// TIA Portal V17 export
// export: Created 2025-03-07T09:16:41.8974117Z, ExportSetting WithDefaults, DisplayName Totally Integrated Automation Portal, DisplayVersion V17 Update 8, DisplayName TIA Portal Openness, DisplayVersion V17 Update 8, DisplayName TIA Portal Version Control Interface, DisplayVersion V17, DisplayName SINAMICS Startdrive Advanced, DisplayVersion V17 SP2, DisplayName SINAMICS Startdrive G110M, G120, G120C, G120D, G120P, G115D, DisplayVersion V17 SP2, DisplayName SINAMICS Startdrive G130, G150, S120, S150, SINAMICS MV, S210, DisplayVersion V17 SP2, DisplayName STEP 7 Professional, DisplayVersion V17 Update 8, DisplayName SINUMERIK ONE STEP 7 Toolbox, DisplayVersion V17 Update 12, DisplayName SINUMERIK 840D sl STEP 7 Toolbox, DisplayVersion V17 Update 12, DisplayName STEP 7 Safety, DisplayVersion V17 Update 6, DisplayName WinCC Advanced, DisplayVersion V17 Update 8
FUNCTION "FC2440_GLOBAL_DATA_CLADDING" : Void   // FC2440, LAD
{ S7_Optimized_Access := 'FALSE' }
AUTHOR : ETXETAR
VERSION : 1.0
// stored: AutoNumber false, IsIECCheckEnabled false, SetENOAutomatically false, UDAEnableTagReadback false
   VAR_TEMP
      OPTION_ON : Bool;
      OPTION_OFF : Bool;
   END_VAR
   VAR_TEMP   // added for the SCL form of the ladder/FBD networks
      _w1 : Bool;
      _w2 : Bool;
      _w3 : Bool;
      _w4 : Bool;
   END_VAR
BEGIN

REGION Network 1: OPTIONS OFF
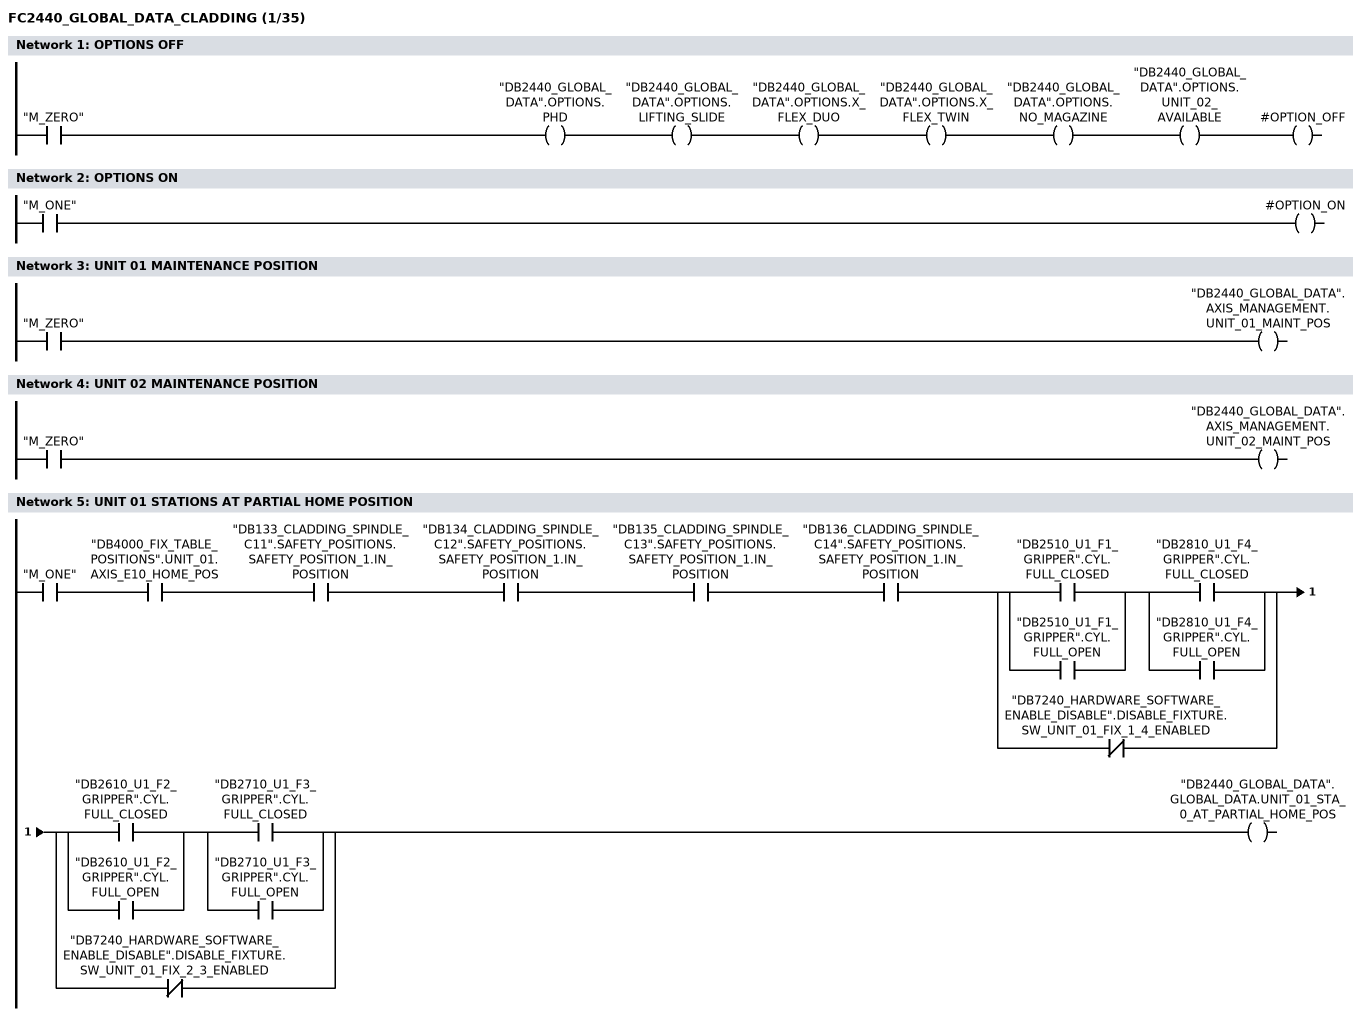
   RUNG wire#powerrail
      Contact( "M_ZERO" )
      Coil( "DB2440_GLOBAL_DATA".OPTIONS.PHD )
      Coil( "DB2440_GLOBAL_DATA".OPTIONS.LIFTING_SLIDE )
      Coil( "DB2440_GLOBAL_DATA".OPTIONS.X_FLEX_DUO )
      Coil( "DB2440_GLOBAL_DATA".OPTIONS.X_FLEX_TWIN )
      Coil( "DB2440_GLOBAL_DATA".OPTIONS.NO_MAGAZINE )
      Coil( "DB2440_GLOBAL_DATA".OPTIONS.UNIT_02_AVAILABLE )
      Coil( #OPTION_OFF )
   END_RUNG
   // the same network as SCL:
   "DB2440_GLOBAL_DATA".OPTIONS.PHD := "M_ZERO";
   "DB2440_GLOBAL_DATA".OPTIONS.LIFTING_SLIDE := "M_ZERO";
   "DB2440_GLOBAL_DATA".OPTIONS.X_FLEX_DUO := "M_ZERO";
   "DB2440_GLOBAL_DATA".OPTIONS.X_FLEX_TWIN := "M_ZERO";
   "DB2440_GLOBAL_DATA".OPTIONS.NO_MAGAZINE := "M_ZERO";
   "DB2440_GLOBAL_DATA".OPTIONS.UNIT_02_AVAILABLE := "M_ZERO";
   #OPTION_OFF := "M_ZERO";
END_REGION

REGION Network 2: OPTIONS ON
   RUNG wire#powerrail
      Contact( "M_ONE" )
      Coil( #OPTION_ON )
   END_RUNG
   // the same network as SCL:
   #OPTION_ON := "M_ONE";
END_REGION

REGION Network 3: UNIT 01 MAINTENANCE POSITION
   RUNG wire#powerrail
      Contact( "M_ZERO" )
      Coil( "DB2440_GLOBAL_DATA".AXIS_MANAGEMENT.UNIT_01_MAINT_POS )
   END_RUNG
   // the same network as SCL:
   "DB2440_GLOBAL_DATA".AXIS_MANAGEMENT.UNIT_01_MAINT_POS := "M_ZERO";
END_REGION

REGION Network 4: UNIT 02 MAINTENANCE POSITION
   RUNG wire#powerrail
      Contact( "M_ZERO" )
      Coil( "DB2440_GLOBAL_DATA".AXIS_MANAGEMENT.UNIT_02_MAINT_POS )
   END_RUNG
   // the same network as SCL:
   "DB2440_GLOBAL_DATA".AXIS_MANAGEMENT.UNIT_02_MAINT_POS := "M_ZERO";
END_REGION

REGION Network 5: UNIT 01 STATIONS AT PARTIAL HOME POSITION
   RUNG wire#powerrail
      Contact( "M_ONE" )
      Contact( "DB4000_FIX_TABLE_POSITIONS".UNIT_01.AXIS_E10_HOME_POS )
      Contact( "DB133_CLADDING_SPINDLE_C11".SAFETY_POSITIONS.SAFETY_POSITION_1.IN_POSITION )
      Contact( "DB134_CLADDING_SPINDLE_C12".SAFETY_POSITIONS.SAFETY_POSITION_1.IN_POSITION )
      Contact( "DB135_CLADDING_SPINDLE_C13".SAFETY_POSITIONS.SAFETY_POSITION_1.IN_POSITION )
      Contact( "DB136_CLADDING_SPINDLE_C14".SAFETY_POSITIONS.SAFETY_POSITION_1.IN_POSITION )
      wire#w1
      Contact( "DB2510_U1_F1_GRIPPER".CYL.FULL_CLOSED )
      wire#w2
      Contact( "DB2810_U1_F4_GRIPPER".CYL.FULL_CLOSED )
      wire#w3
      Contact( "DB2610_U1_F2_GRIPPER".CYL.FULL_CLOSED )
      wire#w4
      Contact( "DB2710_U1_F3_GRIPPER".CYL.FULL_CLOSED )
      wire#w5
      Coil( "DB2440_GLOBAL_DATA".GLOBAL_DATA.UNIT_01_STA_0_AT_PARTIAL_HOME_POS )
   END_RUNG
   RUNG wire#w1
      Contact( "DB2510_U1_F1_GRIPPER".CYL.FULL_OPEN )
   END_RUNG wire#w2
   RUNG wire#w2
      Contact( "DB2810_U1_F4_GRIPPER".CYL.FULL_OPEN )
   END_RUNG wire#w3
   RUNG wire#w1
      I_Contact( "DB7240_HARDWARE_SOFTWARE_ENABLE_DISABLE".DISABLE_FIXTURE.SW_UNIT_01_FIX_1_4_ENABLED )
   END_RUNG wire#w3
   RUNG wire#w3
      Contact( "DB2610_U1_F2_GRIPPER".CYL.FULL_OPEN )
   END_RUNG wire#w4
   RUNG wire#w4
      Contact( "DB2710_U1_F3_GRIPPER".CYL.FULL_OPEN )
   END_RUNG wire#w5
   RUNG wire#w3
      I_Contact( "DB7240_HARDWARE_SOFTWARE_ENABLE_DISABLE".DISABLE_FIXTURE.SW_UNIT_01_FIX_2_3_ENABLED )
   END_RUNG wire#w5
   // the same network as SCL:
   "DB2440_GLOBAL_DATA".GLOBAL_DATA.UNIT_01_STA_0_AT_PARTIAL_HOME_POS := "M_ONE" AND "DB4000_FIX_TABLE_POSITIONS".UNIT_01.AXIS_E10_HOME_POS AND "DB133_CLADDING_SPINDLE_C11".SAFETY_POSITIONS.SAFETY_POSITION_1.IN_POSITION AND "DB134_CLADDING_SPINDLE_C12".SAFETY_POSITIONS.SAFETY_POSITION_1.IN_POSITION AND "DB135_CLADDING_SPINDLE_C13".SAFETY_POSITIONS.SAFETY_POSITION_1.IN_POSITION AND "DB136_CLADDING_SPINDLE_C14".SAFETY_POSITIONS.SAFETY_POSITION_1.IN_POSITION AND ((("DB2510_U1_F1_GRIPPER".CYL.FULL_CLOSED OR "DB2510_U1_F1_GRIPPER".CYL.FULL_OPEN) AND ("DB2810_U1_F4_GRIPPER".CYL.FULL_CLOSED OR "DB2810_U1_F4_GRIPPER".CYL.FULL_OPEN)) OR NOT "DB7240_HARDWARE_SOFTWARE_ENABLE_DISABLE".DISABLE_FIXTURE.SW_UNIT_01_FIX_1_4_ENABLED) AND ((("DB2610_U1_F2_GRIPPER".CYL.FULL_CLOSED OR "DB2610_U1_F2_GRIPPER".CYL.FULL_OPEN) AND ("DB2710_U1_F3_GRIPPER".CYL.FULL_CLOSED OR "DB2710_U1_F3_GRIPPER".CYL.FULL_OPEN)) OR NOT "DB7240_HARDWARE_SOFTWARE_ENABLE_DISABLE".DISABLE_FIXTURE.SW_UNIT_01_FIX_2_3_ENABLED);
END_REGION

REGION Network 6: UNIT 01 STATIONS AT HOME POSITION
   // CILINDERS AND B13
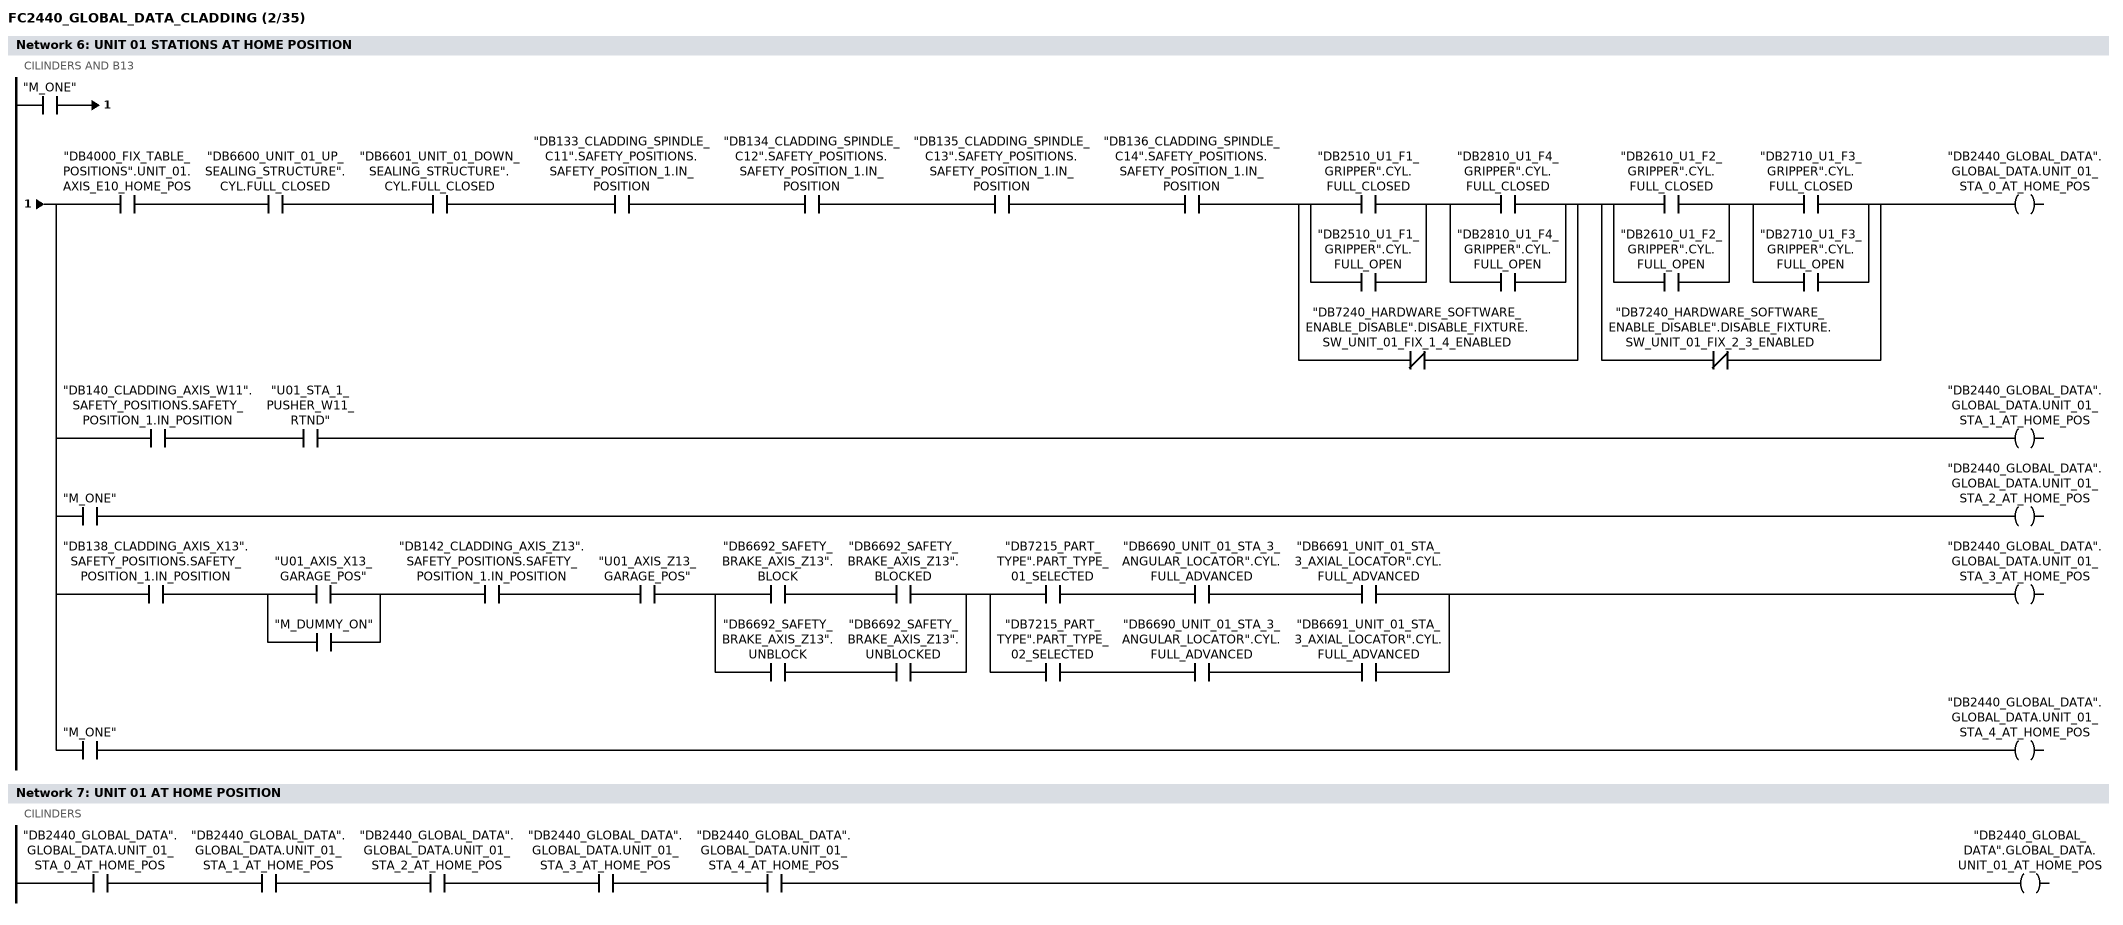
   RUNG wire#powerrail
      Contact( "M_ONE" )
      wire#w1
      Contact( "DB4000_FIX_TABLE_POSITIONS".UNIT_01.AXIS_E10_HOME_POS )
      Contact( "DB6600_UNIT_01_UP_SEALING_STRUCTURE".CYL.FULL_CLOSED )
      Contact( "DB6601_UNIT_01_DOWN_SEALING_STRUCTURE".CYL.FULL_CLOSED )
      Contact( "DB133_CLADDING_SPINDLE_C11".SAFETY_POSITIONS.SAFETY_POSITION_1.IN_POSITION )
      Contact( "DB134_CLADDING_SPINDLE_C12".SAFETY_POSITIONS.SAFETY_POSITION_1.IN_POSITION )
      Contact( "DB135_CLADDING_SPINDLE_C13".SAFETY_POSITIONS.SAFETY_POSITION_1.IN_POSITION )
      Contact( "DB136_CLADDING_SPINDLE_C14".SAFETY_POSITIONS.SAFETY_POSITION_1.IN_POSITION )
      wire#w2
      Contact( "DB2510_U1_F1_GRIPPER".CYL.FULL_CLOSED )
      wire#w3
      Contact( "DB2810_U1_F4_GRIPPER".CYL.FULL_CLOSED )
      wire#w4
      Contact( "DB2610_U1_F2_GRIPPER".CYL.FULL_CLOSED )
      wire#w5
      Contact( "DB2710_U1_F3_GRIPPER".CYL.FULL_CLOSED )
      wire#w6
      Coil( "DB2440_GLOBAL_DATA".GLOBAL_DATA.UNIT_01_STA_0_AT_HOME_POS )
   END_RUNG
   RUNG wire#w2
      Contact( "DB2510_U1_F1_GRIPPER".CYL.FULL_OPEN )
   END_RUNG wire#w3
   RUNG wire#w3
      Contact( "DB2810_U1_F4_GRIPPER".CYL.FULL_OPEN )
   END_RUNG wire#w4
   RUNG wire#w2
      I_Contact( "DB7240_HARDWARE_SOFTWARE_ENABLE_DISABLE".DISABLE_FIXTURE.SW_UNIT_01_FIX_1_4_ENABLED )
   END_RUNG wire#w4
   RUNG wire#w4
      Contact( "DB2610_U1_F2_GRIPPER".CYL.FULL_OPEN )
   END_RUNG wire#w5
   RUNG wire#w5
      Contact( "DB2710_U1_F3_GRIPPER".CYL.FULL_OPEN )
   END_RUNG wire#w6
   RUNG wire#w4
      I_Contact( "DB7240_HARDWARE_SOFTWARE_ENABLE_DISABLE".DISABLE_FIXTURE.SW_UNIT_01_FIX_2_3_ENABLED )
   END_RUNG wire#w6
   RUNG wire#w1
      Contact( "DB140_CLADDING_AXIS_W11".SAFETY_POSITIONS.SAFETY_POSITION_1.IN_POSITION )
      Contact( "U01_STA_1_PUSHER_W11_RTND" )
      Coil( "DB2440_GLOBAL_DATA".GLOBAL_DATA.UNIT_01_STA_1_AT_HOME_POS )
   END_RUNG
   RUNG wire#w1
      Contact( "M_ONE" )
      Coil( "DB2440_GLOBAL_DATA".GLOBAL_DATA.UNIT_01_STA_2_AT_HOME_POS )
   END_RUNG
   RUNG wire#w1
      Contact( "DB138_CLADDING_AXIS_X13".SAFETY_POSITIONS.SAFETY_POSITION_1.IN_POSITION )
      wire#w7
      Contact( "U01_AXIS_X13_GARAGE_POS" )
      wire#w8
      Contact( "DB142_CLADDING_AXIS_Z13".SAFETY_POSITIONS.SAFETY_POSITION_1.IN_POSITION )
      Contact( "U01_AXIS_Z13_GARAGE_POS" )
      wire#w9
      Contact( "DB6692_SAFETY_BRAKE_AXIS_Z13".BLOCK )
      Contact( "DB6692_SAFETY_BRAKE_AXIS_Z13".BLOCKED )
      wire#w10
      Contact( "DB7215_PART_TYPE".PART_TYPE_01_SELECTED )
      Contact( "DB6690_UNIT_01_STA_3_ANGULAR_LOCATOR".CYL.FULL_ADVANCED )
      Contact( "DB6691_UNIT_01_STA_3_AXIAL_LOCATOR".CYL.FULL_ADVANCED )
      wire#w11
      Coil( "DB2440_GLOBAL_DATA".GLOBAL_DATA.UNIT_01_STA_3_AT_HOME_POS )
   END_RUNG
   RUNG wire#w7
      Contact( "M_DUMMY_ON" )
   END_RUNG wire#w8
   RUNG wire#w9
      Contact( "DB6692_SAFETY_BRAKE_AXIS_Z13".UNBLOCK )
      Contact( "DB6692_SAFETY_BRAKE_AXIS_Z13".UNBLOCKED )
   END_RUNG wire#w10
   RUNG wire#w10
      Contact( "DB7215_PART_TYPE".PART_TYPE_02_SELECTED )
      Contact( "DB6690_UNIT_01_STA_3_ANGULAR_LOCATOR".CYL.FULL_ADVANCED )
      Contact( "DB6691_UNIT_01_STA_3_AXIAL_LOCATOR".CYL.FULL_ADVANCED )
   END_RUNG wire#w11
   RUNG wire#w1
      Contact( "M_ONE" )
      Coil( "DB2440_GLOBAL_DATA".GLOBAL_DATA.UNIT_01_STA_4_AT_HOME_POS )
   END_RUNG
   // the same network as SCL:
   "DB2440_GLOBAL_DATA".GLOBAL_DATA.UNIT_01_STA_0_AT_HOME_POS := "M_ONE" AND "DB4000_FIX_TABLE_POSITIONS".UNIT_01.AXIS_E10_HOME_POS AND "DB6600_UNIT_01_UP_SEALING_STRUCTURE".CYL.FULL_CLOSED AND "DB6601_UNIT_01_DOWN_SEALING_STRUCTURE".CYL.FULL_CLOSED AND "DB133_CLADDING_SPINDLE_C11".SAFETY_POSITIONS.SAFETY_POSITION_1.IN_POSITION AND "DB134_CLADDING_SPINDLE_C12".SAFETY_POSITIONS.SAFETY_POSITION_1.IN_POSITION AND "DB135_CLADDING_SPINDLE_C13".SAFETY_POSITIONS.SAFETY_POSITION_1.IN_POSITION AND "DB136_CLADDING_SPINDLE_C14".SAFETY_POSITIONS.SAFETY_POSITION_1.IN_POSITION AND ((("DB2510_U1_F1_GRIPPER".CYL.FULL_CLOSED OR "DB2510_U1_F1_GRIPPER".CYL.FULL_OPEN) AND ("DB2810_U1_F4_GRIPPER".CYL.FULL_CLOSED OR "DB2810_U1_F4_GRIPPER".CYL.FULL_OPEN)) OR NOT "DB7240_HARDWARE_SOFTWARE_ENABLE_DISABLE".DISABLE_FIXTURE.SW_UNIT_01_FIX_1_4_ENABLED) AND ((("DB2610_U1_F2_GRIPPER".CYL.FULL_CLOSED OR "DB2610_U1_F2_GRIPPER".CYL.FULL_OPEN) AND ("DB2710_U1_F3_GRIPPER".CYL.FULL_CLOSED OR "DB2710_U1_F3_GRIPPER".CYL.FULL_OPEN)) OR NOT "DB7240_HARDWARE_SOFTWARE_ENABLE_DISABLE".DISABLE_FIXTURE.SW_UNIT_01_FIX_2_3_ENABLED);
   "DB2440_GLOBAL_DATA".GLOBAL_DATA.UNIT_01_STA_1_AT_HOME_POS := "M_ONE" AND "DB140_CLADDING_AXIS_W11".SAFETY_POSITIONS.SAFETY_POSITION_1.IN_POSITION AND "U01_STA_1_PUSHER_W11_RTND";
   "DB2440_GLOBAL_DATA".GLOBAL_DATA.UNIT_01_STA_2_AT_HOME_POS := "M_ONE" AND "M_ONE";
   "DB2440_GLOBAL_DATA".GLOBAL_DATA.UNIT_01_STA_3_AT_HOME_POS := "M_ONE" AND "DB138_CLADDING_AXIS_X13".SAFETY_POSITIONS.SAFETY_POSITION_1.IN_POSITION AND ("U01_AXIS_X13_GARAGE_POS" OR "M_DUMMY_ON") AND "DB142_CLADDING_AXIS_Z13".SAFETY_POSITIONS.SAFETY_POSITION_1.IN_POSITION AND "U01_AXIS_Z13_GARAGE_POS" AND (("DB6692_SAFETY_BRAKE_AXIS_Z13".BLOCK AND "DB6692_SAFETY_BRAKE_AXIS_Z13".BLOCKED) OR ("DB6692_SAFETY_BRAKE_AXIS_Z13".UNBLOCK AND "DB6692_SAFETY_BRAKE_AXIS_Z13".UNBLOCKED)) AND (("DB7215_PART_TYPE".PART_TYPE_01_SELECTED AND "DB6690_UNIT_01_STA_3_ANGULAR_LOCATOR".CYL.FULL_ADVANCED AND "DB6691_UNIT_01_STA_3_AXIAL_LOCATOR".CYL.FULL_ADVANCED) OR ("DB7215_PART_TYPE".PART_TYPE_02_SELECTED AND "DB6690_UNIT_01_STA_3_ANGULAR_LOCATOR".CYL.FULL_ADVANCED AND "DB6691_UNIT_01_STA_3_AXIAL_LOCATOR".CYL.FULL_ADVANCED));
   "DB2440_GLOBAL_DATA".GLOBAL_DATA.UNIT_01_STA_4_AT_HOME_POS := "M_ONE" AND "M_ONE";
END_REGION

REGION Network 7: UNIT 01 AT HOME POSITION
   // CILINDERS
   RUNG wire#powerrail
      Contact( "DB2440_GLOBAL_DATA".GLOBAL_DATA.UNIT_01_STA_0_AT_HOME_POS )
      Contact( "DB2440_GLOBAL_DATA".GLOBAL_DATA.UNIT_01_STA_1_AT_HOME_POS )
      Contact( "DB2440_GLOBAL_DATA".GLOBAL_DATA.UNIT_01_STA_2_AT_HOME_POS )
      Contact( "DB2440_GLOBAL_DATA".GLOBAL_DATA.UNIT_01_STA_3_AT_HOME_POS )
      Contact( "DB2440_GLOBAL_DATA".GLOBAL_DATA.UNIT_01_STA_4_AT_HOME_POS )
      Coil( "DB2440_GLOBAL_DATA".GLOBAL_DATA.UNIT_01_AT_HOME_POS )
   END_RUNG
   // the same network as SCL:
   "DB2440_GLOBAL_DATA".GLOBAL_DATA.UNIT_01_AT_HOME_POS := "DB2440_GLOBAL_DATA".GLOBAL_DATA.UNIT_01_STA_0_AT_HOME_POS AND "DB2440_GLOBAL_DATA".GLOBAL_DATA.UNIT_01_STA_1_AT_HOME_POS AND "DB2440_GLOBAL_DATA".GLOBAL_DATA.UNIT_01_STA_2_AT_HOME_POS AND "DB2440_GLOBAL_DATA".GLOBAL_DATA.UNIT_01_STA_3_AT_HOME_POS AND "DB2440_GLOBAL_DATA".GLOBAL_DATA.UNIT_01_STA_4_AT_HOME_POS;
END_REGION

REGION Network 8: UNIT 02 STATIONS AT PARTIAL HOME POSITION
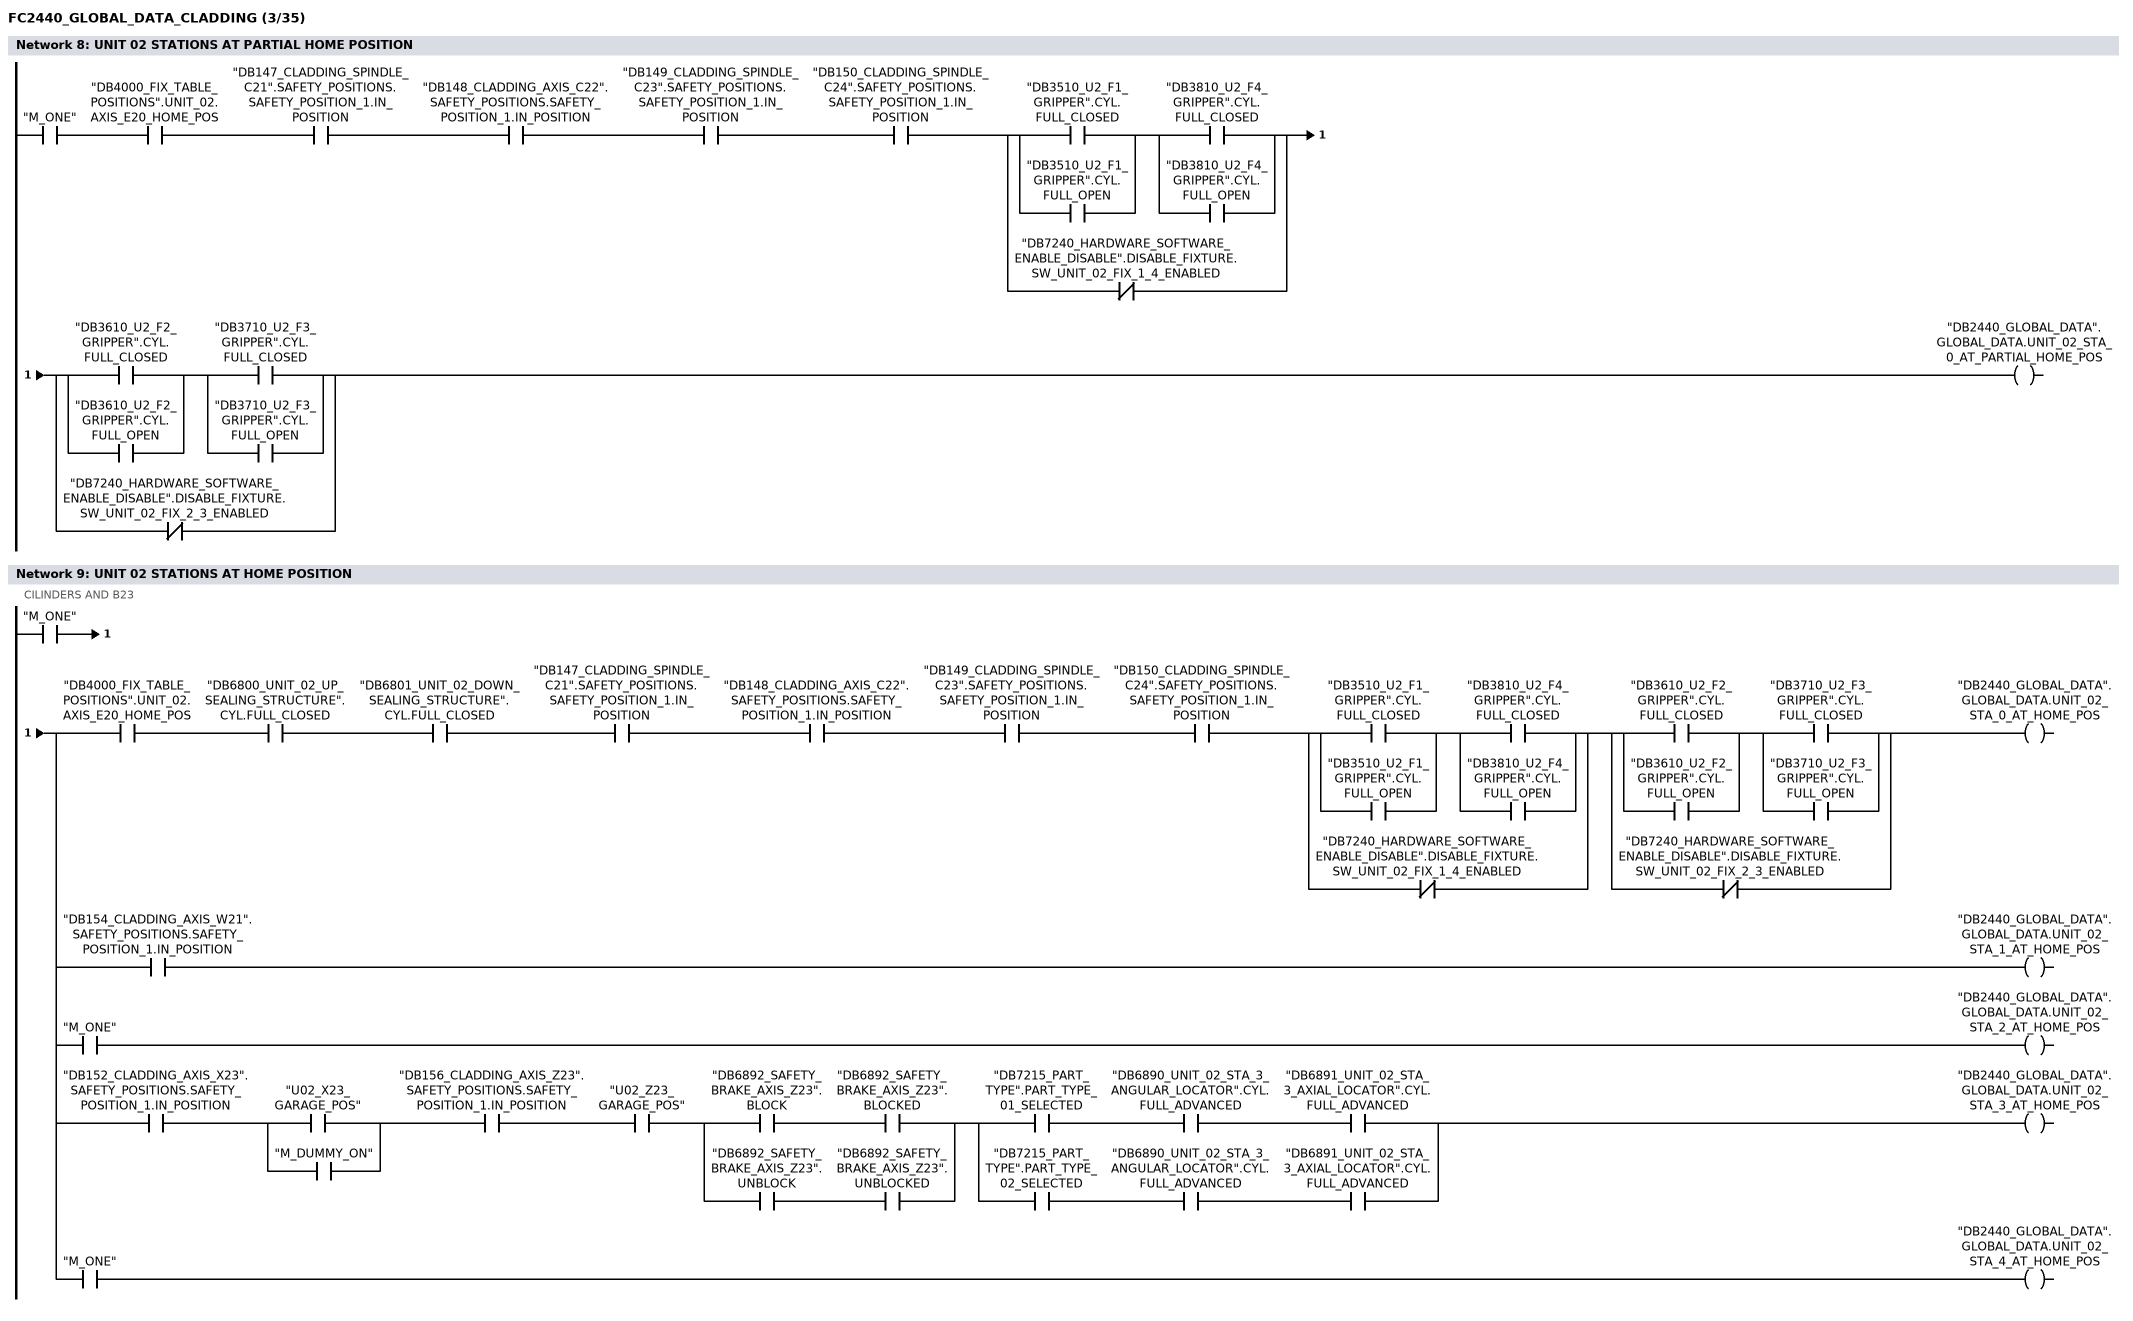
   RUNG wire#powerrail
      Contact( "M_ONE" )
      Contact( "DB4000_FIX_TABLE_POSITIONS".UNIT_02.AXIS_E20_HOME_POS )
      Contact( "DB147_CLADDING_SPINDLE_C21".SAFETY_POSITIONS.SAFETY_POSITION_1.IN_POSITION )
      Contact( "DB148_CLADDING_AXIS_C22".SAFETY_POSITIONS.SAFETY_POSITION_1.IN_POSITION )
      Contact( "DB149_CLADDING_SPINDLE_C23".SAFETY_POSITIONS.SAFETY_POSITION_1.IN_POSITION )
      Contact( "DB150_CLADDING_SPINDLE_C24".SAFETY_POSITIONS.SAFETY_POSITION_1.IN_POSITION )
      wire#w1
      Contact( "DB3510_U2_F1_GRIPPER".CYL.FULL_CLOSED )
      wire#w2
      Contact( "DB3810_U2_F4_GRIPPER".CYL.FULL_CLOSED )
      wire#w3
      Contact( "DB3610_U2_F2_GRIPPER".CYL.FULL_CLOSED )
      wire#w4
      Contact( "DB3710_U2_F3_GRIPPER".CYL.FULL_CLOSED )
      wire#w5
      Coil( "DB2440_GLOBAL_DATA".GLOBAL_DATA.UNIT_02_STA_0_AT_PARTIAL_HOME_POS )
   END_RUNG
   RUNG wire#w1
      Contact( "DB3510_U2_F1_GRIPPER".CYL.FULL_OPEN )
   END_RUNG wire#w2
   RUNG wire#w2
      Contact( "DB3810_U2_F4_GRIPPER".CYL.FULL_OPEN )
   END_RUNG wire#w3
   RUNG wire#w1
      I_Contact( "DB7240_HARDWARE_SOFTWARE_ENABLE_DISABLE".DISABLE_FIXTURE.SW_UNIT_02_FIX_1_4_ENABLED )
   END_RUNG wire#w3
   RUNG wire#w3
      Contact( "DB3610_U2_F2_GRIPPER".CYL.FULL_OPEN )
   END_RUNG wire#w4
   RUNG wire#w4
      Contact( "DB3710_U2_F3_GRIPPER".CYL.FULL_OPEN )
   END_RUNG wire#w5
   RUNG wire#w3
      I_Contact( "DB7240_HARDWARE_SOFTWARE_ENABLE_DISABLE".DISABLE_FIXTURE.SW_UNIT_02_FIX_2_3_ENABLED )
   END_RUNG wire#w5
   // the same network as SCL:
   "DB2440_GLOBAL_DATA".GLOBAL_DATA.UNIT_02_STA_0_AT_PARTIAL_HOME_POS := "M_ONE" AND "DB4000_FIX_TABLE_POSITIONS".UNIT_02.AXIS_E20_HOME_POS AND "DB147_CLADDING_SPINDLE_C21".SAFETY_POSITIONS.SAFETY_POSITION_1.IN_POSITION AND "DB148_CLADDING_AXIS_C22".SAFETY_POSITIONS.SAFETY_POSITION_1.IN_POSITION AND "DB149_CLADDING_SPINDLE_C23".SAFETY_POSITIONS.SAFETY_POSITION_1.IN_POSITION AND "DB150_CLADDING_SPINDLE_C24".SAFETY_POSITIONS.SAFETY_POSITION_1.IN_POSITION AND ((("DB3510_U2_F1_GRIPPER".CYL.FULL_CLOSED OR "DB3510_U2_F1_GRIPPER".CYL.FULL_OPEN) AND ("DB3810_U2_F4_GRIPPER".CYL.FULL_CLOSED OR "DB3810_U2_F4_GRIPPER".CYL.FULL_OPEN)) OR NOT "DB7240_HARDWARE_SOFTWARE_ENABLE_DISABLE".DISABLE_FIXTURE.SW_UNIT_02_FIX_1_4_ENABLED) AND ((("DB3610_U2_F2_GRIPPER".CYL.FULL_CLOSED OR "DB3610_U2_F2_GRIPPER".CYL.FULL_OPEN) AND ("DB3710_U2_F3_GRIPPER".CYL.FULL_CLOSED OR "DB3710_U2_F3_GRIPPER".CYL.FULL_OPEN)) OR NOT "DB7240_HARDWARE_SOFTWARE_ENABLE_DISABLE".DISABLE_FIXTURE.SW_UNIT_02_FIX_2_3_ENABLED);
END_REGION

REGION Network 9: UNIT 02 STATIONS AT HOME POSITION
   // CILINDERS AND B23
   RUNG wire#powerrail
      Contact( "M_ONE" )
      wire#w1
      Contact( "DB4000_FIX_TABLE_POSITIONS".UNIT_02.AXIS_E20_HOME_POS )
      Contact( "DB6800_UNIT_02_UP_SEALING_STRUCTURE".CYL.FULL_CLOSED )
      Contact( "DB6801_UNIT_02_DOWN_SEALING_STRUCTURE".CYL.FULL_CLOSED )
      Contact( "DB147_CLADDING_SPINDLE_C21".SAFETY_POSITIONS.SAFETY_POSITION_1.IN_POSITION )
      Contact( "DB148_CLADDING_AXIS_C22".SAFETY_POSITIONS.SAFETY_POSITION_1.IN_POSITION )
      Contact( "DB149_CLADDING_SPINDLE_C23".SAFETY_POSITIONS.SAFETY_POSITION_1.IN_POSITION )
      Contact( "DB150_CLADDING_SPINDLE_C24".SAFETY_POSITIONS.SAFETY_POSITION_1.IN_POSITION )
      wire#w2
      Contact( "DB3510_U2_F1_GRIPPER".CYL.FULL_CLOSED )
      wire#w3
      Contact( "DB3810_U2_F4_GRIPPER".CYL.FULL_CLOSED )
      wire#w4
      Contact( "DB3610_U2_F2_GRIPPER".CYL.FULL_CLOSED )
      wire#w5
      Contact( "DB3710_U2_F3_GRIPPER".CYL.FULL_CLOSED )
      wire#w6
      Coil( "DB2440_GLOBAL_DATA".GLOBAL_DATA.UNIT_02_STA_0_AT_HOME_POS )
   END_RUNG
   RUNG wire#w2
      Contact( "DB3510_U2_F1_GRIPPER".CYL.FULL_OPEN )
   END_RUNG wire#w3
   RUNG wire#w3
      Contact( "DB3810_U2_F4_GRIPPER".CYL.FULL_OPEN )
   END_RUNG wire#w4
   RUNG wire#w2
      I_Contact( "DB7240_HARDWARE_SOFTWARE_ENABLE_DISABLE".DISABLE_FIXTURE.SW_UNIT_02_FIX_1_4_ENABLED )
   END_RUNG wire#w4
   RUNG wire#w4
      Contact( "DB3610_U2_F2_GRIPPER".CYL.FULL_OPEN )
   END_RUNG wire#w5
   RUNG wire#w5
      Contact( "DB3710_U2_F3_GRIPPER".CYL.FULL_OPEN )
   END_RUNG wire#w6
   RUNG wire#w4
      I_Contact( "DB7240_HARDWARE_SOFTWARE_ENABLE_DISABLE".DISABLE_FIXTURE.SW_UNIT_02_FIX_2_3_ENABLED )
   END_RUNG wire#w6
   RUNG wire#w1
      Contact( "DB154_CLADDING_AXIS_W21".SAFETY_POSITIONS.SAFETY_POSITION_1.IN_POSITION )
      Coil( "DB2440_GLOBAL_DATA".GLOBAL_DATA.UNIT_02_STA_1_AT_HOME_POS )
   END_RUNG
   RUNG wire#w1
      Contact( "M_ONE" )
      Coil( "DB2440_GLOBAL_DATA".GLOBAL_DATA.UNIT_02_STA_2_AT_HOME_POS )
   END_RUNG
   RUNG wire#w1
      Contact( "DB152_CLADDING_AXIS_X23".SAFETY_POSITIONS.SAFETY_POSITION_1.IN_POSITION )
      wire#w7
      Contact( "U02_X23_GARAGE_POS" )
      wire#w8
      Contact( "DB156_CLADDING_AXIS_Z23".SAFETY_POSITIONS.SAFETY_POSITION_1.IN_POSITION )
      Contact( "U02_Z23_GARAGE_POS" )
      wire#w9
      Contact( "DB6892_SAFETY_BRAKE_AXIS_Z23".BLOCK )
      Contact( "DB6892_SAFETY_BRAKE_AXIS_Z23".BLOCKED )
      wire#w10
      Contact( "DB7215_PART_TYPE".PART_TYPE_01_SELECTED )
      Contact( "DB6890_UNIT_02_STA_3_ANGULAR_LOCATOR".CYL.FULL_ADVANCED )
      Contact( "DB6891_UNIT_02_STA_3_AXIAL_LOCATOR".CYL.FULL_ADVANCED )
      wire#w11
      Coil( "DB2440_GLOBAL_DATA".GLOBAL_DATA.UNIT_02_STA_3_AT_HOME_POS )
   END_RUNG
   RUNG wire#w7
      Contact( "M_DUMMY_ON" )
   END_RUNG wire#w8
   RUNG wire#w9
      Contact( "DB6892_SAFETY_BRAKE_AXIS_Z23".UNBLOCK )
      Contact( "DB6892_SAFETY_BRAKE_AXIS_Z23".UNBLOCKED )
   END_RUNG wire#w10
   RUNG wire#w10
      Contact( "DB7215_PART_TYPE".PART_TYPE_02_SELECTED )
      Contact( "DB6890_UNIT_02_STA_3_ANGULAR_LOCATOR".CYL.FULL_ADVANCED )
      Contact( "DB6891_UNIT_02_STA_3_AXIAL_LOCATOR".CYL.FULL_ADVANCED )
   END_RUNG wire#w11
   RUNG wire#w1
      Contact( "M_ONE" )
      Coil( "DB2440_GLOBAL_DATA".GLOBAL_DATA.UNIT_02_STA_4_AT_HOME_POS )
   END_RUNG
   // the same network as SCL:
   "DB2440_GLOBAL_DATA".GLOBAL_DATA.UNIT_02_STA_0_AT_HOME_POS := "M_ONE" AND "DB4000_FIX_TABLE_POSITIONS".UNIT_02.AXIS_E20_HOME_POS AND "DB6800_UNIT_02_UP_SEALING_STRUCTURE".CYL.FULL_CLOSED AND "DB6801_UNIT_02_DOWN_SEALING_STRUCTURE".CYL.FULL_CLOSED AND "DB147_CLADDING_SPINDLE_C21".SAFETY_POSITIONS.SAFETY_POSITION_1.IN_POSITION AND "DB148_CLADDING_AXIS_C22".SAFETY_POSITIONS.SAFETY_POSITION_1.IN_POSITION AND "DB149_CLADDING_SPINDLE_C23".SAFETY_POSITIONS.SAFETY_POSITION_1.IN_POSITION AND "DB150_CLADDING_SPINDLE_C24".SAFETY_POSITIONS.SAFETY_POSITION_1.IN_POSITION AND ((("DB3510_U2_F1_GRIPPER".CYL.FULL_CLOSED OR "DB3510_U2_F1_GRIPPER".CYL.FULL_OPEN) AND ("DB3810_U2_F4_GRIPPER".CYL.FULL_CLOSED OR "DB3810_U2_F4_GRIPPER".CYL.FULL_OPEN)) OR NOT "DB7240_HARDWARE_SOFTWARE_ENABLE_DISABLE".DISABLE_FIXTURE.SW_UNIT_02_FIX_1_4_ENABLED) AND ((("DB3610_U2_F2_GRIPPER".CYL.FULL_CLOSED OR "DB3610_U2_F2_GRIPPER".CYL.FULL_OPEN) AND ("DB3710_U2_F3_GRIPPER".CYL.FULL_CLOSED OR "DB3710_U2_F3_GRIPPER".CYL.FULL_OPEN)) OR NOT "DB7240_HARDWARE_SOFTWARE_ENABLE_DISABLE".DISABLE_FIXTURE.SW_UNIT_02_FIX_2_3_ENABLED);
   "DB2440_GLOBAL_DATA".GLOBAL_DATA.UNIT_02_STA_1_AT_HOME_POS := "M_ONE" AND "DB154_CLADDING_AXIS_W21".SAFETY_POSITIONS.SAFETY_POSITION_1.IN_POSITION;
   "DB2440_GLOBAL_DATA".GLOBAL_DATA.UNIT_02_STA_2_AT_HOME_POS := "M_ONE" AND "M_ONE";
   "DB2440_GLOBAL_DATA".GLOBAL_DATA.UNIT_02_STA_3_AT_HOME_POS := "M_ONE" AND "DB152_CLADDING_AXIS_X23".SAFETY_POSITIONS.SAFETY_POSITION_1.IN_POSITION AND ("U02_X23_GARAGE_POS" OR "M_DUMMY_ON") AND "DB156_CLADDING_AXIS_Z23".SAFETY_POSITIONS.SAFETY_POSITION_1.IN_POSITION AND "U02_Z23_GARAGE_POS" AND (("DB6892_SAFETY_BRAKE_AXIS_Z23".BLOCK AND "DB6892_SAFETY_BRAKE_AXIS_Z23".BLOCKED) OR ("DB6892_SAFETY_BRAKE_AXIS_Z23".UNBLOCK AND "DB6892_SAFETY_BRAKE_AXIS_Z23".UNBLOCKED)) AND (("DB7215_PART_TYPE".PART_TYPE_01_SELECTED AND "DB6890_UNIT_02_STA_3_ANGULAR_LOCATOR".CYL.FULL_ADVANCED AND "DB6891_UNIT_02_STA_3_AXIAL_LOCATOR".CYL.FULL_ADVANCED) OR ("DB7215_PART_TYPE".PART_TYPE_02_SELECTED AND "DB6890_UNIT_02_STA_3_ANGULAR_LOCATOR".CYL.FULL_ADVANCED AND "DB6891_UNIT_02_STA_3_AXIAL_LOCATOR".CYL.FULL_ADVANCED));
   "DB2440_GLOBAL_DATA".GLOBAL_DATA.UNIT_02_STA_4_AT_HOME_POS := "M_ONE" AND "M_ONE";
END_REGION

REGION Network 10: UNIT 02 AT HOME POSITION
   // CILINDERS
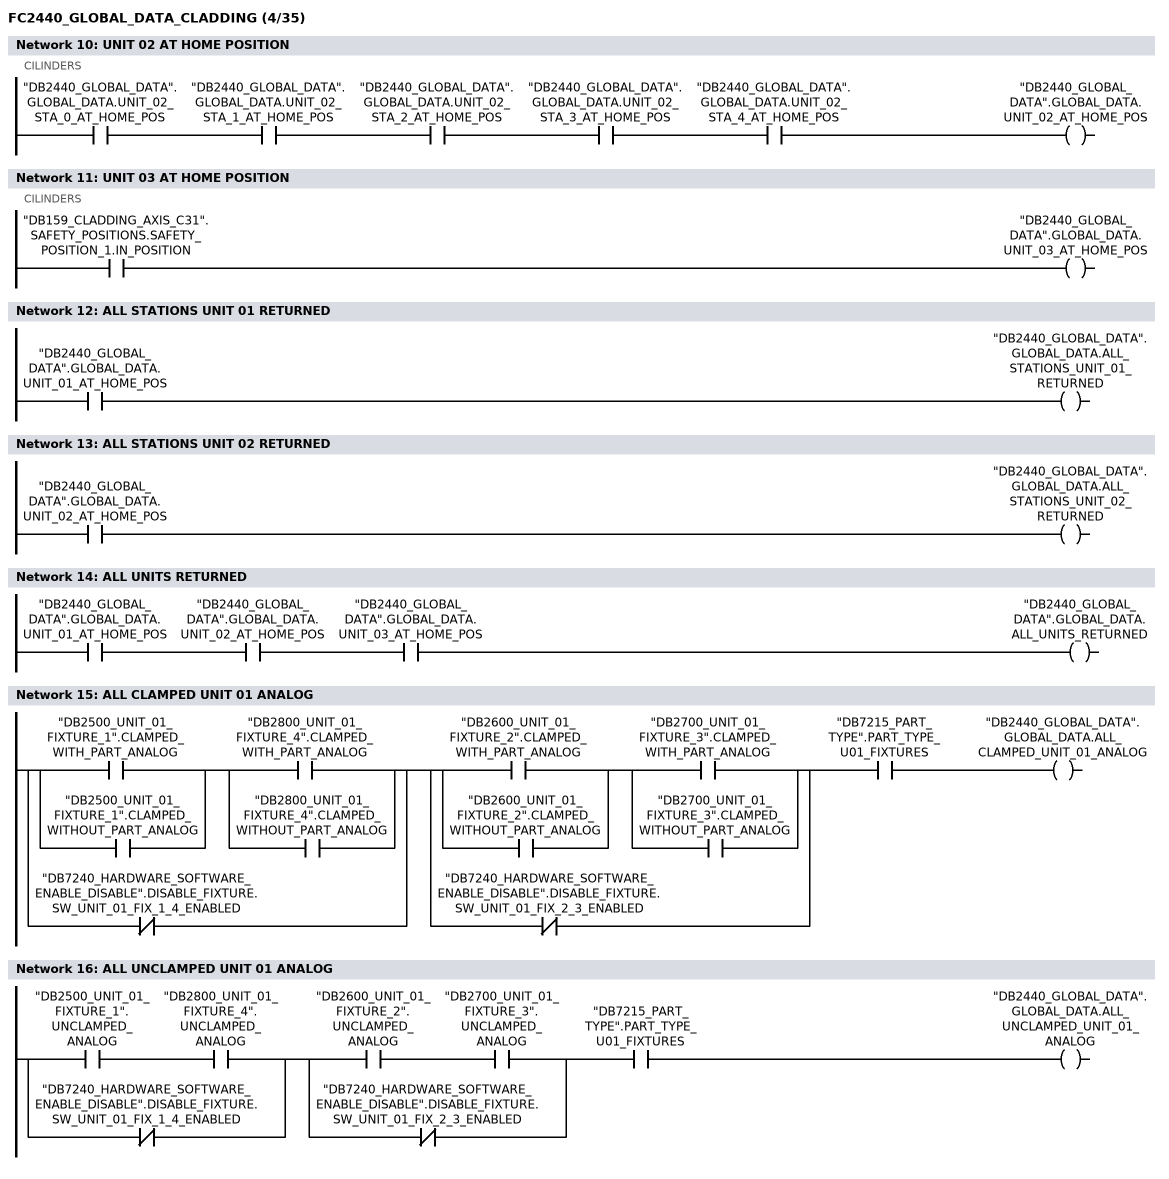
   RUNG wire#powerrail
      Contact( "DB2440_GLOBAL_DATA".GLOBAL_DATA.UNIT_02_STA_0_AT_HOME_POS )
      Contact( "DB2440_GLOBAL_DATA".GLOBAL_DATA.UNIT_02_STA_1_AT_HOME_POS )
      Contact( "DB2440_GLOBAL_DATA".GLOBAL_DATA.UNIT_02_STA_2_AT_HOME_POS )
      Contact( "DB2440_GLOBAL_DATA".GLOBAL_DATA.UNIT_02_STA_3_AT_HOME_POS )
      Contact( "DB2440_GLOBAL_DATA".GLOBAL_DATA.UNIT_02_STA_4_AT_HOME_POS )
      Coil( "DB2440_GLOBAL_DATA".GLOBAL_DATA.UNIT_02_AT_HOME_POS )
   END_RUNG
   // the same network as SCL:
   "DB2440_GLOBAL_DATA".GLOBAL_DATA.UNIT_02_AT_HOME_POS := "DB2440_GLOBAL_DATA".GLOBAL_DATA.UNIT_02_STA_0_AT_HOME_POS AND "DB2440_GLOBAL_DATA".GLOBAL_DATA.UNIT_02_STA_1_AT_HOME_POS AND "DB2440_GLOBAL_DATA".GLOBAL_DATA.UNIT_02_STA_2_AT_HOME_POS AND "DB2440_GLOBAL_DATA".GLOBAL_DATA.UNIT_02_STA_3_AT_HOME_POS AND "DB2440_GLOBAL_DATA".GLOBAL_DATA.UNIT_02_STA_4_AT_HOME_POS;
END_REGION

REGION Network 11: UNIT 03 AT HOME POSITION
   // CILINDERS
   RUNG wire#powerrail
      Contact( "DB159_CLADDING_AXIS_C31".SAFETY_POSITIONS.SAFETY_POSITION_1.IN_POSITION )
      Coil( "DB2440_GLOBAL_DATA".GLOBAL_DATA.UNIT_03_AT_HOME_POS )
   END_RUNG
   // the same network as SCL:
   "DB2440_GLOBAL_DATA".GLOBAL_DATA.UNIT_03_AT_HOME_POS := "DB159_CLADDING_AXIS_C31".SAFETY_POSITIONS.SAFETY_POSITION_1.IN_POSITION;
END_REGION

REGION Network 12: ALL STATIONS UNIT 01 RETURNED
   RUNG wire#powerrail
      Contact( "DB2440_GLOBAL_DATA".GLOBAL_DATA.UNIT_01_AT_HOME_POS )
      Coil( "DB2440_GLOBAL_DATA".GLOBAL_DATA.ALL_STATIONS_UNIT_01_RETURNED )
   END_RUNG
   // the same network as SCL:
   "DB2440_GLOBAL_DATA".GLOBAL_DATA.ALL_STATIONS_UNIT_01_RETURNED := "DB2440_GLOBAL_DATA".GLOBAL_DATA.UNIT_01_AT_HOME_POS;
END_REGION

REGION Network 13: ALL STATIONS UNIT 02 RETURNED
   RUNG wire#powerrail
      Contact( "DB2440_GLOBAL_DATA".GLOBAL_DATA.UNIT_02_AT_HOME_POS )
      Coil( "DB2440_GLOBAL_DATA".GLOBAL_DATA.ALL_STATIONS_UNIT_02_RETURNED )
   END_RUNG
   // the same network as SCL:
   "DB2440_GLOBAL_DATA".GLOBAL_DATA.ALL_STATIONS_UNIT_02_RETURNED := "DB2440_GLOBAL_DATA".GLOBAL_DATA.UNIT_02_AT_HOME_POS;
END_REGION

REGION Network 14: ALL UNITS RETURNED
   RUNG wire#powerrail
      Contact( "DB2440_GLOBAL_DATA".GLOBAL_DATA.UNIT_01_AT_HOME_POS )
      Contact( "DB2440_GLOBAL_DATA".GLOBAL_DATA.UNIT_02_AT_HOME_POS )
      Contact( "DB2440_GLOBAL_DATA".GLOBAL_DATA.UNIT_03_AT_HOME_POS )
      Coil( "DB2440_GLOBAL_DATA".GLOBAL_DATA.ALL_UNITS_RETURNED )
   END_RUNG
   // the same network as SCL:
   "DB2440_GLOBAL_DATA".GLOBAL_DATA.ALL_UNITS_RETURNED := "DB2440_GLOBAL_DATA".GLOBAL_DATA.UNIT_01_AT_HOME_POS AND "DB2440_GLOBAL_DATA".GLOBAL_DATA.UNIT_02_AT_HOME_POS AND "DB2440_GLOBAL_DATA".GLOBAL_DATA.UNIT_03_AT_HOME_POS;
END_REGION

REGION Network 15: ALL CLAMPED UNIT 01 ANALOG
   RUNG wire#powerrail
      Contact( "DB2500_UNIT_01_FIXTURE_1".CLAMPED_WITH_PART_ANALOG )
      wire#w1
      Contact( "DB2800_UNIT_01_FIXTURE_4".CLAMPED_WITH_PART_ANALOG )
      wire#w2
      Contact( "DB2600_UNIT_01_FIXTURE_2".CLAMPED_WITH_PART_ANALOG )
      wire#w3
      Contact( "DB2700_UNIT_01_FIXTURE_3".CLAMPED_WITH_PART_ANALOG )
      wire#w4
      Contact( "DB7215_PART_TYPE".PART_TYPE_U01_FIXTURES )
      Coil( "DB2440_GLOBAL_DATA".GLOBAL_DATA.ALL_CLAMPED_UNIT_01_ANALOG )
   END_RUNG
   RUNG wire#powerrail
      Contact( "DB2500_UNIT_01_FIXTURE_1".CLAMPED_WITHOUT_PART_ANALOG )
   END_RUNG wire#w1
   RUNG wire#w1
      Contact( "DB2800_UNIT_01_FIXTURE_4".CLAMPED_WITHOUT_PART_ANALOG )
   END_RUNG wire#w2
   RUNG wire#powerrail
      I_Contact( "DB7240_HARDWARE_SOFTWARE_ENABLE_DISABLE".DISABLE_FIXTURE.SW_UNIT_01_FIX_1_4_ENABLED )
   END_RUNG wire#w2
   RUNG wire#w2
      Contact( "DB2600_UNIT_01_FIXTURE_2".CLAMPED_WITHOUT_PART_ANALOG )
   END_RUNG wire#w3
   RUNG wire#w3
      Contact( "DB2700_UNIT_01_FIXTURE_3".CLAMPED_WITHOUT_PART_ANALOG )
   END_RUNG wire#w4
   RUNG wire#w2
      I_Contact( "DB7240_HARDWARE_SOFTWARE_ENABLE_DISABLE".DISABLE_FIXTURE.SW_UNIT_01_FIX_2_3_ENABLED )
   END_RUNG wire#w4
   // the same network as SCL:
   "DB2440_GLOBAL_DATA".GLOBAL_DATA.ALL_CLAMPED_UNIT_01_ANALOG := ((("DB2500_UNIT_01_FIXTURE_1".CLAMPED_WITH_PART_ANALOG OR "DB2500_UNIT_01_FIXTURE_1".CLAMPED_WITHOUT_PART_ANALOG) AND ("DB2800_UNIT_01_FIXTURE_4".CLAMPED_WITH_PART_ANALOG OR "DB2800_UNIT_01_FIXTURE_4".CLAMPED_WITHOUT_PART_ANALOG)) OR NOT "DB7240_HARDWARE_SOFTWARE_ENABLE_DISABLE".DISABLE_FIXTURE.SW_UNIT_01_FIX_1_4_ENABLED) AND ((("DB2600_UNIT_01_FIXTURE_2".CLAMPED_WITH_PART_ANALOG OR "DB2600_UNIT_01_FIXTURE_2".CLAMPED_WITHOUT_PART_ANALOG) AND ("DB2700_UNIT_01_FIXTURE_3".CLAMPED_WITH_PART_ANALOG OR "DB2700_UNIT_01_FIXTURE_3".CLAMPED_WITHOUT_PART_ANALOG)) OR NOT "DB7240_HARDWARE_SOFTWARE_ENABLE_DISABLE".DISABLE_FIXTURE.SW_UNIT_01_FIX_2_3_ENABLED) AND "DB7215_PART_TYPE".PART_TYPE_U01_FIXTURES;
END_REGION

REGION Network 16: ALL UNCLAMPED UNIT 01 ANALOG
   RUNG wire#powerrail
      Contact( "DB2500_UNIT_01_FIXTURE_1".UNCLAMPED_ANALOG )
      Contact( "DB2800_UNIT_01_FIXTURE_4".UNCLAMPED_ANALOG )
      wire#w1
      Contact( "DB2600_UNIT_01_FIXTURE_2".UNCLAMPED_ANALOG )
      Contact( "DB2700_UNIT_01_FIXTURE_3".UNCLAMPED_ANALOG )
      wire#w2
      Contact( "DB7215_PART_TYPE".PART_TYPE_U01_FIXTURES )
      Coil( "DB2440_GLOBAL_DATA".GLOBAL_DATA.ALL_UNCLAMPED_UNIT_01_ANALOG )
   END_RUNG
   RUNG wire#powerrail
      I_Contact( "DB7240_HARDWARE_SOFTWARE_ENABLE_DISABLE".DISABLE_FIXTURE.SW_UNIT_01_FIX_1_4_ENABLED )
   END_RUNG wire#w1
   RUNG wire#w1
      I_Contact( "DB7240_HARDWARE_SOFTWARE_ENABLE_DISABLE".DISABLE_FIXTURE.SW_UNIT_01_FIX_2_3_ENABLED )
   END_RUNG wire#w2
   // the same network as SCL:
   "DB2440_GLOBAL_DATA".GLOBAL_DATA.ALL_UNCLAMPED_UNIT_01_ANALOG := (("DB2500_UNIT_01_FIXTURE_1".UNCLAMPED_ANALOG AND "DB2800_UNIT_01_FIXTURE_4".UNCLAMPED_ANALOG) OR NOT "DB7240_HARDWARE_SOFTWARE_ENABLE_DISABLE".DISABLE_FIXTURE.SW_UNIT_01_FIX_1_4_ENABLED) AND (("DB2600_UNIT_01_FIXTURE_2".UNCLAMPED_ANALOG AND "DB2700_UNIT_01_FIXTURE_3".UNCLAMPED_ANALOG) OR NOT "DB7240_HARDWARE_SOFTWARE_ENABLE_DISABLE".DISABLE_FIXTURE.SW_UNIT_01_FIX_2_3_ENABLED) AND "DB7215_PART_TYPE".PART_TYPE_U01_FIXTURES;
END_REGION

REGION Network 17: CLAMPED OR UNCLAMPED UNIT 01 ANALOG
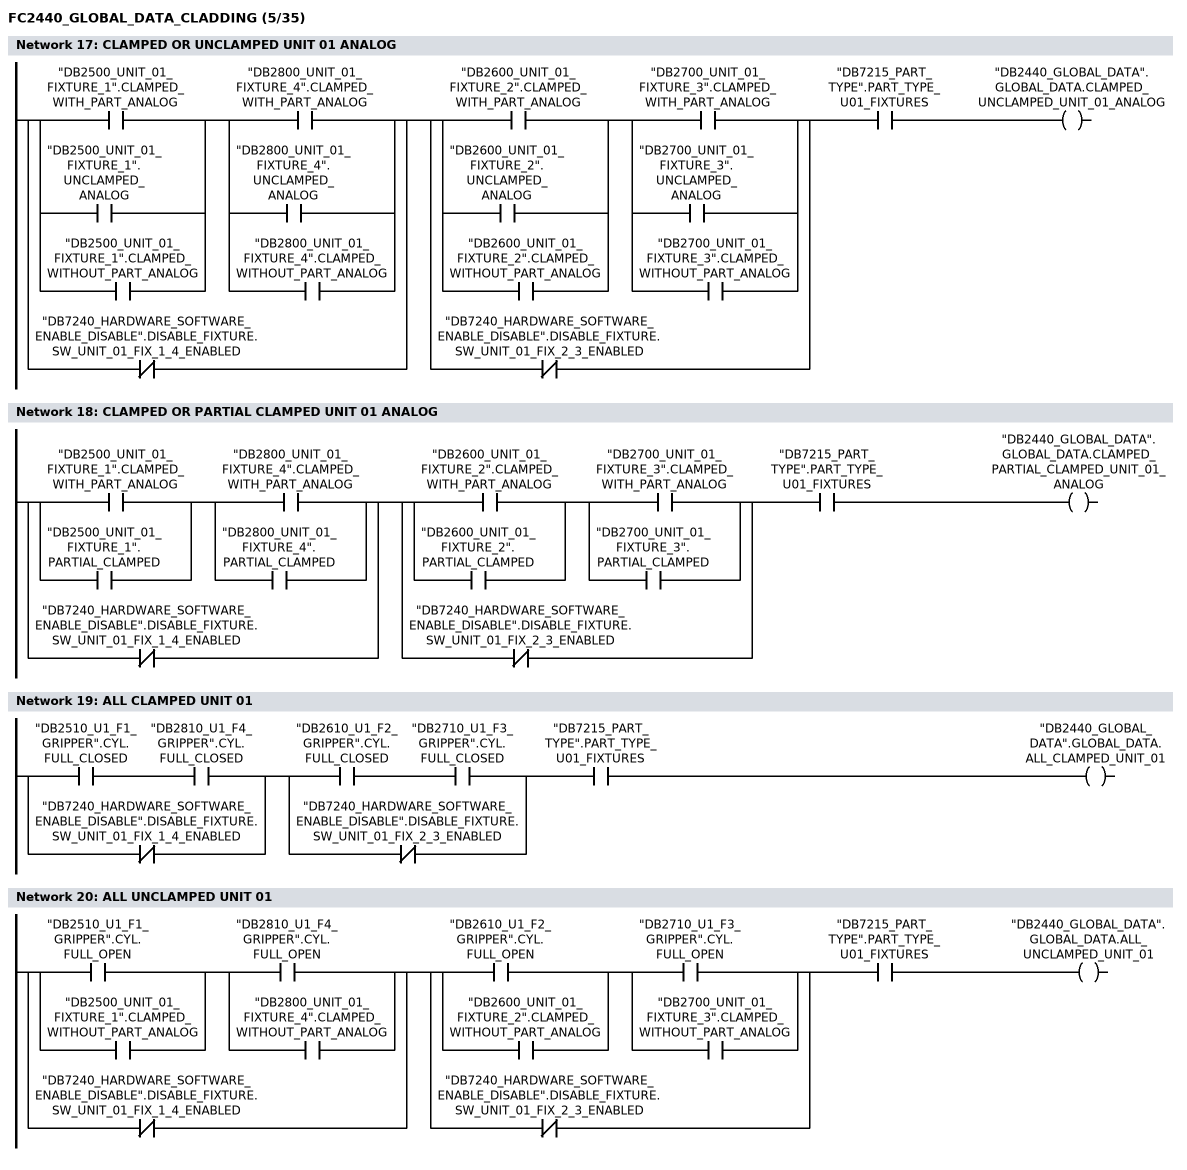
   RUNG wire#powerrail
      Contact( "DB2500_UNIT_01_FIXTURE_1".CLAMPED_WITH_PART_ANALOG )
      wire#w1
      Contact( "DB2800_UNIT_01_FIXTURE_4".CLAMPED_WITH_PART_ANALOG )
      wire#w2
      Contact( "DB2600_UNIT_01_FIXTURE_2".CLAMPED_WITH_PART_ANALOG )
      wire#w3
      Contact( "DB2700_UNIT_01_FIXTURE_3".CLAMPED_WITH_PART_ANALOG )
      wire#w4
      Contact( "DB7215_PART_TYPE".PART_TYPE_U01_FIXTURES )
      Coil( "DB2440_GLOBAL_DATA".GLOBAL_DATA.CLAMPED_UNCLAMPED_UNIT_01_ANALOG )
   END_RUNG
   RUNG wire#powerrail
      Contact( "DB2500_UNIT_01_FIXTURE_1".UNCLAMPED_ANALOG )
   END_RUNG wire#w1
   RUNG wire#powerrail
      Contact( "DB2500_UNIT_01_FIXTURE_1".CLAMPED_WITHOUT_PART_ANALOG )
   END_RUNG wire#w1
   RUNG wire#w1
      Contact( "DB2800_UNIT_01_FIXTURE_4".UNCLAMPED_ANALOG )
   END_RUNG wire#w2
   RUNG wire#w1
      Contact( "DB2800_UNIT_01_FIXTURE_4".CLAMPED_WITHOUT_PART_ANALOG )
   END_RUNG wire#w2
   RUNG wire#powerrail
      I_Contact( "DB7240_HARDWARE_SOFTWARE_ENABLE_DISABLE".DISABLE_FIXTURE.SW_UNIT_01_FIX_1_4_ENABLED )
   END_RUNG wire#w2
   RUNG wire#w2
      Contact( "DB2600_UNIT_01_FIXTURE_2".UNCLAMPED_ANALOG )
   END_RUNG wire#w3
   RUNG wire#w2
      Contact( "DB2600_UNIT_01_FIXTURE_2".CLAMPED_WITHOUT_PART_ANALOG )
   END_RUNG wire#w3
   RUNG wire#w3
      Contact( "DB2700_UNIT_01_FIXTURE_3".UNCLAMPED_ANALOG )
   END_RUNG wire#w4
   RUNG wire#w3
      Contact( "DB2700_UNIT_01_FIXTURE_3".CLAMPED_WITHOUT_PART_ANALOG )
   END_RUNG wire#w4
   RUNG wire#w2
      I_Contact( "DB7240_HARDWARE_SOFTWARE_ENABLE_DISABLE".DISABLE_FIXTURE.SW_UNIT_01_FIX_2_3_ENABLED )
   END_RUNG wire#w4
   // the same network as SCL:
   "DB2440_GLOBAL_DATA".GLOBAL_DATA.CLAMPED_UNCLAMPED_UNIT_01_ANALOG := ((("DB2500_UNIT_01_FIXTURE_1".CLAMPED_WITH_PART_ANALOG OR "DB2500_UNIT_01_FIXTURE_1".UNCLAMPED_ANALOG OR "DB2500_UNIT_01_FIXTURE_1".CLAMPED_WITHOUT_PART_ANALOG) AND ("DB2800_UNIT_01_FIXTURE_4".CLAMPED_WITH_PART_ANALOG OR "DB2800_UNIT_01_FIXTURE_4".UNCLAMPED_ANALOG OR "DB2800_UNIT_01_FIXTURE_4".CLAMPED_WITHOUT_PART_ANALOG)) OR NOT "DB7240_HARDWARE_SOFTWARE_ENABLE_DISABLE".DISABLE_FIXTURE.SW_UNIT_01_FIX_1_4_ENABLED) AND ((("DB2600_UNIT_01_FIXTURE_2".CLAMPED_WITH_PART_ANALOG OR "DB2600_UNIT_01_FIXTURE_2".UNCLAMPED_ANALOG OR "DB2600_UNIT_01_FIXTURE_2".CLAMPED_WITHOUT_PART_ANALOG) AND ("DB2700_UNIT_01_FIXTURE_3".CLAMPED_WITH_PART_ANALOG OR "DB2700_UNIT_01_FIXTURE_3".UNCLAMPED_ANALOG OR "DB2700_UNIT_01_FIXTURE_3".CLAMPED_WITHOUT_PART_ANALOG)) OR NOT "DB7240_HARDWARE_SOFTWARE_ENABLE_DISABLE".DISABLE_FIXTURE.SW_UNIT_01_FIX_2_3_ENABLED) AND "DB7215_PART_TYPE".PART_TYPE_U01_FIXTURES;
END_REGION

REGION Network 18: CLAMPED OR PARTIAL CLAMPED UNIT 01 ANALOG
   RUNG wire#powerrail
      Contact( "DB2500_UNIT_01_FIXTURE_1".CLAMPED_WITH_PART_ANALOG )
      wire#w1
      Contact( "DB2800_UNIT_01_FIXTURE_4".CLAMPED_WITH_PART_ANALOG )
      wire#w2
      Contact( "DB2600_UNIT_01_FIXTURE_2".CLAMPED_WITH_PART_ANALOG )
      wire#w3
      Contact( "DB2700_UNIT_01_FIXTURE_3".CLAMPED_WITH_PART_ANALOG )
      wire#w4
      Contact( "DB7215_PART_TYPE".PART_TYPE_U01_FIXTURES )
      Coil( "DB2440_GLOBAL_DATA".GLOBAL_DATA.CLAMPED_PARTIAL_CLAMPED_UNIT_01_ANALOG )
   END_RUNG
   RUNG wire#powerrail
      Contact( "DB2500_UNIT_01_FIXTURE_1".PARTIAL_CLAMPED )
   END_RUNG wire#w1
   RUNG wire#w1
      Contact( "DB2800_UNIT_01_FIXTURE_4".PARTIAL_CLAMPED )
   END_RUNG wire#w2
   RUNG wire#powerrail
      I_Contact( "DB7240_HARDWARE_SOFTWARE_ENABLE_DISABLE".DISABLE_FIXTURE.SW_UNIT_01_FIX_1_4_ENABLED )
   END_RUNG wire#w2
   RUNG wire#w2
      Contact( "DB2600_UNIT_01_FIXTURE_2".PARTIAL_CLAMPED )
   END_RUNG wire#w3
   RUNG wire#w3
      Contact( "DB2700_UNIT_01_FIXTURE_3".PARTIAL_CLAMPED )
   END_RUNG wire#w4
   RUNG wire#w2
      I_Contact( "DB7240_HARDWARE_SOFTWARE_ENABLE_DISABLE".DISABLE_FIXTURE.SW_UNIT_01_FIX_2_3_ENABLED )
   END_RUNG wire#w4
   // the same network as SCL:
   "DB2440_GLOBAL_DATA".GLOBAL_DATA.CLAMPED_PARTIAL_CLAMPED_UNIT_01_ANALOG := ((("DB2500_UNIT_01_FIXTURE_1".CLAMPED_WITH_PART_ANALOG OR "DB2500_UNIT_01_FIXTURE_1".PARTIAL_CLAMPED) AND ("DB2800_UNIT_01_FIXTURE_4".CLAMPED_WITH_PART_ANALOG OR "DB2800_UNIT_01_FIXTURE_4".PARTIAL_CLAMPED)) OR NOT "DB7240_HARDWARE_SOFTWARE_ENABLE_DISABLE".DISABLE_FIXTURE.SW_UNIT_01_FIX_1_4_ENABLED) AND ((("DB2600_UNIT_01_FIXTURE_2".CLAMPED_WITH_PART_ANALOG OR "DB2600_UNIT_01_FIXTURE_2".PARTIAL_CLAMPED) AND ("DB2700_UNIT_01_FIXTURE_3".CLAMPED_WITH_PART_ANALOG OR "DB2700_UNIT_01_FIXTURE_3".PARTIAL_CLAMPED)) OR NOT "DB7240_HARDWARE_SOFTWARE_ENABLE_DISABLE".DISABLE_FIXTURE.SW_UNIT_01_FIX_2_3_ENABLED) AND "DB7215_PART_TYPE".PART_TYPE_U01_FIXTURES;
END_REGION

REGION Network 19: ALL CLAMPED UNIT 01
   RUNG wire#powerrail
      Contact( "DB2510_U1_F1_GRIPPER".CYL.FULL_CLOSED )
      Contact( "DB2810_U1_F4_GRIPPER".CYL.FULL_CLOSED )
      wire#w1
      Contact( "DB2610_U1_F2_GRIPPER".CYL.FULL_CLOSED )
      Contact( "DB2710_U1_F3_GRIPPER".CYL.FULL_CLOSED )
      wire#w2
      Contact( "DB7215_PART_TYPE".PART_TYPE_U01_FIXTURES )
      Coil( "DB2440_GLOBAL_DATA".GLOBAL_DATA.ALL_CLAMPED_UNIT_01 )
   END_RUNG
   RUNG wire#powerrail
      I_Contact( "DB7240_HARDWARE_SOFTWARE_ENABLE_DISABLE".DISABLE_FIXTURE.SW_UNIT_01_FIX_1_4_ENABLED )
   END_RUNG wire#w1
   RUNG wire#w1
      I_Contact( "DB7240_HARDWARE_SOFTWARE_ENABLE_DISABLE".DISABLE_FIXTURE.SW_UNIT_01_FIX_2_3_ENABLED )
   END_RUNG wire#w2
   // the same network as SCL:
   "DB2440_GLOBAL_DATA".GLOBAL_DATA.ALL_CLAMPED_UNIT_01 := (("DB2510_U1_F1_GRIPPER".CYL.FULL_CLOSED AND "DB2810_U1_F4_GRIPPER".CYL.FULL_CLOSED) OR NOT "DB7240_HARDWARE_SOFTWARE_ENABLE_DISABLE".DISABLE_FIXTURE.SW_UNIT_01_FIX_1_4_ENABLED) AND (("DB2610_U1_F2_GRIPPER".CYL.FULL_CLOSED AND "DB2710_U1_F3_GRIPPER".CYL.FULL_CLOSED) OR NOT "DB7240_HARDWARE_SOFTWARE_ENABLE_DISABLE".DISABLE_FIXTURE.SW_UNIT_01_FIX_2_3_ENABLED) AND "DB7215_PART_TYPE".PART_TYPE_U01_FIXTURES;
END_REGION

REGION Network 20: ALL UNCLAMPED UNIT 01
   RUNG wire#powerrail
      Contact( "DB2510_U1_F1_GRIPPER".CYL.FULL_OPEN )
      wire#w1
      Contact( "DB2810_U1_F4_GRIPPER".CYL.FULL_OPEN )
      wire#w2
      Contact( "DB2610_U1_F2_GRIPPER".CYL.FULL_OPEN )
      wire#w3
      Contact( "DB2710_U1_F3_GRIPPER".CYL.FULL_OPEN )
      wire#w4
      Contact( "DB7215_PART_TYPE".PART_TYPE_U01_FIXTURES )
      Coil( "DB2440_GLOBAL_DATA".GLOBAL_DATA.ALL_UNCLAMPED_UNIT_01 )
   END_RUNG
   RUNG wire#powerrail
      Contact( "DB2500_UNIT_01_FIXTURE_1".CLAMPED_WITHOUT_PART_ANALOG )
   END_RUNG wire#w1
   RUNG wire#w1
      Contact( "DB2800_UNIT_01_FIXTURE_4".CLAMPED_WITHOUT_PART_ANALOG )
   END_RUNG wire#w2
   RUNG wire#powerrail
      I_Contact( "DB7240_HARDWARE_SOFTWARE_ENABLE_DISABLE".DISABLE_FIXTURE.SW_UNIT_01_FIX_1_4_ENABLED )
   END_RUNG wire#w2
   RUNG wire#w2
      Contact( "DB2600_UNIT_01_FIXTURE_2".CLAMPED_WITHOUT_PART_ANALOG )
   END_RUNG wire#w3
   RUNG wire#w3
      Contact( "DB2700_UNIT_01_FIXTURE_3".CLAMPED_WITHOUT_PART_ANALOG )
   END_RUNG wire#w4
   RUNG wire#w2
      I_Contact( "DB7240_HARDWARE_SOFTWARE_ENABLE_DISABLE".DISABLE_FIXTURE.SW_UNIT_01_FIX_2_3_ENABLED )
   END_RUNG wire#w4
   // the same network as SCL:
   "DB2440_GLOBAL_DATA".GLOBAL_DATA.ALL_UNCLAMPED_UNIT_01 := ((("DB2510_U1_F1_GRIPPER".CYL.FULL_OPEN OR "DB2500_UNIT_01_FIXTURE_1".CLAMPED_WITHOUT_PART_ANALOG) AND ("DB2810_U1_F4_GRIPPER".CYL.FULL_OPEN OR "DB2800_UNIT_01_FIXTURE_4".CLAMPED_WITHOUT_PART_ANALOG)) OR NOT "DB7240_HARDWARE_SOFTWARE_ENABLE_DISABLE".DISABLE_FIXTURE.SW_UNIT_01_FIX_1_4_ENABLED) AND ((("DB2610_U1_F2_GRIPPER".CYL.FULL_OPEN OR "DB2600_UNIT_01_FIXTURE_2".CLAMPED_WITHOUT_PART_ANALOG) AND ("DB2710_U1_F3_GRIPPER".CYL.FULL_OPEN OR "DB2700_UNIT_01_FIXTURE_3".CLAMPED_WITHOUT_PART_ANALOG)) OR NOT "DB7240_HARDWARE_SOFTWARE_ENABLE_DISABLE".DISABLE_FIXTURE.SW_UNIT_01_FIX_2_3_ENABLED) AND "DB7215_PART_TYPE".PART_TYPE_U01_FIXTURES;
END_REGION

REGION Network 21: CLAMPED OR UNCLAMPED UNIT 01
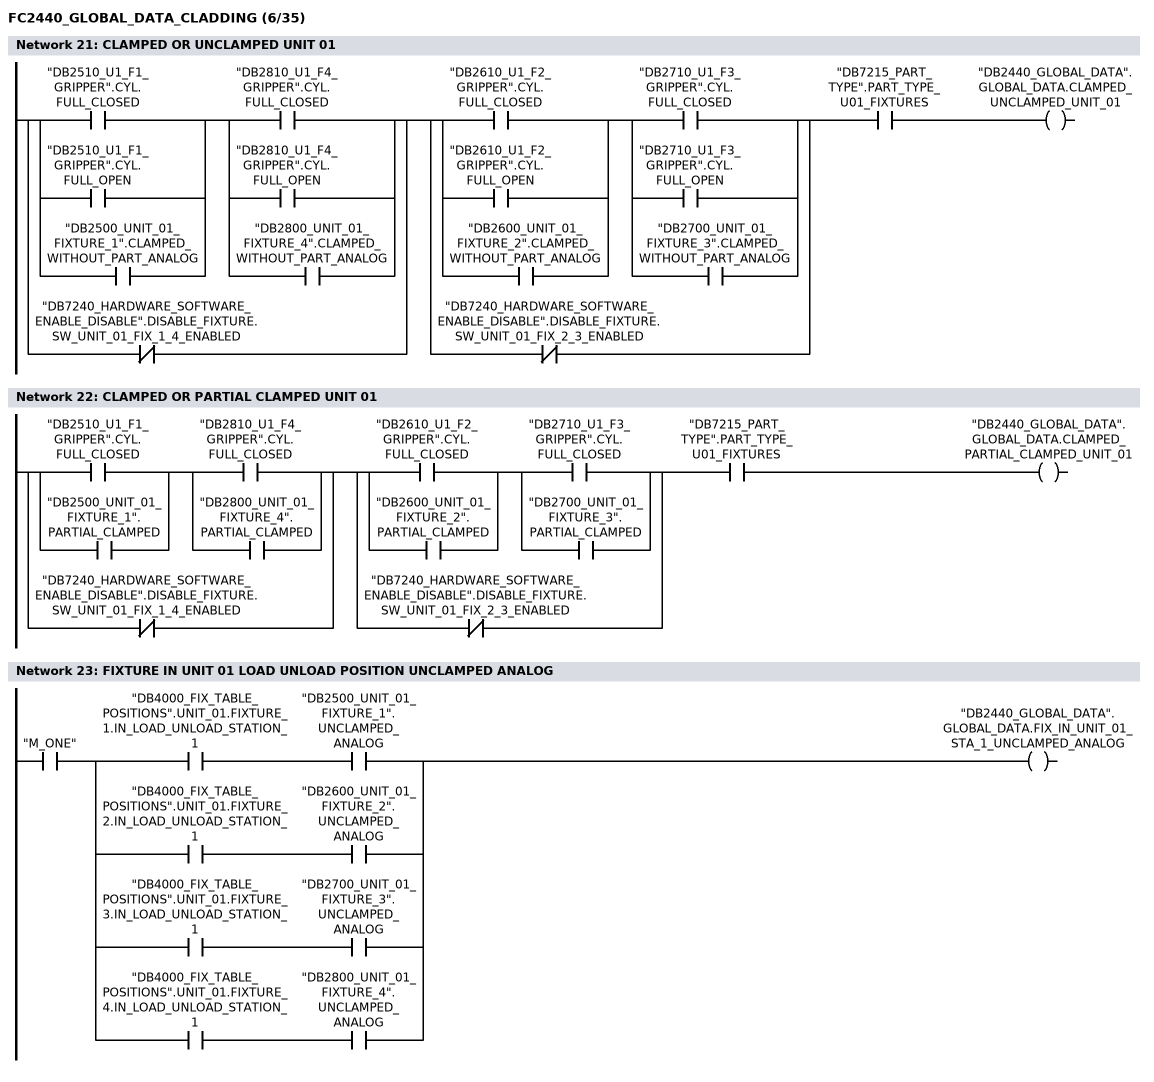
   RUNG wire#powerrail
      Contact( "DB2510_U1_F1_GRIPPER".CYL.FULL_CLOSED )
      wire#w1
      Contact( "DB2810_U1_F4_GRIPPER".CYL.FULL_CLOSED )
      wire#w2
      Contact( "DB2610_U1_F2_GRIPPER".CYL.FULL_CLOSED )
      wire#w3
      Contact( "DB2710_U1_F3_GRIPPER".CYL.FULL_CLOSED )
      wire#w4
      Contact( "DB7215_PART_TYPE".PART_TYPE_U01_FIXTURES )
      Coil( "DB2440_GLOBAL_DATA".GLOBAL_DATA.CLAMPED_UNCLAMPED_UNIT_01 )
   END_RUNG
   RUNG wire#powerrail
      Contact( "DB2510_U1_F1_GRIPPER".CYL.FULL_OPEN )
   END_RUNG wire#w1
   RUNG wire#powerrail
      Contact( "DB2500_UNIT_01_FIXTURE_1".CLAMPED_WITHOUT_PART_ANALOG )
   END_RUNG wire#w1
   RUNG wire#w1
      Contact( "DB2810_U1_F4_GRIPPER".CYL.FULL_OPEN )
   END_RUNG wire#w2
   RUNG wire#w1
      Contact( "DB2800_UNIT_01_FIXTURE_4".CLAMPED_WITHOUT_PART_ANALOG )
   END_RUNG wire#w2
   RUNG wire#powerrail
      I_Contact( "DB7240_HARDWARE_SOFTWARE_ENABLE_DISABLE".DISABLE_FIXTURE.SW_UNIT_01_FIX_1_4_ENABLED )
   END_RUNG wire#w2
   RUNG wire#w2
      Contact( "DB2610_U1_F2_GRIPPER".CYL.FULL_OPEN )
   END_RUNG wire#w3
   RUNG wire#w2
      Contact( "DB2600_UNIT_01_FIXTURE_2".CLAMPED_WITHOUT_PART_ANALOG )
   END_RUNG wire#w3
   RUNG wire#w3
      Contact( "DB2710_U1_F3_GRIPPER".CYL.FULL_OPEN )
   END_RUNG wire#w4
   RUNG wire#w3
      Contact( "DB2700_UNIT_01_FIXTURE_3".CLAMPED_WITHOUT_PART_ANALOG )
   END_RUNG wire#w4
   RUNG wire#w2
      I_Contact( "DB7240_HARDWARE_SOFTWARE_ENABLE_DISABLE".DISABLE_FIXTURE.SW_UNIT_01_FIX_2_3_ENABLED )
   END_RUNG wire#w4
   // the same network as SCL:
   "DB2440_GLOBAL_DATA".GLOBAL_DATA.CLAMPED_UNCLAMPED_UNIT_01 := ((("DB2510_U1_F1_GRIPPER".CYL.FULL_CLOSED OR "DB2510_U1_F1_GRIPPER".CYL.FULL_OPEN OR "DB2500_UNIT_01_FIXTURE_1".CLAMPED_WITHOUT_PART_ANALOG) AND ("DB2810_U1_F4_GRIPPER".CYL.FULL_CLOSED OR "DB2810_U1_F4_GRIPPER".CYL.FULL_OPEN OR "DB2800_UNIT_01_FIXTURE_4".CLAMPED_WITHOUT_PART_ANALOG)) OR NOT "DB7240_HARDWARE_SOFTWARE_ENABLE_DISABLE".DISABLE_FIXTURE.SW_UNIT_01_FIX_1_4_ENABLED) AND ((("DB2610_U1_F2_GRIPPER".CYL.FULL_CLOSED OR "DB2610_U1_F2_GRIPPER".CYL.FULL_OPEN OR "DB2600_UNIT_01_FIXTURE_2".CLAMPED_WITHOUT_PART_ANALOG) AND ("DB2710_U1_F3_GRIPPER".CYL.FULL_CLOSED OR "DB2710_U1_F3_GRIPPER".CYL.FULL_OPEN OR "DB2700_UNIT_01_FIXTURE_3".CLAMPED_WITHOUT_PART_ANALOG)) OR NOT "DB7240_HARDWARE_SOFTWARE_ENABLE_DISABLE".DISABLE_FIXTURE.SW_UNIT_01_FIX_2_3_ENABLED) AND "DB7215_PART_TYPE".PART_TYPE_U01_FIXTURES;
END_REGION

REGION Network 22: CLAMPED OR PARTIAL CLAMPED UNIT 01
   RUNG wire#powerrail
      Contact( "DB2510_U1_F1_GRIPPER".CYL.FULL_CLOSED )
      wire#w1
      Contact( "DB2810_U1_F4_GRIPPER".CYL.FULL_CLOSED )
      wire#w2
      Contact( "DB2610_U1_F2_GRIPPER".CYL.FULL_CLOSED )
      wire#w3
      Contact( "DB2710_U1_F3_GRIPPER".CYL.FULL_CLOSED )
      wire#w4
      Contact( "DB7215_PART_TYPE".PART_TYPE_U01_FIXTURES )
      Coil( "DB2440_GLOBAL_DATA".GLOBAL_DATA.CLAMPED_PARTIAL_CLAMPED_UNIT_01 )
   END_RUNG
   RUNG wire#powerrail
      Contact( "DB2500_UNIT_01_FIXTURE_1".PARTIAL_CLAMPED )
   END_RUNG wire#w1
   RUNG wire#w1
      Contact( "DB2800_UNIT_01_FIXTURE_4".PARTIAL_CLAMPED )
   END_RUNG wire#w2
   RUNG wire#powerrail
      I_Contact( "DB7240_HARDWARE_SOFTWARE_ENABLE_DISABLE".DISABLE_FIXTURE.SW_UNIT_01_FIX_1_4_ENABLED )
   END_RUNG wire#w2
   RUNG wire#w2
      Contact( "DB2600_UNIT_01_FIXTURE_2".PARTIAL_CLAMPED )
   END_RUNG wire#w3
   RUNG wire#w3
      Contact( "DB2700_UNIT_01_FIXTURE_3".PARTIAL_CLAMPED )
   END_RUNG wire#w4
   RUNG wire#w2
      I_Contact( "DB7240_HARDWARE_SOFTWARE_ENABLE_DISABLE".DISABLE_FIXTURE.SW_UNIT_01_FIX_2_3_ENABLED )
   END_RUNG wire#w4
   // the same network as SCL:
   "DB2440_GLOBAL_DATA".GLOBAL_DATA.CLAMPED_PARTIAL_CLAMPED_UNIT_01 := ((("DB2510_U1_F1_GRIPPER".CYL.FULL_CLOSED OR "DB2500_UNIT_01_FIXTURE_1".PARTIAL_CLAMPED) AND ("DB2810_U1_F4_GRIPPER".CYL.FULL_CLOSED OR "DB2800_UNIT_01_FIXTURE_4".PARTIAL_CLAMPED)) OR NOT "DB7240_HARDWARE_SOFTWARE_ENABLE_DISABLE".DISABLE_FIXTURE.SW_UNIT_01_FIX_1_4_ENABLED) AND ((("DB2610_U1_F2_GRIPPER".CYL.FULL_CLOSED OR "DB2600_UNIT_01_FIXTURE_2".PARTIAL_CLAMPED) AND ("DB2710_U1_F3_GRIPPER".CYL.FULL_CLOSED OR "DB2700_UNIT_01_FIXTURE_3".PARTIAL_CLAMPED)) OR NOT "DB7240_HARDWARE_SOFTWARE_ENABLE_DISABLE".DISABLE_FIXTURE.SW_UNIT_01_FIX_2_3_ENABLED) AND "DB7215_PART_TYPE".PART_TYPE_U01_FIXTURES;
END_REGION

REGION Network 23: FIXTURE IN UNIT 01 LOAD UNLOAD POSITION UNCLAMPED ANALOG
   RUNG wire#powerrail
      Contact( "M_ONE" )
      wire#w1
      Contact( "DB4000_FIX_TABLE_POSITIONS".UNIT_01.FIXTURE_1.IN_LOAD_UNLOAD_STATION_1 )
      Contact( "DB2500_UNIT_01_FIXTURE_1".UNCLAMPED_ANALOG )
      wire#w2
      Coil( "DB2440_GLOBAL_DATA".GLOBAL_DATA.FIX_IN_UNIT_01_STA_1_UNCLAMPED_ANALOG )
   END_RUNG
   RUNG wire#w1
      Contact( "DB4000_FIX_TABLE_POSITIONS".UNIT_01.FIXTURE_2.IN_LOAD_UNLOAD_STATION_1 )
      Contact( "DB2600_UNIT_01_FIXTURE_2".UNCLAMPED_ANALOG )
   END_RUNG wire#w2
   RUNG wire#w1
      Contact( "DB4000_FIX_TABLE_POSITIONS".UNIT_01.FIXTURE_3.IN_LOAD_UNLOAD_STATION_1 )
      Contact( "DB2700_UNIT_01_FIXTURE_3".UNCLAMPED_ANALOG )
   END_RUNG wire#w2
   RUNG wire#w1
      Contact( "DB4000_FIX_TABLE_POSITIONS".UNIT_01.FIXTURE_4.IN_LOAD_UNLOAD_STATION_1 )
      Contact( "DB2800_UNIT_01_FIXTURE_4".UNCLAMPED_ANALOG )
   END_RUNG wire#w2
   // the same network as SCL:
   "DB2440_GLOBAL_DATA".GLOBAL_DATA.FIX_IN_UNIT_01_STA_1_UNCLAMPED_ANALOG := "M_ONE" AND (("DB4000_FIX_TABLE_POSITIONS".UNIT_01.FIXTURE_1.IN_LOAD_UNLOAD_STATION_1 AND "DB2500_UNIT_01_FIXTURE_1".UNCLAMPED_ANALOG) OR ("DB4000_FIX_TABLE_POSITIONS".UNIT_01.FIXTURE_2.IN_LOAD_UNLOAD_STATION_1 AND "DB2600_UNIT_01_FIXTURE_2".UNCLAMPED_ANALOG) OR ("DB4000_FIX_TABLE_POSITIONS".UNIT_01.FIXTURE_3.IN_LOAD_UNLOAD_STATION_1 AND "DB2700_UNIT_01_FIXTURE_3".UNCLAMPED_ANALOG) OR ("DB4000_FIX_TABLE_POSITIONS".UNIT_01.FIXTURE_4.IN_LOAD_UNLOAD_STATION_1 AND "DB2800_UNIT_01_FIXTURE_4".UNCLAMPED_ANALOG));
END_REGION

REGION Network 24: FIXTURE IN UNIT 01 LOAD UNLOAD POSITION CLAMPED ANALOG
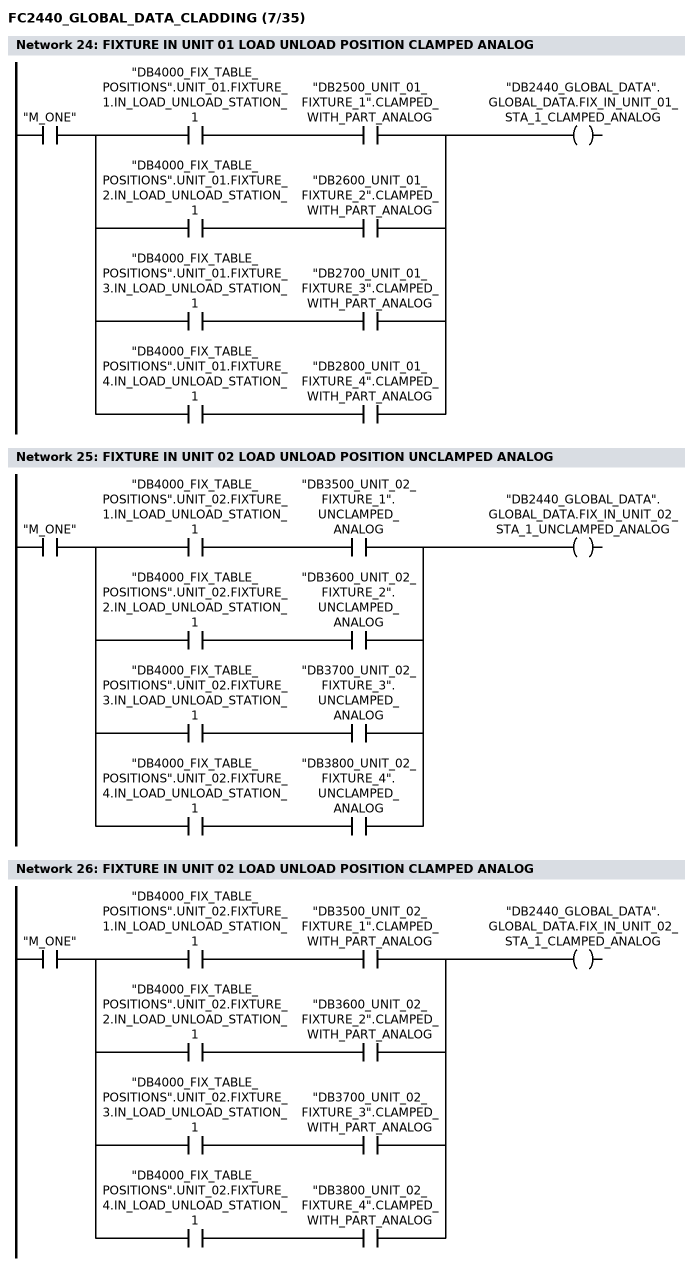
   RUNG wire#powerrail
      Contact( "M_ONE" )
      wire#w1
      Contact( "DB4000_FIX_TABLE_POSITIONS".UNIT_01.FIXTURE_1.IN_LOAD_UNLOAD_STATION_1 )
      Contact( "DB2500_UNIT_01_FIXTURE_1".CLAMPED_WITH_PART_ANALOG )
      wire#w2
      Coil( "DB2440_GLOBAL_DATA".GLOBAL_DATA.FIX_IN_UNIT_01_STA_1_CLAMPED_ANALOG )
   END_RUNG
   RUNG wire#w1
      Contact( "DB4000_FIX_TABLE_POSITIONS".UNIT_01.FIXTURE_2.IN_LOAD_UNLOAD_STATION_1 )
      Contact( "DB2600_UNIT_01_FIXTURE_2".CLAMPED_WITH_PART_ANALOG )
   END_RUNG wire#w2
   RUNG wire#w1
      Contact( "DB4000_FIX_TABLE_POSITIONS".UNIT_01.FIXTURE_3.IN_LOAD_UNLOAD_STATION_1 )
      Contact( "DB2700_UNIT_01_FIXTURE_3".CLAMPED_WITH_PART_ANALOG )
   END_RUNG wire#w2
   RUNG wire#w1
      Contact( "DB4000_FIX_TABLE_POSITIONS".UNIT_01.FIXTURE_4.IN_LOAD_UNLOAD_STATION_1 )
      Contact( "DB2800_UNIT_01_FIXTURE_4".CLAMPED_WITH_PART_ANALOG )
   END_RUNG wire#w2
   // the same network as SCL:
   "DB2440_GLOBAL_DATA".GLOBAL_DATA.FIX_IN_UNIT_01_STA_1_CLAMPED_ANALOG := "M_ONE" AND (("DB4000_FIX_TABLE_POSITIONS".UNIT_01.FIXTURE_1.IN_LOAD_UNLOAD_STATION_1 AND "DB2500_UNIT_01_FIXTURE_1".CLAMPED_WITH_PART_ANALOG) OR ("DB4000_FIX_TABLE_POSITIONS".UNIT_01.FIXTURE_2.IN_LOAD_UNLOAD_STATION_1 AND "DB2600_UNIT_01_FIXTURE_2".CLAMPED_WITH_PART_ANALOG) OR ("DB4000_FIX_TABLE_POSITIONS".UNIT_01.FIXTURE_3.IN_LOAD_UNLOAD_STATION_1 AND "DB2700_UNIT_01_FIXTURE_3".CLAMPED_WITH_PART_ANALOG) OR ("DB4000_FIX_TABLE_POSITIONS".UNIT_01.FIXTURE_4.IN_LOAD_UNLOAD_STATION_1 AND "DB2800_UNIT_01_FIXTURE_4".CLAMPED_WITH_PART_ANALOG));
END_REGION

REGION Network 25: FIXTURE IN UNIT 02 LOAD UNLOAD POSITION UNCLAMPED ANALOG
   RUNG wire#powerrail
      Contact( "M_ONE" )
      wire#w1
      Contact( "DB4000_FIX_TABLE_POSITIONS".UNIT_02.FIXTURE_1.IN_LOAD_UNLOAD_STATION_1 )
      Contact( "DB3500_UNIT_02_FIXTURE_1".UNCLAMPED_ANALOG )
      wire#w2
      Coil( "DB2440_GLOBAL_DATA".GLOBAL_DATA.FIX_IN_UNIT_02_STA_1_UNCLAMPED_ANALOG )
   END_RUNG
   RUNG wire#w1
      Contact( "DB4000_FIX_TABLE_POSITIONS".UNIT_02.FIXTURE_2.IN_LOAD_UNLOAD_STATION_1 )
      Contact( "DB3600_UNIT_02_FIXTURE_2".UNCLAMPED_ANALOG )
   END_RUNG wire#w2
   RUNG wire#w1
      Contact( "DB4000_FIX_TABLE_POSITIONS".UNIT_02.FIXTURE_3.IN_LOAD_UNLOAD_STATION_1 )
      Contact( "DB3700_UNIT_02_FIXTURE_3".UNCLAMPED_ANALOG )
   END_RUNG wire#w2
   RUNG wire#w1
      Contact( "DB4000_FIX_TABLE_POSITIONS".UNIT_02.FIXTURE_4.IN_LOAD_UNLOAD_STATION_1 )
      Contact( "DB3800_UNIT_02_FIXTURE_4".UNCLAMPED_ANALOG )
   END_RUNG wire#w2
   // the same network as SCL:
   "DB2440_GLOBAL_DATA".GLOBAL_DATA.FIX_IN_UNIT_02_STA_1_UNCLAMPED_ANALOG := "M_ONE" AND (("DB4000_FIX_TABLE_POSITIONS".UNIT_02.FIXTURE_1.IN_LOAD_UNLOAD_STATION_1 AND "DB3500_UNIT_02_FIXTURE_1".UNCLAMPED_ANALOG) OR ("DB4000_FIX_TABLE_POSITIONS".UNIT_02.FIXTURE_2.IN_LOAD_UNLOAD_STATION_1 AND "DB3600_UNIT_02_FIXTURE_2".UNCLAMPED_ANALOG) OR ("DB4000_FIX_TABLE_POSITIONS".UNIT_02.FIXTURE_3.IN_LOAD_UNLOAD_STATION_1 AND "DB3700_UNIT_02_FIXTURE_3".UNCLAMPED_ANALOG) OR ("DB4000_FIX_TABLE_POSITIONS".UNIT_02.FIXTURE_4.IN_LOAD_UNLOAD_STATION_1 AND "DB3800_UNIT_02_FIXTURE_4".UNCLAMPED_ANALOG));
END_REGION

REGION Network 26: FIXTURE IN UNIT 02 LOAD UNLOAD POSITION CLAMPED ANALOG
   RUNG wire#powerrail
      Contact( "M_ONE" )
      wire#w1
      Contact( "DB4000_FIX_TABLE_POSITIONS".UNIT_02.FIXTURE_1.IN_LOAD_UNLOAD_STATION_1 )
      Contact( "DB3500_UNIT_02_FIXTURE_1".CLAMPED_WITH_PART_ANALOG )
      wire#w2
      Coil( "DB2440_GLOBAL_DATA".GLOBAL_DATA.FIX_IN_UNIT_02_STA_1_CLAMPED_ANALOG )
   END_RUNG
   RUNG wire#w1
      Contact( "DB4000_FIX_TABLE_POSITIONS".UNIT_02.FIXTURE_2.IN_LOAD_UNLOAD_STATION_1 )
      Contact( "DB3600_UNIT_02_FIXTURE_2".CLAMPED_WITH_PART_ANALOG )
   END_RUNG wire#w2
   RUNG wire#w1
      Contact( "DB4000_FIX_TABLE_POSITIONS".UNIT_02.FIXTURE_3.IN_LOAD_UNLOAD_STATION_1 )
      Contact( "DB3700_UNIT_02_FIXTURE_3".CLAMPED_WITH_PART_ANALOG )
   END_RUNG wire#w2
   RUNG wire#w1
      Contact( "DB4000_FIX_TABLE_POSITIONS".UNIT_02.FIXTURE_4.IN_LOAD_UNLOAD_STATION_1 )
      Contact( "DB3800_UNIT_02_FIXTURE_4".CLAMPED_WITH_PART_ANALOG )
   END_RUNG wire#w2
   // the same network as SCL:
   "DB2440_GLOBAL_DATA".GLOBAL_DATA.FIX_IN_UNIT_02_STA_1_CLAMPED_ANALOG := "M_ONE" AND (("DB4000_FIX_TABLE_POSITIONS".UNIT_02.FIXTURE_1.IN_LOAD_UNLOAD_STATION_1 AND "DB3500_UNIT_02_FIXTURE_1".CLAMPED_WITH_PART_ANALOG) OR ("DB4000_FIX_TABLE_POSITIONS".UNIT_02.FIXTURE_2.IN_LOAD_UNLOAD_STATION_1 AND "DB3600_UNIT_02_FIXTURE_2".CLAMPED_WITH_PART_ANALOG) OR ("DB4000_FIX_TABLE_POSITIONS".UNIT_02.FIXTURE_3.IN_LOAD_UNLOAD_STATION_1 AND "DB3700_UNIT_02_FIXTURE_3".CLAMPED_WITH_PART_ANALOG) OR ("DB4000_FIX_TABLE_POSITIONS".UNIT_02.FIXTURE_4.IN_LOAD_UNLOAD_STATION_1 AND "DB3800_UNIT_02_FIXTURE_4".CLAMPED_WITH_PART_ANALOG));
END_REGION

REGION Network 27: FIXTURE IN UNIT 01 SPARE POSITION UNCLAMPED ANALOG
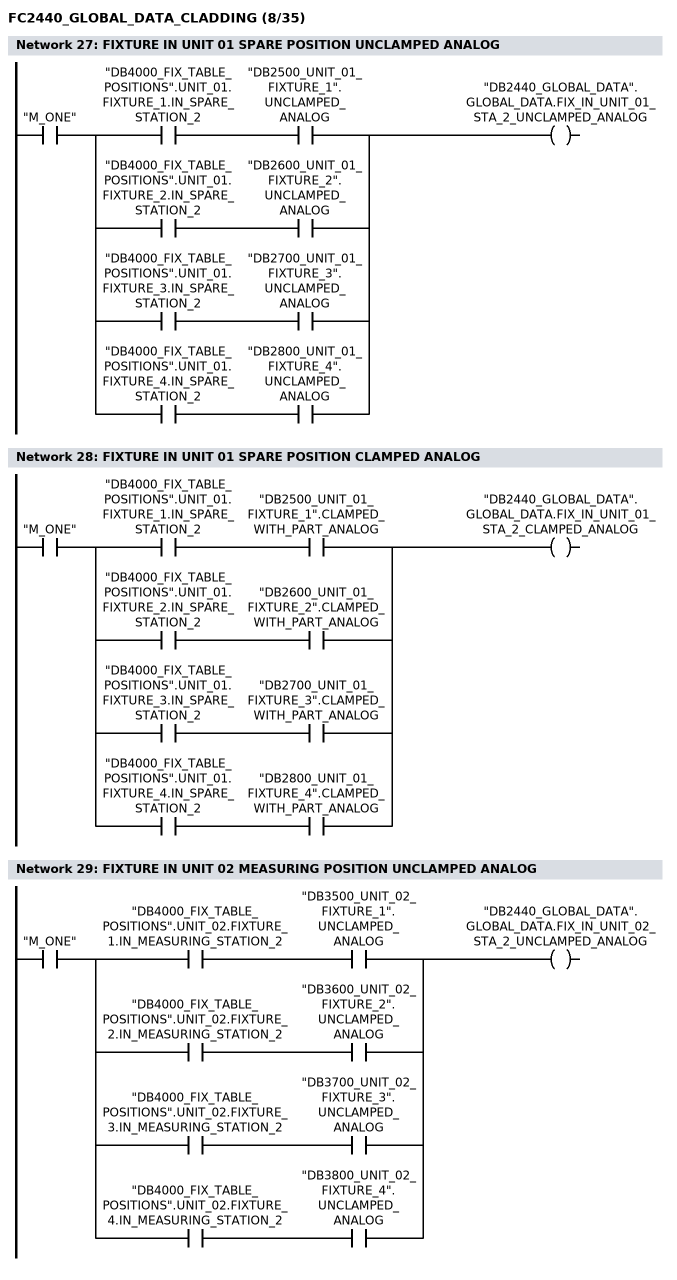
   RUNG wire#powerrail
      Contact( "M_ONE" )
      wire#w1
      Contact( "DB4000_FIX_TABLE_POSITIONS".UNIT_01.FIXTURE_1.IN_SPARE_STATION_2 )
      Contact( "DB2500_UNIT_01_FIXTURE_1".UNCLAMPED_ANALOG )
      wire#w2
      Coil( "DB2440_GLOBAL_DATA".GLOBAL_DATA.FIX_IN_UNIT_01_STA_2_UNCLAMPED_ANALOG )
   END_RUNG
   RUNG wire#w1
      Contact( "DB4000_FIX_TABLE_POSITIONS".UNIT_01.FIXTURE_2.IN_SPARE_STATION_2 )
      Contact( "DB2600_UNIT_01_FIXTURE_2".UNCLAMPED_ANALOG )
   END_RUNG wire#w2
   RUNG wire#w1
      Contact( "DB4000_FIX_TABLE_POSITIONS".UNIT_01.FIXTURE_3.IN_SPARE_STATION_2 )
      Contact( "DB2700_UNIT_01_FIXTURE_3".UNCLAMPED_ANALOG )
   END_RUNG wire#w2
   RUNG wire#w1
      Contact( "DB4000_FIX_TABLE_POSITIONS".UNIT_01.FIXTURE_4.IN_SPARE_STATION_2 )
      Contact( "DB2800_UNIT_01_FIXTURE_4".UNCLAMPED_ANALOG )
   END_RUNG wire#w2
   // the same network as SCL:
   "DB2440_GLOBAL_DATA".GLOBAL_DATA.FIX_IN_UNIT_01_STA_2_UNCLAMPED_ANALOG := "M_ONE" AND (("DB4000_FIX_TABLE_POSITIONS".UNIT_01.FIXTURE_1.IN_SPARE_STATION_2 AND "DB2500_UNIT_01_FIXTURE_1".UNCLAMPED_ANALOG) OR ("DB4000_FIX_TABLE_POSITIONS".UNIT_01.FIXTURE_2.IN_SPARE_STATION_2 AND "DB2600_UNIT_01_FIXTURE_2".UNCLAMPED_ANALOG) OR ("DB4000_FIX_TABLE_POSITIONS".UNIT_01.FIXTURE_3.IN_SPARE_STATION_2 AND "DB2700_UNIT_01_FIXTURE_3".UNCLAMPED_ANALOG) OR ("DB4000_FIX_TABLE_POSITIONS".UNIT_01.FIXTURE_4.IN_SPARE_STATION_2 AND "DB2800_UNIT_01_FIXTURE_4".UNCLAMPED_ANALOG));
END_REGION

REGION Network 28: FIXTURE IN UNIT 01 SPARE POSITION CLAMPED ANALOG
   RUNG wire#powerrail
      Contact( "M_ONE" )
      wire#w1
      Contact( "DB4000_FIX_TABLE_POSITIONS".UNIT_01.FIXTURE_1.IN_SPARE_STATION_2 )
      Contact( "DB2500_UNIT_01_FIXTURE_1".CLAMPED_WITH_PART_ANALOG )
      wire#w2
      Coil( "DB2440_GLOBAL_DATA".GLOBAL_DATA.FIX_IN_UNIT_01_STA_2_CLAMPED_ANALOG )
   END_RUNG
   RUNG wire#w1
      Contact( "DB4000_FIX_TABLE_POSITIONS".UNIT_01.FIXTURE_2.IN_SPARE_STATION_2 )
      Contact( "DB2600_UNIT_01_FIXTURE_2".CLAMPED_WITH_PART_ANALOG )
   END_RUNG wire#w2
   RUNG wire#w1
      Contact( "DB4000_FIX_TABLE_POSITIONS".UNIT_01.FIXTURE_3.IN_SPARE_STATION_2 )
      Contact( "DB2700_UNIT_01_FIXTURE_3".CLAMPED_WITH_PART_ANALOG )
   END_RUNG wire#w2
   RUNG wire#w1
      Contact( "DB4000_FIX_TABLE_POSITIONS".UNIT_01.FIXTURE_4.IN_SPARE_STATION_2 )
      Contact( "DB2800_UNIT_01_FIXTURE_4".CLAMPED_WITH_PART_ANALOG )
   END_RUNG wire#w2
   // the same network as SCL:
   "DB2440_GLOBAL_DATA".GLOBAL_DATA.FIX_IN_UNIT_01_STA_2_CLAMPED_ANALOG := "M_ONE" AND (("DB4000_FIX_TABLE_POSITIONS".UNIT_01.FIXTURE_1.IN_SPARE_STATION_2 AND "DB2500_UNIT_01_FIXTURE_1".CLAMPED_WITH_PART_ANALOG) OR ("DB4000_FIX_TABLE_POSITIONS".UNIT_01.FIXTURE_2.IN_SPARE_STATION_2 AND "DB2600_UNIT_01_FIXTURE_2".CLAMPED_WITH_PART_ANALOG) OR ("DB4000_FIX_TABLE_POSITIONS".UNIT_01.FIXTURE_3.IN_SPARE_STATION_2 AND "DB2700_UNIT_01_FIXTURE_3".CLAMPED_WITH_PART_ANALOG) OR ("DB4000_FIX_TABLE_POSITIONS".UNIT_01.FIXTURE_4.IN_SPARE_STATION_2 AND "DB2800_UNIT_01_FIXTURE_4".CLAMPED_WITH_PART_ANALOG));
END_REGION

REGION Network 29: FIXTURE IN UNIT 02 MEASURING POSITION UNCLAMPED ANALOG
   RUNG wire#powerrail
      Contact( "M_ONE" )
      wire#w1
      Contact( "DB4000_FIX_TABLE_POSITIONS".UNIT_02.FIXTURE_1.IN_MEASURING_STATION_2 )
      Contact( "DB3500_UNIT_02_FIXTURE_1".UNCLAMPED_ANALOG )
      wire#w2
      Coil( "DB2440_GLOBAL_DATA".GLOBAL_DATA.FIX_IN_UNIT_02_STA_2_UNCLAMPED_ANALOG )
   END_RUNG
   RUNG wire#w1
      Contact( "DB4000_FIX_TABLE_POSITIONS".UNIT_02.FIXTURE_2.IN_MEASURING_STATION_2 )
      Contact( "DB3600_UNIT_02_FIXTURE_2".UNCLAMPED_ANALOG )
   END_RUNG wire#w2
   RUNG wire#w1
      Contact( "DB4000_FIX_TABLE_POSITIONS".UNIT_02.FIXTURE_3.IN_MEASURING_STATION_2 )
      Contact( "DB3700_UNIT_02_FIXTURE_3".UNCLAMPED_ANALOG )
   END_RUNG wire#w2
   RUNG wire#w1
      Contact( "DB4000_FIX_TABLE_POSITIONS".UNIT_02.FIXTURE_4.IN_MEASURING_STATION_2 )
      Contact( "DB3800_UNIT_02_FIXTURE_4".UNCLAMPED_ANALOG )
   END_RUNG wire#w2
   // the same network as SCL:
   "DB2440_GLOBAL_DATA".GLOBAL_DATA.FIX_IN_UNIT_02_STA_2_UNCLAMPED_ANALOG := "M_ONE" AND (("DB4000_FIX_TABLE_POSITIONS".UNIT_02.FIXTURE_1.IN_MEASURING_STATION_2 AND "DB3500_UNIT_02_FIXTURE_1".UNCLAMPED_ANALOG) OR ("DB4000_FIX_TABLE_POSITIONS".UNIT_02.FIXTURE_2.IN_MEASURING_STATION_2 AND "DB3600_UNIT_02_FIXTURE_2".UNCLAMPED_ANALOG) OR ("DB4000_FIX_TABLE_POSITIONS".UNIT_02.FIXTURE_3.IN_MEASURING_STATION_2 AND "DB3700_UNIT_02_FIXTURE_3".UNCLAMPED_ANALOG) OR ("DB4000_FIX_TABLE_POSITIONS".UNIT_02.FIXTURE_4.IN_MEASURING_STATION_2 AND "DB3800_UNIT_02_FIXTURE_4".UNCLAMPED_ANALOG));
END_REGION

REGION Network 30: FIXTURE IN UNIT 02 MEASURING POSITION CLAMPED ANALOG
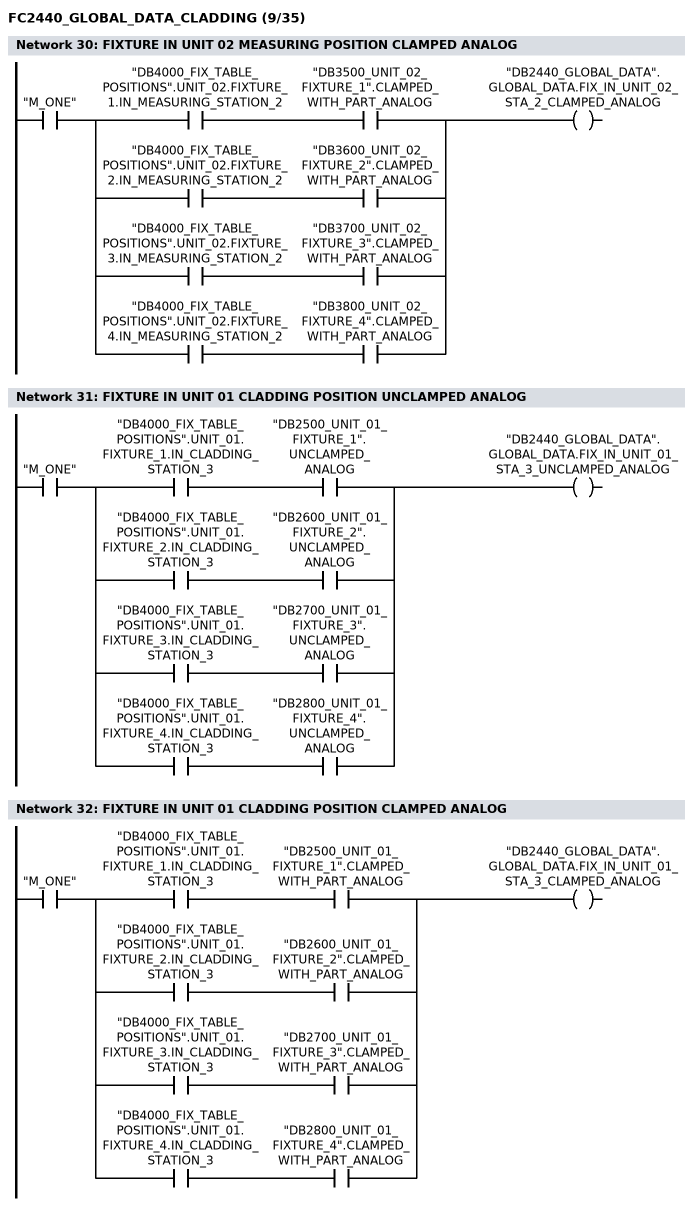
   RUNG wire#powerrail
      Contact( "M_ONE" )
      wire#w1
      Contact( "DB4000_FIX_TABLE_POSITIONS".UNIT_02.FIXTURE_1.IN_MEASURING_STATION_2 )
      Contact( "DB3500_UNIT_02_FIXTURE_1".CLAMPED_WITH_PART_ANALOG )
      wire#w2
      Coil( "DB2440_GLOBAL_DATA".GLOBAL_DATA.FIX_IN_UNIT_02_STA_2_CLAMPED_ANALOG )
   END_RUNG
   RUNG wire#w1
      Contact( "DB4000_FIX_TABLE_POSITIONS".UNIT_02.FIXTURE_2.IN_MEASURING_STATION_2 )
      Contact( "DB3600_UNIT_02_FIXTURE_2".CLAMPED_WITH_PART_ANALOG )
   END_RUNG wire#w2
   RUNG wire#w1
      Contact( "DB4000_FIX_TABLE_POSITIONS".UNIT_02.FIXTURE_3.IN_MEASURING_STATION_2 )
      Contact( "DB3700_UNIT_02_FIXTURE_3".CLAMPED_WITH_PART_ANALOG )
   END_RUNG wire#w2
   RUNG wire#w1
      Contact( "DB4000_FIX_TABLE_POSITIONS".UNIT_02.FIXTURE_4.IN_MEASURING_STATION_2 )
      Contact( "DB3800_UNIT_02_FIXTURE_4".CLAMPED_WITH_PART_ANALOG )
   END_RUNG wire#w2
   // the same network as SCL:
   "DB2440_GLOBAL_DATA".GLOBAL_DATA.FIX_IN_UNIT_02_STA_2_CLAMPED_ANALOG := "M_ONE" AND (("DB4000_FIX_TABLE_POSITIONS".UNIT_02.FIXTURE_1.IN_MEASURING_STATION_2 AND "DB3500_UNIT_02_FIXTURE_1".CLAMPED_WITH_PART_ANALOG) OR ("DB4000_FIX_TABLE_POSITIONS".UNIT_02.FIXTURE_2.IN_MEASURING_STATION_2 AND "DB3600_UNIT_02_FIXTURE_2".CLAMPED_WITH_PART_ANALOG) OR ("DB4000_FIX_TABLE_POSITIONS".UNIT_02.FIXTURE_3.IN_MEASURING_STATION_2 AND "DB3700_UNIT_02_FIXTURE_3".CLAMPED_WITH_PART_ANALOG) OR ("DB4000_FIX_TABLE_POSITIONS".UNIT_02.FIXTURE_4.IN_MEASURING_STATION_2 AND "DB3800_UNIT_02_FIXTURE_4".CLAMPED_WITH_PART_ANALOG));
END_REGION

REGION Network 31: FIXTURE IN UNIT 01 CLADDING POSITION UNCLAMPED ANALOG
   RUNG wire#powerrail
      Contact( "M_ONE" )
      wire#w1
      Contact( "DB4000_FIX_TABLE_POSITIONS".UNIT_01.FIXTURE_1.IN_CLADDING_STATION_3 )
      Contact( "DB2500_UNIT_01_FIXTURE_1".UNCLAMPED_ANALOG )
      wire#w2
      Coil( "DB2440_GLOBAL_DATA".GLOBAL_DATA.FIX_IN_UNIT_01_STA_3_UNCLAMPED_ANALOG )
   END_RUNG
   RUNG wire#w1
      Contact( "DB4000_FIX_TABLE_POSITIONS".UNIT_01.FIXTURE_2.IN_CLADDING_STATION_3 )
      Contact( "DB2600_UNIT_01_FIXTURE_2".UNCLAMPED_ANALOG )
   END_RUNG wire#w2
   RUNG wire#w1
      Contact( "DB4000_FIX_TABLE_POSITIONS".UNIT_01.FIXTURE_3.IN_CLADDING_STATION_3 )
      Contact( "DB2700_UNIT_01_FIXTURE_3".UNCLAMPED_ANALOG )
   END_RUNG wire#w2
   RUNG wire#w1
      Contact( "DB4000_FIX_TABLE_POSITIONS".UNIT_01.FIXTURE_4.IN_CLADDING_STATION_3 )
      Contact( "DB2800_UNIT_01_FIXTURE_4".UNCLAMPED_ANALOG )
   END_RUNG wire#w2
   // the same network as SCL:
   "DB2440_GLOBAL_DATA".GLOBAL_DATA.FIX_IN_UNIT_01_STA_3_UNCLAMPED_ANALOG := "M_ONE" AND (("DB4000_FIX_TABLE_POSITIONS".UNIT_01.FIXTURE_1.IN_CLADDING_STATION_3 AND "DB2500_UNIT_01_FIXTURE_1".UNCLAMPED_ANALOG) OR ("DB4000_FIX_TABLE_POSITIONS".UNIT_01.FIXTURE_2.IN_CLADDING_STATION_3 AND "DB2600_UNIT_01_FIXTURE_2".UNCLAMPED_ANALOG) OR ("DB4000_FIX_TABLE_POSITIONS".UNIT_01.FIXTURE_3.IN_CLADDING_STATION_3 AND "DB2700_UNIT_01_FIXTURE_3".UNCLAMPED_ANALOG) OR ("DB4000_FIX_TABLE_POSITIONS".UNIT_01.FIXTURE_4.IN_CLADDING_STATION_3 AND "DB2800_UNIT_01_FIXTURE_4".UNCLAMPED_ANALOG));
END_REGION

REGION Network 32: FIXTURE IN UNIT 01 CLADDING POSITION CLAMPED ANALOG
   RUNG wire#powerrail
      Contact( "M_ONE" )
      wire#w1
      Contact( "DB4000_FIX_TABLE_POSITIONS".UNIT_01.FIXTURE_1.IN_CLADDING_STATION_3 )
      Contact( "DB2500_UNIT_01_FIXTURE_1".CLAMPED_WITH_PART_ANALOG )
      wire#w2
      Coil( "DB2440_GLOBAL_DATA".GLOBAL_DATA.FIX_IN_UNIT_01_STA_3_CLAMPED_ANALOG )
   END_RUNG
   RUNG wire#w1
      Contact( "DB4000_FIX_TABLE_POSITIONS".UNIT_01.FIXTURE_2.IN_CLADDING_STATION_3 )
      Contact( "DB2600_UNIT_01_FIXTURE_2".CLAMPED_WITH_PART_ANALOG )
   END_RUNG wire#w2
   RUNG wire#w1
      Contact( "DB4000_FIX_TABLE_POSITIONS".UNIT_01.FIXTURE_3.IN_CLADDING_STATION_3 )
      Contact( "DB2700_UNIT_01_FIXTURE_3".CLAMPED_WITH_PART_ANALOG )
   END_RUNG wire#w2
   RUNG wire#w1
      Contact( "DB4000_FIX_TABLE_POSITIONS".UNIT_01.FIXTURE_4.IN_CLADDING_STATION_3 )
      Contact( "DB2800_UNIT_01_FIXTURE_4".CLAMPED_WITH_PART_ANALOG )
   END_RUNG wire#w2
   // the same network as SCL:
   "DB2440_GLOBAL_DATA".GLOBAL_DATA.FIX_IN_UNIT_01_STA_3_CLAMPED_ANALOG := "M_ONE" AND (("DB4000_FIX_TABLE_POSITIONS".UNIT_01.FIXTURE_1.IN_CLADDING_STATION_3 AND "DB2500_UNIT_01_FIXTURE_1".CLAMPED_WITH_PART_ANALOG) OR ("DB4000_FIX_TABLE_POSITIONS".UNIT_01.FIXTURE_2.IN_CLADDING_STATION_3 AND "DB2600_UNIT_01_FIXTURE_2".CLAMPED_WITH_PART_ANALOG) OR ("DB4000_FIX_TABLE_POSITIONS".UNIT_01.FIXTURE_3.IN_CLADDING_STATION_3 AND "DB2700_UNIT_01_FIXTURE_3".CLAMPED_WITH_PART_ANALOG) OR ("DB4000_FIX_TABLE_POSITIONS".UNIT_01.FIXTURE_4.IN_CLADDING_STATION_3 AND "DB2800_UNIT_01_FIXTURE_4".CLAMPED_WITH_PART_ANALOG));
END_REGION

REGION Network 33: FIXTURE IN UNIT 02 CLADDING POSITION UNCLAMPED ANALOG
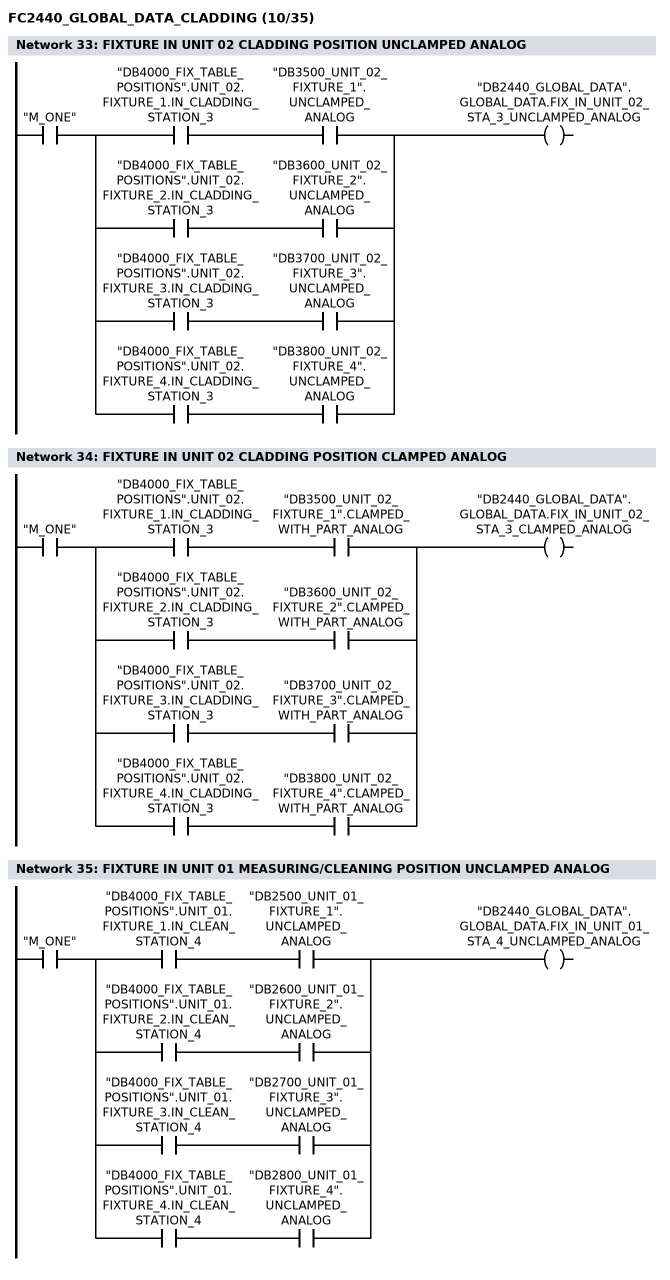
   RUNG wire#powerrail
      Contact( "M_ONE" )
      wire#w1
      Contact( "DB4000_FIX_TABLE_POSITIONS".UNIT_02.FIXTURE_1.IN_CLADDING_STATION_3 )
      Contact( "DB3500_UNIT_02_FIXTURE_1".UNCLAMPED_ANALOG )
      wire#w2
      Coil( "DB2440_GLOBAL_DATA".GLOBAL_DATA.FIX_IN_UNIT_02_STA_3_UNCLAMPED_ANALOG )
   END_RUNG
   RUNG wire#w1
      Contact( "DB4000_FIX_TABLE_POSITIONS".UNIT_02.FIXTURE_2.IN_CLADDING_STATION_3 )
      Contact( "DB3600_UNIT_02_FIXTURE_2".UNCLAMPED_ANALOG )
   END_RUNG wire#w2
   RUNG wire#w1
      Contact( "DB4000_FIX_TABLE_POSITIONS".UNIT_02.FIXTURE_3.IN_CLADDING_STATION_3 )
      Contact( "DB3700_UNIT_02_FIXTURE_3".UNCLAMPED_ANALOG )
   END_RUNG wire#w2
   RUNG wire#w1
      Contact( "DB4000_FIX_TABLE_POSITIONS".UNIT_02.FIXTURE_4.IN_CLADDING_STATION_3 )
      Contact( "DB3800_UNIT_02_FIXTURE_4".UNCLAMPED_ANALOG )
   END_RUNG wire#w2
   // the same network as SCL:
   "DB2440_GLOBAL_DATA".GLOBAL_DATA.FIX_IN_UNIT_02_STA_3_UNCLAMPED_ANALOG := "M_ONE" AND (("DB4000_FIX_TABLE_POSITIONS".UNIT_02.FIXTURE_1.IN_CLADDING_STATION_3 AND "DB3500_UNIT_02_FIXTURE_1".UNCLAMPED_ANALOG) OR ("DB4000_FIX_TABLE_POSITIONS".UNIT_02.FIXTURE_2.IN_CLADDING_STATION_3 AND "DB3600_UNIT_02_FIXTURE_2".UNCLAMPED_ANALOG) OR ("DB4000_FIX_TABLE_POSITIONS".UNIT_02.FIXTURE_3.IN_CLADDING_STATION_3 AND "DB3700_UNIT_02_FIXTURE_3".UNCLAMPED_ANALOG) OR ("DB4000_FIX_TABLE_POSITIONS".UNIT_02.FIXTURE_4.IN_CLADDING_STATION_3 AND "DB3800_UNIT_02_FIXTURE_4".UNCLAMPED_ANALOG));
END_REGION

REGION Network 34: FIXTURE IN UNIT 02 CLADDING POSITION CLAMPED ANALOG
   RUNG wire#powerrail
      Contact( "M_ONE" )
      wire#w1
      Contact( "DB4000_FIX_TABLE_POSITIONS".UNIT_02.FIXTURE_1.IN_CLADDING_STATION_3 )
      Contact( "DB3500_UNIT_02_FIXTURE_1".CLAMPED_WITH_PART_ANALOG )
      wire#w2
      Coil( "DB2440_GLOBAL_DATA".GLOBAL_DATA.FIX_IN_UNIT_02_STA_3_CLAMPED_ANALOG )
   END_RUNG
   RUNG wire#w1
      Contact( "DB4000_FIX_TABLE_POSITIONS".UNIT_02.FIXTURE_2.IN_CLADDING_STATION_3 )
      Contact( "DB3600_UNIT_02_FIXTURE_2".CLAMPED_WITH_PART_ANALOG )
   END_RUNG wire#w2
   RUNG wire#w1
      Contact( "DB4000_FIX_TABLE_POSITIONS".UNIT_02.FIXTURE_3.IN_CLADDING_STATION_3 )
      Contact( "DB3700_UNIT_02_FIXTURE_3".CLAMPED_WITH_PART_ANALOG )
   END_RUNG wire#w2
   RUNG wire#w1
      Contact( "DB4000_FIX_TABLE_POSITIONS".UNIT_02.FIXTURE_4.IN_CLADDING_STATION_3 )
      Contact( "DB3800_UNIT_02_FIXTURE_4".CLAMPED_WITH_PART_ANALOG )
   END_RUNG wire#w2
   // the same network as SCL:
   "DB2440_GLOBAL_DATA".GLOBAL_DATA.FIX_IN_UNIT_02_STA_3_CLAMPED_ANALOG := "M_ONE" AND (("DB4000_FIX_TABLE_POSITIONS".UNIT_02.FIXTURE_1.IN_CLADDING_STATION_3 AND "DB3500_UNIT_02_FIXTURE_1".CLAMPED_WITH_PART_ANALOG) OR ("DB4000_FIX_TABLE_POSITIONS".UNIT_02.FIXTURE_2.IN_CLADDING_STATION_3 AND "DB3600_UNIT_02_FIXTURE_2".CLAMPED_WITH_PART_ANALOG) OR ("DB4000_FIX_TABLE_POSITIONS".UNIT_02.FIXTURE_3.IN_CLADDING_STATION_3 AND "DB3700_UNIT_02_FIXTURE_3".CLAMPED_WITH_PART_ANALOG) OR ("DB4000_FIX_TABLE_POSITIONS".UNIT_02.FIXTURE_4.IN_CLADDING_STATION_3 AND "DB3800_UNIT_02_FIXTURE_4".CLAMPED_WITH_PART_ANALOG));
END_REGION

REGION Network 35: FIXTURE IN UNIT 01 MEASURING/CLEANING POSITION UNCLAMPED ANALOG
   RUNG wire#powerrail
      Contact( "M_ONE" )
      wire#w1
      Contact( "DB4000_FIX_TABLE_POSITIONS".UNIT_01.FIXTURE_1.IN_CLEAN_STATION_4 )
      Contact( "DB2500_UNIT_01_FIXTURE_1".UNCLAMPED_ANALOG )
      wire#w2
      Coil( "DB2440_GLOBAL_DATA".GLOBAL_DATA.FIX_IN_UNIT_01_STA_4_UNCLAMPED_ANALOG )
   END_RUNG
   RUNG wire#w1
      Contact( "DB4000_FIX_TABLE_POSITIONS".UNIT_01.FIXTURE_2.IN_CLEAN_STATION_4 )
      Contact( "DB2600_UNIT_01_FIXTURE_2".UNCLAMPED_ANALOG )
   END_RUNG wire#w2
   RUNG wire#w1
      Contact( "DB4000_FIX_TABLE_POSITIONS".UNIT_01.FIXTURE_3.IN_CLEAN_STATION_4 )
      Contact( "DB2700_UNIT_01_FIXTURE_3".UNCLAMPED_ANALOG )
   END_RUNG wire#w2
   RUNG wire#w1
      Contact( "DB4000_FIX_TABLE_POSITIONS".UNIT_01.FIXTURE_4.IN_CLEAN_STATION_4 )
      Contact( "DB2800_UNIT_01_FIXTURE_4".UNCLAMPED_ANALOG )
   END_RUNG wire#w2
   // the same network as SCL:
   "DB2440_GLOBAL_DATA".GLOBAL_DATA.FIX_IN_UNIT_01_STA_4_UNCLAMPED_ANALOG := "M_ONE" AND (("DB4000_FIX_TABLE_POSITIONS".UNIT_01.FIXTURE_1.IN_CLEAN_STATION_4 AND "DB2500_UNIT_01_FIXTURE_1".UNCLAMPED_ANALOG) OR ("DB4000_FIX_TABLE_POSITIONS".UNIT_01.FIXTURE_2.IN_CLEAN_STATION_4 AND "DB2600_UNIT_01_FIXTURE_2".UNCLAMPED_ANALOG) OR ("DB4000_FIX_TABLE_POSITIONS".UNIT_01.FIXTURE_3.IN_CLEAN_STATION_4 AND "DB2700_UNIT_01_FIXTURE_3".UNCLAMPED_ANALOG) OR ("DB4000_FIX_TABLE_POSITIONS".UNIT_01.FIXTURE_4.IN_CLEAN_STATION_4 AND "DB2800_UNIT_01_FIXTURE_4".UNCLAMPED_ANALOG));
END_REGION

REGION Network 36: FIXTURE IN UNIT 01 MEASURING/CLEANING POSITION CLAMPED ANALOG
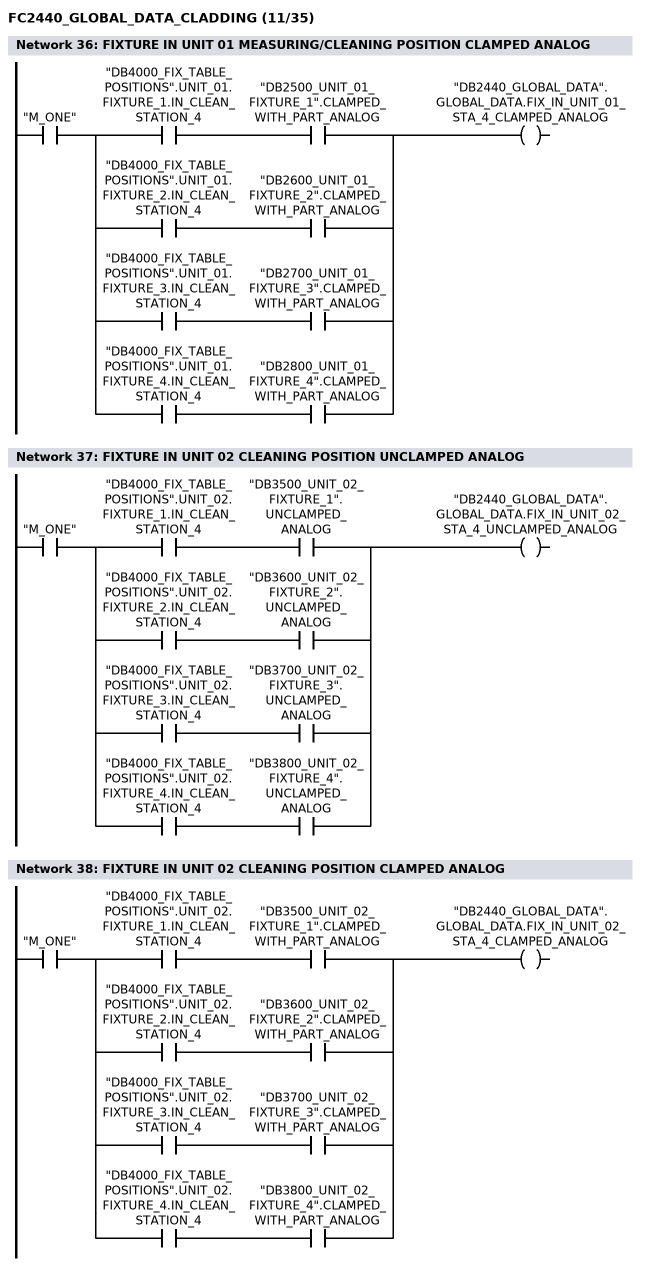
   RUNG wire#powerrail
      Contact( "M_ONE" )
      wire#w1
      Contact( "DB4000_FIX_TABLE_POSITIONS".UNIT_01.FIXTURE_1.IN_CLEAN_STATION_4 )
      Contact( "DB2500_UNIT_01_FIXTURE_1".CLAMPED_WITH_PART_ANALOG )
      wire#w2
      Coil( "DB2440_GLOBAL_DATA".GLOBAL_DATA.FIX_IN_UNIT_01_STA_4_CLAMPED_ANALOG )
   END_RUNG
   RUNG wire#w1
      Contact( "DB4000_FIX_TABLE_POSITIONS".UNIT_01.FIXTURE_2.IN_CLEAN_STATION_4 )
      Contact( "DB2600_UNIT_01_FIXTURE_2".CLAMPED_WITH_PART_ANALOG )
   END_RUNG wire#w2
   RUNG wire#w1
      Contact( "DB4000_FIX_TABLE_POSITIONS".UNIT_01.FIXTURE_3.IN_CLEAN_STATION_4 )
      Contact( "DB2700_UNIT_01_FIXTURE_3".CLAMPED_WITH_PART_ANALOG )
   END_RUNG wire#w2
   RUNG wire#w1
      Contact( "DB4000_FIX_TABLE_POSITIONS".UNIT_01.FIXTURE_4.IN_CLEAN_STATION_4 )
      Contact( "DB2800_UNIT_01_FIXTURE_4".CLAMPED_WITH_PART_ANALOG )
   END_RUNG wire#w2
   // the same network as SCL:
   "DB2440_GLOBAL_DATA".GLOBAL_DATA.FIX_IN_UNIT_01_STA_4_CLAMPED_ANALOG := "M_ONE" AND (("DB4000_FIX_TABLE_POSITIONS".UNIT_01.FIXTURE_1.IN_CLEAN_STATION_4 AND "DB2500_UNIT_01_FIXTURE_1".CLAMPED_WITH_PART_ANALOG) OR ("DB4000_FIX_TABLE_POSITIONS".UNIT_01.FIXTURE_2.IN_CLEAN_STATION_4 AND "DB2600_UNIT_01_FIXTURE_2".CLAMPED_WITH_PART_ANALOG) OR ("DB4000_FIX_TABLE_POSITIONS".UNIT_01.FIXTURE_3.IN_CLEAN_STATION_4 AND "DB2700_UNIT_01_FIXTURE_3".CLAMPED_WITH_PART_ANALOG) OR ("DB4000_FIX_TABLE_POSITIONS".UNIT_01.FIXTURE_4.IN_CLEAN_STATION_4 AND "DB2800_UNIT_01_FIXTURE_4".CLAMPED_WITH_PART_ANALOG));
END_REGION

REGION Network 37: FIXTURE IN UNIT 02 CLEANING POSITION UNCLAMPED ANALOG
   RUNG wire#powerrail
      Contact( "M_ONE" )
      wire#w1
      Contact( "DB4000_FIX_TABLE_POSITIONS".UNIT_02.FIXTURE_1.IN_CLEAN_STATION_4 )
      Contact( "DB3500_UNIT_02_FIXTURE_1".UNCLAMPED_ANALOG )
      wire#w2
      Coil( "DB2440_GLOBAL_DATA".GLOBAL_DATA.FIX_IN_UNIT_02_STA_4_UNCLAMPED_ANALOG )
   END_RUNG
   RUNG wire#w1
      Contact( "DB4000_FIX_TABLE_POSITIONS".UNIT_02.FIXTURE_2.IN_CLEAN_STATION_4 )
      Contact( "DB3600_UNIT_02_FIXTURE_2".UNCLAMPED_ANALOG )
   END_RUNG wire#w2
   RUNG wire#w1
      Contact( "DB4000_FIX_TABLE_POSITIONS".UNIT_02.FIXTURE_3.IN_CLEAN_STATION_4 )
      Contact( "DB3700_UNIT_02_FIXTURE_3".UNCLAMPED_ANALOG )
   END_RUNG wire#w2
   RUNG wire#w1
      Contact( "DB4000_FIX_TABLE_POSITIONS".UNIT_02.FIXTURE_4.IN_CLEAN_STATION_4 )
      Contact( "DB3800_UNIT_02_FIXTURE_4".UNCLAMPED_ANALOG )
   END_RUNG wire#w2
   // the same network as SCL:
   "DB2440_GLOBAL_DATA".GLOBAL_DATA.FIX_IN_UNIT_02_STA_4_UNCLAMPED_ANALOG := "M_ONE" AND (("DB4000_FIX_TABLE_POSITIONS".UNIT_02.FIXTURE_1.IN_CLEAN_STATION_4 AND "DB3500_UNIT_02_FIXTURE_1".UNCLAMPED_ANALOG) OR ("DB4000_FIX_TABLE_POSITIONS".UNIT_02.FIXTURE_2.IN_CLEAN_STATION_4 AND "DB3600_UNIT_02_FIXTURE_2".UNCLAMPED_ANALOG) OR ("DB4000_FIX_TABLE_POSITIONS".UNIT_02.FIXTURE_3.IN_CLEAN_STATION_4 AND "DB3700_UNIT_02_FIXTURE_3".UNCLAMPED_ANALOG) OR ("DB4000_FIX_TABLE_POSITIONS".UNIT_02.FIXTURE_4.IN_CLEAN_STATION_4 AND "DB3800_UNIT_02_FIXTURE_4".UNCLAMPED_ANALOG));
END_REGION

REGION Network 38: FIXTURE IN UNIT 02 CLEANING POSITION CLAMPED ANALOG
   RUNG wire#powerrail
      Contact( "M_ONE" )
      wire#w1
      Contact( "DB4000_FIX_TABLE_POSITIONS".UNIT_02.FIXTURE_1.IN_CLEAN_STATION_4 )
      Contact( "DB3500_UNIT_02_FIXTURE_1".CLAMPED_WITH_PART_ANALOG )
      wire#w2
      Coil( "DB2440_GLOBAL_DATA".GLOBAL_DATA.FIX_IN_UNIT_02_STA_4_CLAMPED_ANALOG )
   END_RUNG
   RUNG wire#w1
      Contact( "DB4000_FIX_TABLE_POSITIONS".UNIT_02.FIXTURE_2.IN_CLEAN_STATION_4 )
      Contact( "DB3600_UNIT_02_FIXTURE_2".CLAMPED_WITH_PART_ANALOG )
   END_RUNG wire#w2
   RUNG wire#w1
      Contact( "DB4000_FIX_TABLE_POSITIONS".UNIT_02.FIXTURE_3.IN_CLEAN_STATION_4 )
      Contact( "DB3700_UNIT_02_FIXTURE_3".CLAMPED_WITH_PART_ANALOG )
   END_RUNG wire#w2
   RUNG wire#w1
      Contact( "DB4000_FIX_TABLE_POSITIONS".UNIT_02.FIXTURE_4.IN_CLEAN_STATION_4 )
      Contact( "DB3800_UNIT_02_FIXTURE_4".CLAMPED_WITH_PART_ANALOG )
   END_RUNG wire#w2
   // the same network as SCL:
   "DB2440_GLOBAL_DATA".GLOBAL_DATA.FIX_IN_UNIT_02_STA_4_CLAMPED_ANALOG := "M_ONE" AND (("DB4000_FIX_TABLE_POSITIONS".UNIT_02.FIXTURE_1.IN_CLEAN_STATION_4 AND "DB3500_UNIT_02_FIXTURE_1".CLAMPED_WITH_PART_ANALOG) OR ("DB4000_FIX_TABLE_POSITIONS".UNIT_02.FIXTURE_2.IN_CLEAN_STATION_4 AND "DB3600_UNIT_02_FIXTURE_2".CLAMPED_WITH_PART_ANALOG) OR ("DB4000_FIX_TABLE_POSITIONS".UNIT_02.FIXTURE_3.IN_CLEAN_STATION_4 AND "DB3700_UNIT_02_FIXTURE_3".CLAMPED_WITH_PART_ANALOG) OR ("DB4000_FIX_TABLE_POSITIONS".UNIT_02.FIXTURE_4.IN_CLEAN_STATION_4 AND "DB3800_UNIT_02_FIXTURE_4".CLAMPED_WITH_PART_ANALOG));
END_REGION

REGION Network 39: FIXTURE IN UNIT 01 LOAD UNLOAD POSITION UNCLAMPED
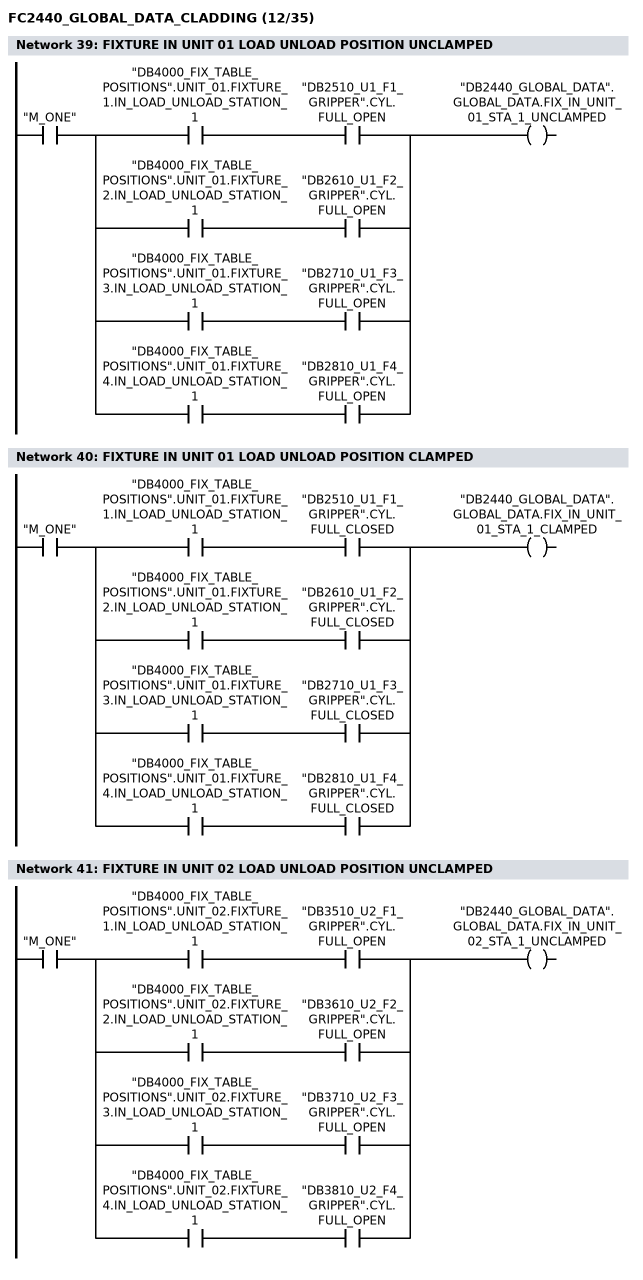
   RUNG wire#powerrail
      Contact( "M_ONE" )
      wire#w1
      Contact( "DB4000_FIX_TABLE_POSITIONS".UNIT_01.FIXTURE_1.IN_LOAD_UNLOAD_STATION_1 )
      Contact( "DB2510_U1_F1_GRIPPER".CYL.FULL_OPEN )
      wire#w2
      Coil( "DB2440_GLOBAL_DATA".GLOBAL_DATA.FIX_IN_UNIT_01_STA_1_UNCLAMPED )
   END_RUNG
   RUNG wire#w1
      Contact( "DB4000_FIX_TABLE_POSITIONS".UNIT_01.FIXTURE_2.IN_LOAD_UNLOAD_STATION_1 )
      Contact( "DB2610_U1_F2_GRIPPER".CYL.FULL_OPEN )
   END_RUNG wire#w2
   RUNG wire#w1
      Contact( "DB4000_FIX_TABLE_POSITIONS".UNIT_01.FIXTURE_3.IN_LOAD_UNLOAD_STATION_1 )
      Contact( "DB2710_U1_F3_GRIPPER".CYL.FULL_OPEN )
   END_RUNG wire#w2
   RUNG wire#w1
      Contact( "DB4000_FIX_TABLE_POSITIONS".UNIT_01.FIXTURE_4.IN_LOAD_UNLOAD_STATION_1 )
      Contact( "DB2810_U1_F4_GRIPPER".CYL.FULL_OPEN )
   END_RUNG wire#w2
   // the same network as SCL:
   "DB2440_GLOBAL_DATA".GLOBAL_DATA.FIX_IN_UNIT_01_STA_1_UNCLAMPED := "M_ONE" AND (("DB4000_FIX_TABLE_POSITIONS".UNIT_01.FIXTURE_1.IN_LOAD_UNLOAD_STATION_1 AND "DB2510_U1_F1_GRIPPER".CYL.FULL_OPEN) OR ("DB4000_FIX_TABLE_POSITIONS".UNIT_01.FIXTURE_2.IN_LOAD_UNLOAD_STATION_1 AND "DB2610_U1_F2_GRIPPER".CYL.FULL_OPEN) OR ("DB4000_FIX_TABLE_POSITIONS".UNIT_01.FIXTURE_3.IN_LOAD_UNLOAD_STATION_1 AND "DB2710_U1_F3_GRIPPER".CYL.FULL_OPEN) OR ("DB4000_FIX_TABLE_POSITIONS".UNIT_01.FIXTURE_4.IN_LOAD_UNLOAD_STATION_1 AND "DB2810_U1_F4_GRIPPER".CYL.FULL_OPEN));
END_REGION

REGION Network 40: FIXTURE IN UNIT 01 LOAD UNLOAD POSITION CLAMPED
   RUNG wire#powerrail
      Contact( "M_ONE" )
      wire#w1
      Contact( "DB4000_FIX_TABLE_POSITIONS".UNIT_01.FIXTURE_1.IN_LOAD_UNLOAD_STATION_1 )
      Contact( "DB2510_U1_F1_GRIPPER".CYL.FULL_CLOSED )
      wire#w2
      Coil( "DB2440_GLOBAL_DATA".GLOBAL_DATA.FIX_IN_UNIT_01_STA_1_CLAMPED )
   END_RUNG
   RUNG wire#w1
      Contact( "DB4000_FIX_TABLE_POSITIONS".UNIT_01.FIXTURE_2.IN_LOAD_UNLOAD_STATION_1 )
      Contact( "DB2610_U1_F2_GRIPPER".CYL.FULL_CLOSED )
   END_RUNG wire#w2
   RUNG wire#w1
      Contact( "DB4000_FIX_TABLE_POSITIONS".UNIT_01.FIXTURE_3.IN_LOAD_UNLOAD_STATION_1 )
      Contact( "DB2710_U1_F3_GRIPPER".CYL.FULL_CLOSED )
   END_RUNG wire#w2
   RUNG wire#w1
      Contact( "DB4000_FIX_TABLE_POSITIONS".UNIT_01.FIXTURE_4.IN_LOAD_UNLOAD_STATION_1 )
      Contact( "DB2810_U1_F4_GRIPPER".CYL.FULL_CLOSED )
   END_RUNG wire#w2
   // the same network as SCL:
   "DB2440_GLOBAL_DATA".GLOBAL_DATA.FIX_IN_UNIT_01_STA_1_CLAMPED := "M_ONE" AND (("DB4000_FIX_TABLE_POSITIONS".UNIT_01.FIXTURE_1.IN_LOAD_UNLOAD_STATION_1 AND "DB2510_U1_F1_GRIPPER".CYL.FULL_CLOSED) OR ("DB4000_FIX_TABLE_POSITIONS".UNIT_01.FIXTURE_2.IN_LOAD_UNLOAD_STATION_1 AND "DB2610_U1_F2_GRIPPER".CYL.FULL_CLOSED) OR ("DB4000_FIX_TABLE_POSITIONS".UNIT_01.FIXTURE_3.IN_LOAD_UNLOAD_STATION_1 AND "DB2710_U1_F3_GRIPPER".CYL.FULL_CLOSED) OR ("DB4000_FIX_TABLE_POSITIONS".UNIT_01.FIXTURE_4.IN_LOAD_UNLOAD_STATION_1 AND "DB2810_U1_F4_GRIPPER".CYL.FULL_CLOSED));
END_REGION

REGION Network 41: FIXTURE IN UNIT 02 LOAD UNLOAD POSITION UNCLAMPED
   RUNG wire#powerrail
      Contact( "M_ONE" )
      wire#w1
      Contact( "DB4000_FIX_TABLE_POSITIONS".UNIT_02.FIXTURE_1.IN_LOAD_UNLOAD_STATION_1 )
      Contact( "DB3510_U2_F1_GRIPPER".CYL.FULL_OPEN )
      wire#w2
      Coil( "DB2440_GLOBAL_DATA".GLOBAL_DATA.FIX_IN_UNIT_02_STA_1_UNCLAMPED )
   END_RUNG
   RUNG wire#w1
      Contact( "DB4000_FIX_TABLE_POSITIONS".UNIT_02.FIXTURE_2.IN_LOAD_UNLOAD_STATION_1 )
      Contact( "DB3610_U2_F2_GRIPPER".CYL.FULL_OPEN )
   END_RUNG wire#w2
   RUNG wire#w1
      Contact( "DB4000_FIX_TABLE_POSITIONS".UNIT_02.FIXTURE_3.IN_LOAD_UNLOAD_STATION_1 )
      Contact( "DB3710_U2_F3_GRIPPER".CYL.FULL_OPEN )
   END_RUNG wire#w2
   RUNG wire#w1
      Contact( "DB4000_FIX_TABLE_POSITIONS".UNIT_02.FIXTURE_4.IN_LOAD_UNLOAD_STATION_1 )
      Contact( "DB3810_U2_F4_GRIPPER".CYL.FULL_OPEN )
   END_RUNG wire#w2
   // the same network as SCL:
   "DB2440_GLOBAL_DATA".GLOBAL_DATA.FIX_IN_UNIT_02_STA_1_UNCLAMPED := "M_ONE" AND (("DB4000_FIX_TABLE_POSITIONS".UNIT_02.FIXTURE_1.IN_LOAD_UNLOAD_STATION_1 AND "DB3510_U2_F1_GRIPPER".CYL.FULL_OPEN) OR ("DB4000_FIX_TABLE_POSITIONS".UNIT_02.FIXTURE_2.IN_LOAD_UNLOAD_STATION_1 AND "DB3610_U2_F2_GRIPPER".CYL.FULL_OPEN) OR ("DB4000_FIX_TABLE_POSITIONS".UNIT_02.FIXTURE_3.IN_LOAD_UNLOAD_STATION_1 AND "DB3710_U2_F3_GRIPPER".CYL.FULL_OPEN) OR ("DB4000_FIX_TABLE_POSITIONS".UNIT_02.FIXTURE_4.IN_LOAD_UNLOAD_STATION_1 AND "DB3810_U2_F4_GRIPPER".CYL.FULL_OPEN));
END_REGION

REGION Network 42: FIXTURE IN UNIT 02 LOAD UNLOAD POSITION CLAMPED
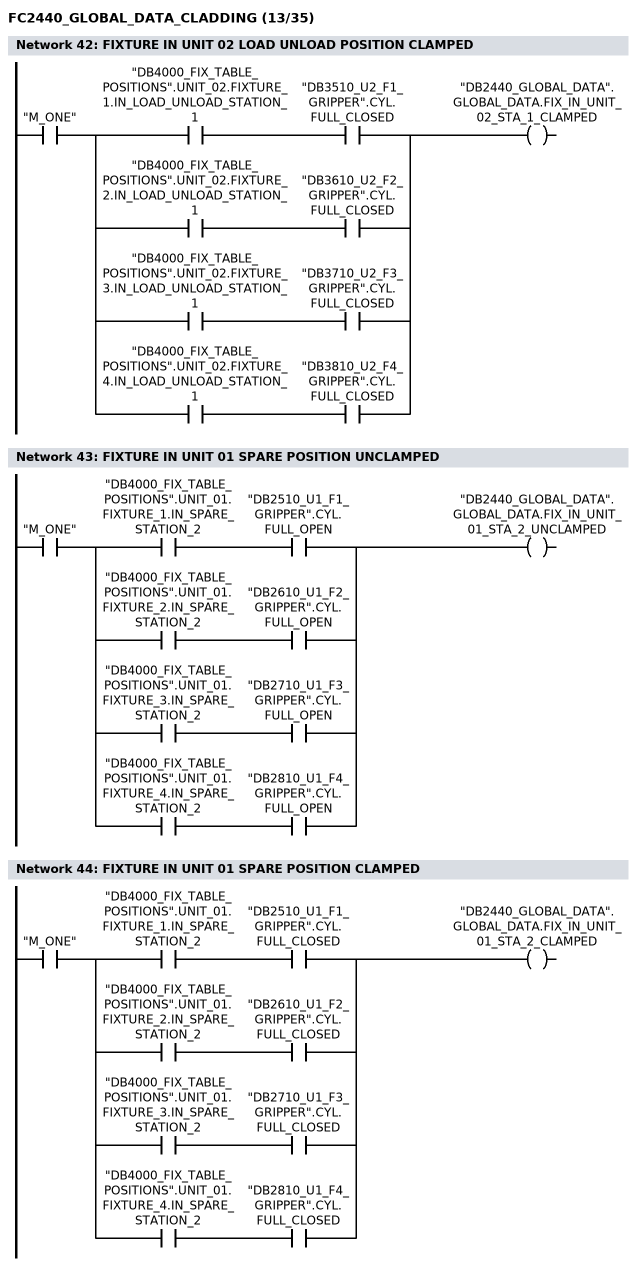
   RUNG wire#powerrail
      Contact( "M_ONE" )
      wire#w1
      Contact( "DB4000_FIX_TABLE_POSITIONS".UNIT_02.FIXTURE_1.IN_LOAD_UNLOAD_STATION_1 )
      Contact( "DB3510_U2_F1_GRIPPER".CYL.FULL_CLOSED )
      wire#w2
      Coil( "DB2440_GLOBAL_DATA".GLOBAL_DATA.FIX_IN_UNIT_02_STA_1_CLAMPED )
   END_RUNG
   RUNG wire#w1
      Contact( "DB4000_FIX_TABLE_POSITIONS".UNIT_02.FIXTURE_2.IN_LOAD_UNLOAD_STATION_1 )
      Contact( "DB3610_U2_F2_GRIPPER".CYL.FULL_CLOSED )
   END_RUNG wire#w2
   RUNG wire#w1
      Contact( "DB4000_FIX_TABLE_POSITIONS".UNIT_02.FIXTURE_3.IN_LOAD_UNLOAD_STATION_1 )
      Contact( "DB3710_U2_F3_GRIPPER".CYL.FULL_CLOSED )
   END_RUNG wire#w2
   RUNG wire#w1
      Contact( "DB4000_FIX_TABLE_POSITIONS".UNIT_02.FIXTURE_4.IN_LOAD_UNLOAD_STATION_1 )
      Contact( "DB3810_U2_F4_GRIPPER".CYL.FULL_CLOSED )
   END_RUNG wire#w2
   // the same network as SCL:
   "DB2440_GLOBAL_DATA".GLOBAL_DATA.FIX_IN_UNIT_02_STA_1_CLAMPED := "M_ONE" AND (("DB4000_FIX_TABLE_POSITIONS".UNIT_02.FIXTURE_1.IN_LOAD_UNLOAD_STATION_1 AND "DB3510_U2_F1_GRIPPER".CYL.FULL_CLOSED) OR ("DB4000_FIX_TABLE_POSITIONS".UNIT_02.FIXTURE_2.IN_LOAD_UNLOAD_STATION_1 AND "DB3610_U2_F2_GRIPPER".CYL.FULL_CLOSED) OR ("DB4000_FIX_TABLE_POSITIONS".UNIT_02.FIXTURE_3.IN_LOAD_UNLOAD_STATION_1 AND "DB3710_U2_F3_GRIPPER".CYL.FULL_CLOSED) OR ("DB4000_FIX_TABLE_POSITIONS".UNIT_02.FIXTURE_4.IN_LOAD_UNLOAD_STATION_1 AND "DB3810_U2_F4_GRIPPER".CYL.FULL_CLOSED));
END_REGION

REGION Network 43: FIXTURE IN UNIT 01 SPARE POSITION UNCLAMPED
   RUNG wire#powerrail
      Contact( "M_ONE" )
      wire#w1
      Contact( "DB4000_FIX_TABLE_POSITIONS".UNIT_01.FIXTURE_1.IN_SPARE_STATION_2 )
      Contact( "DB2510_U1_F1_GRIPPER".CYL.FULL_OPEN )
      wire#w2
      Coil( "DB2440_GLOBAL_DATA".GLOBAL_DATA.FIX_IN_UNIT_01_STA_2_UNCLAMPED )
   END_RUNG
   RUNG wire#w1
      Contact( "DB4000_FIX_TABLE_POSITIONS".UNIT_01.FIXTURE_2.IN_SPARE_STATION_2 )
      Contact( "DB2610_U1_F2_GRIPPER".CYL.FULL_OPEN )
   END_RUNG wire#w2
   RUNG wire#w1
      Contact( "DB4000_FIX_TABLE_POSITIONS".UNIT_01.FIXTURE_3.IN_SPARE_STATION_2 )
      Contact( "DB2710_U1_F3_GRIPPER".CYL.FULL_OPEN )
   END_RUNG wire#w2
   RUNG wire#w1
      Contact( "DB4000_FIX_TABLE_POSITIONS".UNIT_01.FIXTURE_4.IN_SPARE_STATION_2 )
      Contact( "DB2810_U1_F4_GRIPPER".CYL.FULL_OPEN )
   END_RUNG wire#w2
   // the same network as SCL:
   "DB2440_GLOBAL_DATA".GLOBAL_DATA.FIX_IN_UNIT_01_STA_2_UNCLAMPED := "M_ONE" AND (("DB4000_FIX_TABLE_POSITIONS".UNIT_01.FIXTURE_1.IN_SPARE_STATION_2 AND "DB2510_U1_F1_GRIPPER".CYL.FULL_OPEN) OR ("DB4000_FIX_TABLE_POSITIONS".UNIT_01.FIXTURE_2.IN_SPARE_STATION_2 AND "DB2610_U1_F2_GRIPPER".CYL.FULL_OPEN) OR ("DB4000_FIX_TABLE_POSITIONS".UNIT_01.FIXTURE_3.IN_SPARE_STATION_2 AND "DB2710_U1_F3_GRIPPER".CYL.FULL_OPEN) OR ("DB4000_FIX_TABLE_POSITIONS".UNIT_01.FIXTURE_4.IN_SPARE_STATION_2 AND "DB2810_U1_F4_GRIPPER".CYL.FULL_OPEN));
END_REGION

REGION Network 44: FIXTURE IN UNIT 01 SPARE POSITION CLAMPED
   RUNG wire#powerrail
      Contact( "M_ONE" )
      wire#w1
      Contact( "DB4000_FIX_TABLE_POSITIONS".UNIT_01.FIXTURE_1.IN_SPARE_STATION_2 )
      Contact( "DB2510_U1_F1_GRIPPER".CYL.FULL_CLOSED )
      wire#w2
      Coil( "DB2440_GLOBAL_DATA".GLOBAL_DATA.FIX_IN_UNIT_01_STA_2_CLAMPED )
   END_RUNG
   RUNG wire#w1
      Contact( "DB4000_FIX_TABLE_POSITIONS".UNIT_01.FIXTURE_2.IN_SPARE_STATION_2 )
      Contact( "DB2610_U1_F2_GRIPPER".CYL.FULL_CLOSED )
   END_RUNG wire#w2
   RUNG wire#w1
      Contact( "DB4000_FIX_TABLE_POSITIONS".UNIT_01.FIXTURE_3.IN_SPARE_STATION_2 )
      Contact( "DB2710_U1_F3_GRIPPER".CYL.FULL_CLOSED )
   END_RUNG wire#w2
   RUNG wire#w1
      Contact( "DB4000_FIX_TABLE_POSITIONS".UNIT_01.FIXTURE_4.IN_SPARE_STATION_2 )
      Contact( "DB2810_U1_F4_GRIPPER".CYL.FULL_CLOSED )
   END_RUNG wire#w2
   // the same network as SCL:
   "DB2440_GLOBAL_DATA".GLOBAL_DATA.FIX_IN_UNIT_01_STA_2_CLAMPED := "M_ONE" AND (("DB4000_FIX_TABLE_POSITIONS".UNIT_01.FIXTURE_1.IN_SPARE_STATION_2 AND "DB2510_U1_F1_GRIPPER".CYL.FULL_CLOSED) OR ("DB4000_FIX_TABLE_POSITIONS".UNIT_01.FIXTURE_2.IN_SPARE_STATION_2 AND "DB2610_U1_F2_GRIPPER".CYL.FULL_CLOSED) OR ("DB4000_FIX_TABLE_POSITIONS".UNIT_01.FIXTURE_3.IN_SPARE_STATION_2 AND "DB2710_U1_F3_GRIPPER".CYL.FULL_CLOSED) OR ("DB4000_FIX_TABLE_POSITIONS".UNIT_01.FIXTURE_4.IN_SPARE_STATION_2 AND "DB2810_U1_F4_GRIPPER".CYL.FULL_CLOSED));
END_REGION

REGION Network 45: FIXTURE IN UNIT 02 MEASURING POSITION UNCLAMPED
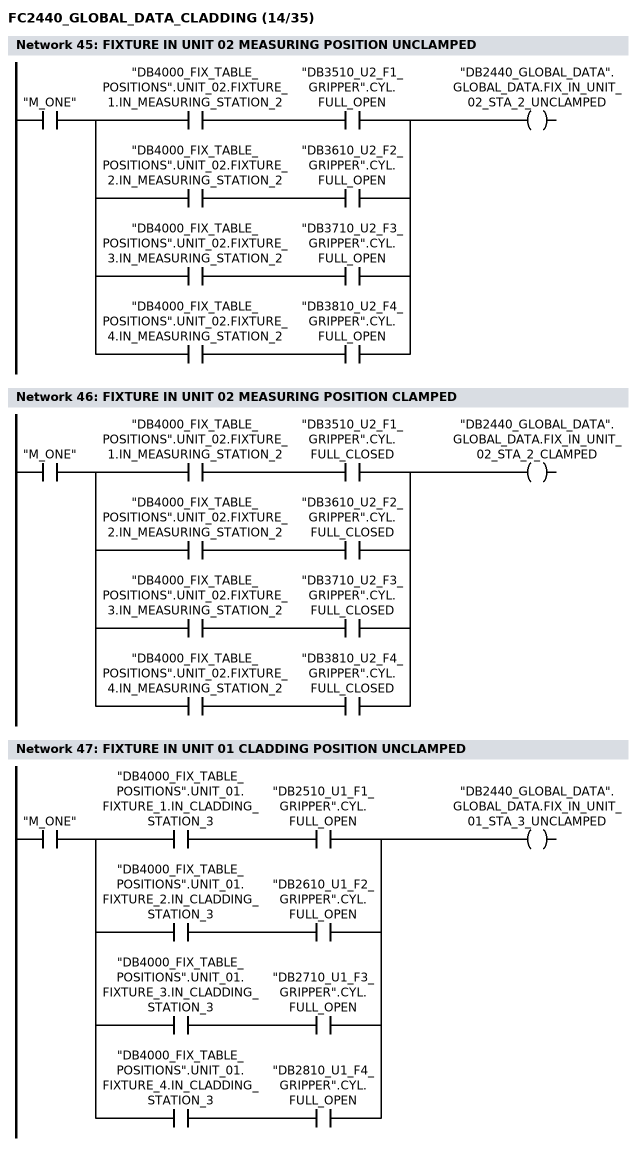
   RUNG wire#powerrail
      Contact( "M_ONE" )
      wire#w1
      Contact( "DB4000_FIX_TABLE_POSITIONS".UNIT_02.FIXTURE_1.IN_MEASURING_STATION_2 )
      Contact( "DB3510_U2_F1_GRIPPER".CYL.FULL_OPEN )
      wire#w2
      Coil( "DB2440_GLOBAL_DATA".GLOBAL_DATA.FIX_IN_UNIT_02_STA_2_UNCLAMPED )
   END_RUNG
   RUNG wire#w1
      Contact( "DB4000_FIX_TABLE_POSITIONS".UNIT_02.FIXTURE_2.IN_MEASURING_STATION_2 )
      Contact( "DB3610_U2_F2_GRIPPER".CYL.FULL_OPEN )
   END_RUNG wire#w2
   RUNG wire#w1
      Contact( "DB4000_FIX_TABLE_POSITIONS".UNIT_02.FIXTURE_3.IN_MEASURING_STATION_2 )
      Contact( "DB3710_U2_F3_GRIPPER".CYL.FULL_OPEN )
   END_RUNG wire#w2
   RUNG wire#w1
      Contact( "DB4000_FIX_TABLE_POSITIONS".UNIT_02.FIXTURE_4.IN_MEASURING_STATION_2 )
      Contact( "DB3810_U2_F4_GRIPPER".CYL.FULL_OPEN )
   END_RUNG wire#w2
   // the same network as SCL:
   "DB2440_GLOBAL_DATA".GLOBAL_DATA.FIX_IN_UNIT_02_STA_2_UNCLAMPED := "M_ONE" AND (("DB4000_FIX_TABLE_POSITIONS".UNIT_02.FIXTURE_1.IN_MEASURING_STATION_2 AND "DB3510_U2_F1_GRIPPER".CYL.FULL_OPEN) OR ("DB4000_FIX_TABLE_POSITIONS".UNIT_02.FIXTURE_2.IN_MEASURING_STATION_2 AND "DB3610_U2_F2_GRIPPER".CYL.FULL_OPEN) OR ("DB4000_FIX_TABLE_POSITIONS".UNIT_02.FIXTURE_3.IN_MEASURING_STATION_2 AND "DB3710_U2_F3_GRIPPER".CYL.FULL_OPEN) OR ("DB4000_FIX_TABLE_POSITIONS".UNIT_02.FIXTURE_4.IN_MEASURING_STATION_2 AND "DB3810_U2_F4_GRIPPER".CYL.FULL_OPEN));
END_REGION

REGION Network 46: FIXTURE IN UNIT 02 MEASURING POSITION CLAMPED
   RUNG wire#powerrail
      Contact( "M_ONE" )
      wire#w1
      Contact( "DB4000_FIX_TABLE_POSITIONS".UNIT_02.FIXTURE_1.IN_MEASURING_STATION_2 )
      Contact( "DB3510_U2_F1_GRIPPER".CYL.FULL_CLOSED )
      wire#w2
      Coil( "DB2440_GLOBAL_DATA".GLOBAL_DATA.FIX_IN_UNIT_02_STA_2_CLAMPED )
   END_RUNG
   RUNG wire#w1
      Contact( "DB4000_FIX_TABLE_POSITIONS".UNIT_02.FIXTURE_2.IN_MEASURING_STATION_2 )
      Contact( "DB3610_U2_F2_GRIPPER".CYL.FULL_CLOSED )
   END_RUNG wire#w2
   RUNG wire#w1
      Contact( "DB4000_FIX_TABLE_POSITIONS".UNIT_02.FIXTURE_3.IN_MEASURING_STATION_2 )
      Contact( "DB3710_U2_F3_GRIPPER".CYL.FULL_CLOSED )
   END_RUNG wire#w2
   RUNG wire#w1
      Contact( "DB4000_FIX_TABLE_POSITIONS".UNIT_02.FIXTURE_4.IN_MEASURING_STATION_2 )
      Contact( "DB3810_U2_F4_GRIPPER".CYL.FULL_CLOSED )
   END_RUNG wire#w2
   // the same network as SCL:
   "DB2440_GLOBAL_DATA".GLOBAL_DATA.FIX_IN_UNIT_02_STA_2_CLAMPED := "M_ONE" AND (("DB4000_FIX_TABLE_POSITIONS".UNIT_02.FIXTURE_1.IN_MEASURING_STATION_2 AND "DB3510_U2_F1_GRIPPER".CYL.FULL_CLOSED) OR ("DB4000_FIX_TABLE_POSITIONS".UNIT_02.FIXTURE_2.IN_MEASURING_STATION_2 AND "DB3610_U2_F2_GRIPPER".CYL.FULL_CLOSED) OR ("DB4000_FIX_TABLE_POSITIONS".UNIT_02.FIXTURE_3.IN_MEASURING_STATION_2 AND "DB3710_U2_F3_GRIPPER".CYL.FULL_CLOSED) OR ("DB4000_FIX_TABLE_POSITIONS".UNIT_02.FIXTURE_4.IN_MEASURING_STATION_2 AND "DB3810_U2_F4_GRIPPER".CYL.FULL_CLOSED));
END_REGION

REGION Network 47: FIXTURE IN UNIT 01 CLADDING POSITION UNCLAMPED
   RUNG wire#powerrail
      Contact( "M_ONE" )
      wire#w1
      Contact( "DB4000_FIX_TABLE_POSITIONS".UNIT_01.FIXTURE_1.IN_CLADDING_STATION_3 )
      Contact( "DB2510_U1_F1_GRIPPER".CYL.FULL_OPEN )
      wire#w2
      Coil( "DB2440_GLOBAL_DATA".GLOBAL_DATA.FIX_IN_UNIT_01_STA_3_UNCLAMPED )
   END_RUNG
   RUNG wire#w1
      Contact( "DB4000_FIX_TABLE_POSITIONS".UNIT_01.FIXTURE_2.IN_CLADDING_STATION_3 )
      Contact( "DB2610_U1_F2_GRIPPER".CYL.FULL_OPEN )
   END_RUNG wire#w2
   RUNG wire#w1
      Contact( "DB4000_FIX_TABLE_POSITIONS".UNIT_01.FIXTURE_3.IN_CLADDING_STATION_3 )
      Contact( "DB2710_U1_F3_GRIPPER".CYL.FULL_OPEN )
   END_RUNG wire#w2
   RUNG wire#w1
      Contact( "DB4000_FIX_TABLE_POSITIONS".UNIT_01.FIXTURE_4.IN_CLADDING_STATION_3 )
      Contact( "DB2810_U1_F4_GRIPPER".CYL.FULL_OPEN )
   END_RUNG wire#w2
   // the same network as SCL:
   "DB2440_GLOBAL_DATA".GLOBAL_DATA.FIX_IN_UNIT_01_STA_3_UNCLAMPED := "M_ONE" AND (("DB4000_FIX_TABLE_POSITIONS".UNIT_01.FIXTURE_1.IN_CLADDING_STATION_3 AND "DB2510_U1_F1_GRIPPER".CYL.FULL_OPEN) OR ("DB4000_FIX_TABLE_POSITIONS".UNIT_01.FIXTURE_2.IN_CLADDING_STATION_3 AND "DB2610_U1_F2_GRIPPER".CYL.FULL_OPEN) OR ("DB4000_FIX_TABLE_POSITIONS".UNIT_01.FIXTURE_3.IN_CLADDING_STATION_3 AND "DB2710_U1_F3_GRIPPER".CYL.FULL_OPEN) OR ("DB4000_FIX_TABLE_POSITIONS".UNIT_01.FIXTURE_4.IN_CLADDING_STATION_3 AND "DB2810_U1_F4_GRIPPER".CYL.FULL_OPEN));
END_REGION

REGION Network 48: FIXTURE IN UNIT 01 CLADDING POSITION CLAMPED
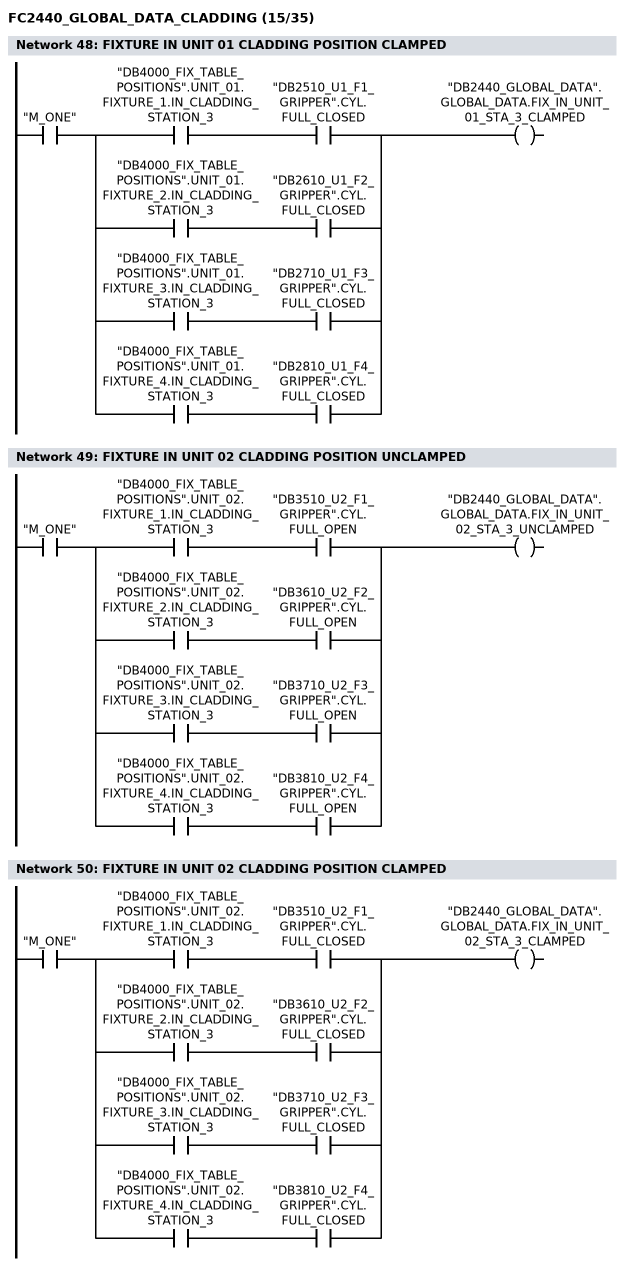
   RUNG wire#powerrail
      Contact( "M_ONE" )
      wire#w1
      Contact( "DB4000_FIX_TABLE_POSITIONS".UNIT_01.FIXTURE_1.IN_CLADDING_STATION_3 )
      Contact( "DB2510_U1_F1_GRIPPER".CYL.FULL_CLOSED )
      wire#w2
      Coil( "DB2440_GLOBAL_DATA".GLOBAL_DATA.FIX_IN_UNIT_01_STA_3_CLAMPED )
   END_RUNG
   RUNG wire#w1
      Contact( "DB4000_FIX_TABLE_POSITIONS".UNIT_01.FIXTURE_2.IN_CLADDING_STATION_3 )
      Contact( "DB2610_U1_F2_GRIPPER".CYL.FULL_CLOSED )
   END_RUNG wire#w2
   RUNG wire#w1
      Contact( "DB4000_FIX_TABLE_POSITIONS".UNIT_01.FIXTURE_3.IN_CLADDING_STATION_3 )
      Contact( "DB2710_U1_F3_GRIPPER".CYL.FULL_CLOSED )
   END_RUNG wire#w2
   RUNG wire#w1
      Contact( "DB4000_FIX_TABLE_POSITIONS".UNIT_01.FIXTURE_4.IN_CLADDING_STATION_3 )
      Contact( "DB2810_U1_F4_GRIPPER".CYL.FULL_CLOSED )
   END_RUNG wire#w2
   // the same network as SCL:
   "DB2440_GLOBAL_DATA".GLOBAL_DATA.FIX_IN_UNIT_01_STA_3_CLAMPED := "M_ONE" AND (("DB4000_FIX_TABLE_POSITIONS".UNIT_01.FIXTURE_1.IN_CLADDING_STATION_3 AND "DB2510_U1_F1_GRIPPER".CYL.FULL_CLOSED) OR ("DB4000_FIX_TABLE_POSITIONS".UNIT_01.FIXTURE_2.IN_CLADDING_STATION_3 AND "DB2610_U1_F2_GRIPPER".CYL.FULL_CLOSED) OR ("DB4000_FIX_TABLE_POSITIONS".UNIT_01.FIXTURE_3.IN_CLADDING_STATION_3 AND "DB2710_U1_F3_GRIPPER".CYL.FULL_CLOSED) OR ("DB4000_FIX_TABLE_POSITIONS".UNIT_01.FIXTURE_4.IN_CLADDING_STATION_3 AND "DB2810_U1_F4_GRIPPER".CYL.FULL_CLOSED));
END_REGION

REGION Network 49: FIXTURE IN UNIT 02 CLADDING POSITION UNCLAMPED
   RUNG wire#powerrail
      Contact( "M_ONE" )
      wire#w1
      Contact( "DB4000_FIX_TABLE_POSITIONS".UNIT_02.FIXTURE_1.IN_CLADDING_STATION_3 )
      Contact( "DB3510_U2_F1_GRIPPER".CYL.FULL_OPEN )
      wire#w2
      Coil( "DB2440_GLOBAL_DATA".GLOBAL_DATA.FIX_IN_UNIT_02_STA_3_UNCLAMPED )
   END_RUNG
   RUNG wire#w1
      Contact( "DB4000_FIX_TABLE_POSITIONS".UNIT_02.FIXTURE_2.IN_CLADDING_STATION_3 )
      Contact( "DB3610_U2_F2_GRIPPER".CYL.FULL_OPEN )
   END_RUNG wire#w2
   RUNG wire#w1
      Contact( "DB4000_FIX_TABLE_POSITIONS".UNIT_02.FIXTURE_3.IN_CLADDING_STATION_3 )
      Contact( "DB3710_U2_F3_GRIPPER".CYL.FULL_OPEN )
   END_RUNG wire#w2
   RUNG wire#w1
      Contact( "DB4000_FIX_TABLE_POSITIONS".UNIT_02.FIXTURE_4.IN_CLADDING_STATION_3 )
      Contact( "DB3810_U2_F4_GRIPPER".CYL.FULL_OPEN )
   END_RUNG wire#w2
   // the same network as SCL:
   "DB2440_GLOBAL_DATA".GLOBAL_DATA.FIX_IN_UNIT_02_STA_3_UNCLAMPED := "M_ONE" AND (("DB4000_FIX_TABLE_POSITIONS".UNIT_02.FIXTURE_1.IN_CLADDING_STATION_3 AND "DB3510_U2_F1_GRIPPER".CYL.FULL_OPEN) OR ("DB4000_FIX_TABLE_POSITIONS".UNIT_02.FIXTURE_2.IN_CLADDING_STATION_3 AND "DB3610_U2_F2_GRIPPER".CYL.FULL_OPEN) OR ("DB4000_FIX_TABLE_POSITIONS".UNIT_02.FIXTURE_3.IN_CLADDING_STATION_3 AND "DB3710_U2_F3_GRIPPER".CYL.FULL_OPEN) OR ("DB4000_FIX_TABLE_POSITIONS".UNIT_02.FIXTURE_4.IN_CLADDING_STATION_3 AND "DB3810_U2_F4_GRIPPER".CYL.FULL_OPEN));
END_REGION

REGION Network 50: FIXTURE IN UNIT 02 CLADDING POSITION CLAMPED
   RUNG wire#powerrail
      Contact( "M_ONE" )
      wire#w1
      Contact( "DB4000_FIX_TABLE_POSITIONS".UNIT_02.FIXTURE_1.IN_CLADDING_STATION_3 )
      Contact( "DB3510_U2_F1_GRIPPER".CYL.FULL_CLOSED )
      wire#w2
      Coil( "DB2440_GLOBAL_DATA".GLOBAL_DATA.FIX_IN_UNIT_02_STA_3_CLAMPED )
   END_RUNG
   RUNG wire#w1
      Contact( "DB4000_FIX_TABLE_POSITIONS".UNIT_02.FIXTURE_2.IN_CLADDING_STATION_3 )
      Contact( "DB3610_U2_F2_GRIPPER".CYL.FULL_CLOSED )
   END_RUNG wire#w2
   RUNG wire#w1
      Contact( "DB4000_FIX_TABLE_POSITIONS".UNIT_02.FIXTURE_3.IN_CLADDING_STATION_3 )
      Contact( "DB3710_U2_F3_GRIPPER".CYL.FULL_CLOSED )
   END_RUNG wire#w2
   RUNG wire#w1
      Contact( "DB4000_FIX_TABLE_POSITIONS".UNIT_02.FIXTURE_4.IN_CLADDING_STATION_3 )
      Contact( "DB3810_U2_F4_GRIPPER".CYL.FULL_CLOSED )
   END_RUNG wire#w2
   // the same network as SCL:
   "DB2440_GLOBAL_DATA".GLOBAL_DATA.FIX_IN_UNIT_02_STA_3_CLAMPED := "M_ONE" AND (("DB4000_FIX_TABLE_POSITIONS".UNIT_02.FIXTURE_1.IN_CLADDING_STATION_3 AND "DB3510_U2_F1_GRIPPER".CYL.FULL_CLOSED) OR ("DB4000_FIX_TABLE_POSITIONS".UNIT_02.FIXTURE_2.IN_CLADDING_STATION_3 AND "DB3610_U2_F2_GRIPPER".CYL.FULL_CLOSED) OR ("DB4000_FIX_TABLE_POSITIONS".UNIT_02.FIXTURE_3.IN_CLADDING_STATION_3 AND "DB3710_U2_F3_GRIPPER".CYL.FULL_CLOSED) OR ("DB4000_FIX_TABLE_POSITIONS".UNIT_02.FIXTURE_4.IN_CLADDING_STATION_3 AND "DB3810_U2_F4_GRIPPER".CYL.FULL_CLOSED));
END_REGION

REGION Network 51: FIXTURE IN UNIT 01 MEASURING/CLEANING POSITION UNCLAMPED
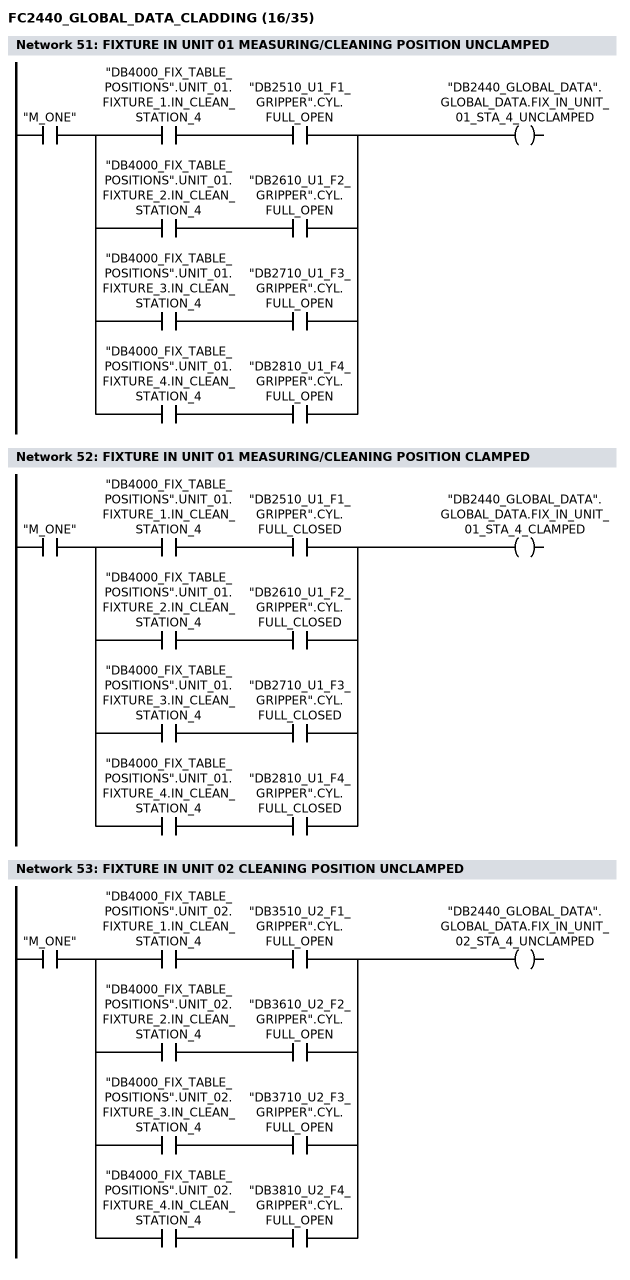
   RUNG wire#powerrail
      Contact( "M_ONE" )
      wire#w1
      Contact( "DB4000_FIX_TABLE_POSITIONS".UNIT_01.FIXTURE_1.IN_CLEAN_STATION_4 )
      Contact( "DB2510_U1_F1_GRIPPER".CYL.FULL_OPEN )
      wire#w2
      Coil( "DB2440_GLOBAL_DATA".GLOBAL_DATA.FIX_IN_UNIT_01_STA_4_UNCLAMPED )
   END_RUNG
   RUNG wire#w1
      Contact( "DB4000_FIX_TABLE_POSITIONS".UNIT_01.FIXTURE_2.IN_CLEAN_STATION_4 )
      Contact( "DB2610_U1_F2_GRIPPER".CYL.FULL_OPEN )
   END_RUNG wire#w2
   RUNG wire#w1
      Contact( "DB4000_FIX_TABLE_POSITIONS".UNIT_01.FIXTURE_3.IN_CLEAN_STATION_4 )
      Contact( "DB2710_U1_F3_GRIPPER".CYL.FULL_OPEN )
   END_RUNG wire#w2
   RUNG wire#w1
      Contact( "DB4000_FIX_TABLE_POSITIONS".UNIT_01.FIXTURE_4.IN_CLEAN_STATION_4 )
      Contact( "DB2810_U1_F4_GRIPPER".CYL.FULL_OPEN )
   END_RUNG wire#w2
   // the same network as SCL:
   "DB2440_GLOBAL_DATA".GLOBAL_DATA.FIX_IN_UNIT_01_STA_4_UNCLAMPED := "M_ONE" AND (("DB4000_FIX_TABLE_POSITIONS".UNIT_01.FIXTURE_1.IN_CLEAN_STATION_4 AND "DB2510_U1_F1_GRIPPER".CYL.FULL_OPEN) OR ("DB4000_FIX_TABLE_POSITIONS".UNIT_01.FIXTURE_2.IN_CLEAN_STATION_4 AND "DB2610_U1_F2_GRIPPER".CYL.FULL_OPEN) OR ("DB4000_FIX_TABLE_POSITIONS".UNIT_01.FIXTURE_3.IN_CLEAN_STATION_4 AND "DB2710_U1_F3_GRIPPER".CYL.FULL_OPEN) OR ("DB4000_FIX_TABLE_POSITIONS".UNIT_01.FIXTURE_4.IN_CLEAN_STATION_4 AND "DB2810_U1_F4_GRIPPER".CYL.FULL_OPEN));
END_REGION

REGION Network 52: FIXTURE IN UNIT 01 MEASURING/CLEANING POSITION CLAMPED
   RUNG wire#powerrail
      Contact( "M_ONE" )
      wire#w1
      Contact( "DB4000_FIX_TABLE_POSITIONS".UNIT_01.FIXTURE_1.IN_CLEAN_STATION_4 )
      Contact( "DB2510_U1_F1_GRIPPER".CYL.FULL_CLOSED )
      wire#w2
      Coil( "DB2440_GLOBAL_DATA".GLOBAL_DATA.FIX_IN_UNIT_01_STA_4_CLAMPED )
   END_RUNG
   RUNG wire#w1
      Contact( "DB4000_FIX_TABLE_POSITIONS".UNIT_01.FIXTURE_2.IN_CLEAN_STATION_4 )
      Contact( "DB2610_U1_F2_GRIPPER".CYL.FULL_CLOSED )
   END_RUNG wire#w2
   RUNG wire#w1
      Contact( "DB4000_FIX_TABLE_POSITIONS".UNIT_01.FIXTURE_3.IN_CLEAN_STATION_4 )
      Contact( "DB2710_U1_F3_GRIPPER".CYL.FULL_CLOSED )
   END_RUNG wire#w2
   RUNG wire#w1
      Contact( "DB4000_FIX_TABLE_POSITIONS".UNIT_01.FIXTURE_4.IN_CLEAN_STATION_4 )
      Contact( "DB2810_U1_F4_GRIPPER".CYL.FULL_CLOSED )
   END_RUNG wire#w2
   // the same network as SCL:
   "DB2440_GLOBAL_DATA".GLOBAL_DATA.FIX_IN_UNIT_01_STA_4_CLAMPED := "M_ONE" AND (("DB4000_FIX_TABLE_POSITIONS".UNIT_01.FIXTURE_1.IN_CLEAN_STATION_4 AND "DB2510_U1_F1_GRIPPER".CYL.FULL_CLOSED) OR ("DB4000_FIX_TABLE_POSITIONS".UNIT_01.FIXTURE_2.IN_CLEAN_STATION_4 AND "DB2610_U1_F2_GRIPPER".CYL.FULL_CLOSED) OR ("DB4000_FIX_TABLE_POSITIONS".UNIT_01.FIXTURE_3.IN_CLEAN_STATION_4 AND "DB2710_U1_F3_GRIPPER".CYL.FULL_CLOSED) OR ("DB4000_FIX_TABLE_POSITIONS".UNIT_01.FIXTURE_4.IN_CLEAN_STATION_4 AND "DB2810_U1_F4_GRIPPER".CYL.FULL_CLOSED));
END_REGION

REGION Network 53: FIXTURE IN UNIT 02 CLEANING POSITION UNCLAMPED
   RUNG wire#powerrail
      Contact( "M_ONE" )
      wire#w1
      Contact( "DB4000_FIX_TABLE_POSITIONS".UNIT_02.FIXTURE_1.IN_CLEAN_STATION_4 )
      Contact( "DB3510_U2_F1_GRIPPER".CYL.FULL_OPEN )
      wire#w2
      Coil( "DB2440_GLOBAL_DATA".GLOBAL_DATA.FIX_IN_UNIT_02_STA_4_UNCLAMPED )
   END_RUNG
   RUNG wire#w1
      Contact( "DB4000_FIX_TABLE_POSITIONS".UNIT_02.FIXTURE_2.IN_CLEAN_STATION_4 )
      Contact( "DB3610_U2_F2_GRIPPER".CYL.FULL_OPEN )
   END_RUNG wire#w2
   RUNG wire#w1
      Contact( "DB4000_FIX_TABLE_POSITIONS".UNIT_02.FIXTURE_3.IN_CLEAN_STATION_4 )
      Contact( "DB3710_U2_F3_GRIPPER".CYL.FULL_OPEN )
   END_RUNG wire#w2
   RUNG wire#w1
      Contact( "DB4000_FIX_TABLE_POSITIONS".UNIT_02.FIXTURE_4.IN_CLEAN_STATION_4 )
      Contact( "DB3810_U2_F4_GRIPPER".CYL.FULL_OPEN )
   END_RUNG wire#w2
   // the same network as SCL:
   "DB2440_GLOBAL_DATA".GLOBAL_DATA.FIX_IN_UNIT_02_STA_4_UNCLAMPED := "M_ONE" AND (("DB4000_FIX_TABLE_POSITIONS".UNIT_02.FIXTURE_1.IN_CLEAN_STATION_4 AND "DB3510_U2_F1_GRIPPER".CYL.FULL_OPEN) OR ("DB4000_FIX_TABLE_POSITIONS".UNIT_02.FIXTURE_2.IN_CLEAN_STATION_4 AND "DB3610_U2_F2_GRIPPER".CYL.FULL_OPEN) OR ("DB4000_FIX_TABLE_POSITIONS".UNIT_02.FIXTURE_3.IN_CLEAN_STATION_4 AND "DB3710_U2_F3_GRIPPER".CYL.FULL_OPEN) OR ("DB4000_FIX_TABLE_POSITIONS".UNIT_02.FIXTURE_4.IN_CLEAN_STATION_4 AND "DB3810_U2_F4_GRIPPER".CYL.FULL_OPEN));
END_REGION

REGION Network 54: FIXTURE IN UNIT 02 CLEANING POSITION CLAMPED
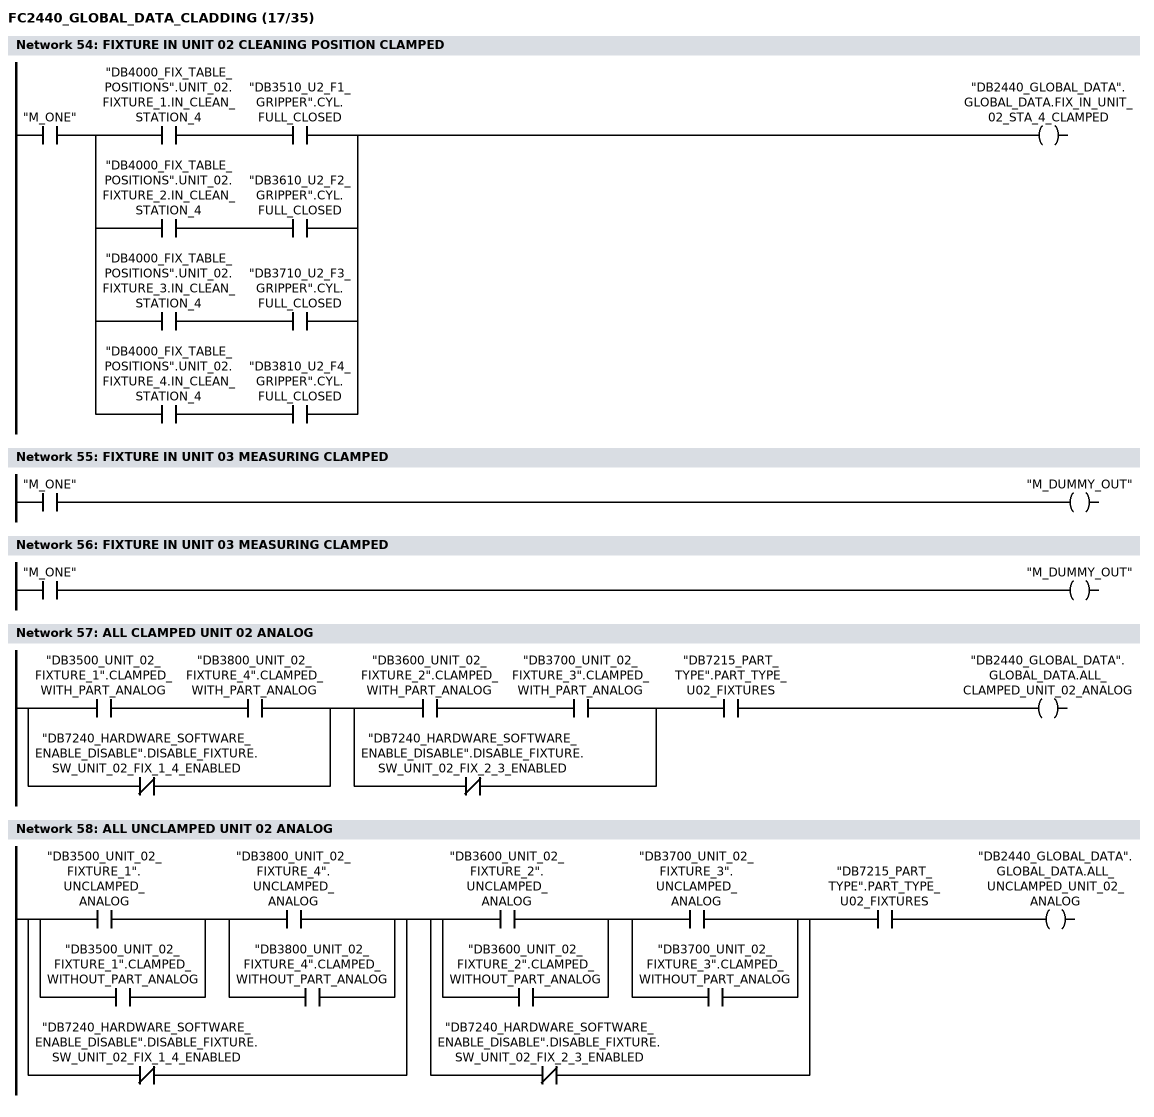
   RUNG wire#powerrail
      Contact( "M_ONE" )
      wire#w1
      Contact( "DB4000_FIX_TABLE_POSITIONS".UNIT_02.FIXTURE_1.IN_CLEAN_STATION_4 )
      Contact( "DB3510_U2_F1_GRIPPER".CYL.FULL_CLOSED )
      wire#w2
      Coil( "DB2440_GLOBAL_DATA".GLOBAL_DATA.FIX_IN_UNIT_02_STA_4_CLAMPED )
   END_RUNG
   RUNG wire#w1
      Contact( "DB4000_FIX_TABLE_POSITIONS".UNIT_02.FIXTURE_2.IN_CLEAN_STATION_4 )
      Contact( "DB3610_U2_F2_GRIPPER".CYL.FULL_CLOSED )
   END_RUNG wire#w2
   RUNG wire#w1
      Contact( "DB4000_FIX_TABLE_POSITIONS".UNIT_02.FIXTURE_3.IN_CLEAN_STATION_4 )
      Contact( "DB3710_U2_F3_GRIPPER".CYL.FULL_CLOSED )
   END_RUNG wire#w2
   RUNG wire#w1
      Contact( "DB4000_FIX_TABLE_POSITIONS".UNIT_02.FIXTURE_4.IN_CLEAN_STATION_4 )
      Contact( "DB3810_U2_F4_GRIPPER".CYL.FULL_CLOSED )
   END_RUNG wire#w2
   // the same network as SCL:
   "DB2440_GLOBAL_DATA".GLOBAL_DATA.FIX_IN_UNIT_02_STA_4_CLAMPED := "M_ONE" AND (("DB4000_FIX_TABLE_POSITIONS".UNIT_02.FIXTURE_1.IN_CLEAN_STATION_4 AND "DB3510_U2_F1_GRIPPER".CYL.FULL_CLOSED) OR ("DB4000_FIX_TABLE_POSITIONS".UNIT_02.FIXTURE_2.IN_CLEAN_STATION_4 AND "DB3610_U2_F2_GRIPPER".CYL.FULL_CLOSED) OR ("DB4000_FIX_TABLE_POSITIONS".UNIT_02.FIXTURE_3.IN_CLEAN_STATION_4 AND "DB3710_U2_F3_GRIPPER".CYL.FULL_CLOSED) OR ("DB4000_FIX_TABLE_POSITIONS".UNIT_02.FIXTURE_4.IN_CLEAN_STATION_4 AND "DB3810_U2_F4_GRIPPER".CYL.FULL_CLOSED));
END_REGION

REGION Network 55: FIXTURE IN UNIT 03 MEASURING CLAMPED
   RUNG wire#powerrail
      Contact( "M_ONE" )
      Coil( "M_DUMMY_OUT" )
   END_RUNG
   // the same network as SCL:
   "M_DUMMY_OUT" := "M_ONE";
END_REGION

REGION Network 56: FIXTURE IN UNIT 03 MEASURING CLAMPED
   RUNG wire#powerrail
      Contact( "M_ONE" )
      Coil( "M_DUMMY_OUT" )
   END_RUNG
   // the same network as SCL:
   "M_DUMMY_OUT" := "M_ONE";
END_REGION

REGION Network 57: ALL CLAMPED UNIT 02 ANALOG
   RUNG wire#powerrail
      Contact( "DB3500_UNIT_02_FIXTURE_1".CLAMPED_WITH_PART_ANALOG )
      Contact( "DB3800_UNIT_02_FIXTURE_4".CLAMPED_WITH_PART_ANALOG )
      wire#w1
      Contact( "DB3600_UNIT_02_FIXTURE_2".CLAMPED_WITH_PART_ANALOG )
      Contact( "DB3700_UNIT_02_FIXTURE_3".CLAMPED_WITH_PART_ANALOG )
      wire#w2
      Contact( "DB7215_PART_TYPE".PART_TYPE_U02_FIXTURES )
      Coil( "DB2440_GLOBAL_DATA".GLOBAL_DATA.ALL_CLAMPED_UNIT_02_ANALOG )
   END_RUNG
   RUNG wire#powerrail
      I_Contact( "DB7240_HARDWARE_SOFTWARE_ENABLE_DISABLE".DISABLE_FIXTURE.SW_UNIT_02_FIX_1_4_ENABLED )
   END_RUNG wire#w1
   RUNG wire#w1
      I_Contact( "DB7240_HARDWARE_SOFTWARE_ENABLE_DISABLE".DISABLE_FIXTURE.SW_UNIT_02_FIX_2_3_ENABLED )
   END_RUNG wire#w2
   // the same network as SCL:
   "DB2440_GLOBAL_DATA".GLOBAL_DATA.ALL_CLAMPED_UNIT_02_ANALOG := (("DB3500_UNIT_02_FIXTURE_1".CLAMPED_WITH_PART_ANALOG AND "DB3800_UNIT_02_FIXTURE_4".CLAMPED_WITH_PART_ANALOG) OR NOT "DB7240_HARDWARE_SOFTWARE_ENABLE_DISABLE".DISABLE_FIXTURE.SW_UNIT_02_FIX_1_4_ENABLED) AND (("DB3600_UNIT_02_FIXTURE_2".CLAMPED_WITH_PART_ANALOG AND "DB3700_UNIT_02_FIXTURE_3".CLAMPED_WITH_PART_ANALOG) OR NOT "DB7240_HARDWARE_SOFTWARE_ENABLE_DISABLE".DISABLE_FIXTURE.SW_UNIT_02_FIX_2_3_ENABLED) AND "DB7215_PART_TYPE".PART_TYPE_U02_FIXTURES;
END_REGION

REGION Network 58: ALL UNCLAMPED UNIT 02 ANALOG
   RUNG wire#powerrail
      Contact( "DB3500_UNIT_02_FIXTURE_1".UNCLAMPED_ANALOG )
      wire#w1
      Contact( "DB3800_UNIT_02_FIXTURE_4".UNCLAMPED_ANALOG )
      wire#w2
      Contact( "DB3600_UNIT_02_FIXTURE_2".UNCLAMPED_ANALOG )
      wire#w3
      Contact( "DB3700_UNIT_02_FIXTURE_3".UNCLAMPED_ANALOG )
      wire#w4
      Contact( "DB7215_PART_TYPE".PART_TYPE_U02_FIXTURES )
      Coil( "DB2440_GLOBAL_DATA".GLOBAL_DATA.ALL_UNCLAMPED_UNIT_02_ANALOG )
   END_RUNG
   RUNG wire#powerrail
      Contact( "DB3500_UNIT_02_FIXTURE_1".CLAMPED_WITHOUT_PART_ANALOG )
   END_RUNG wire#w1
   RUNG wire#w1
      Contact( "DB3800_UNIT_02_FIXTURE_4".CLAMPED_WITHOUT_PART_ANALOG )
   END_RUNG wire#w2
   RUNG wire#powerrail
      I_Contact( "DB7240_HARDWARE_SOFTWARE_ENABLE_DISABLE".DISABLE_FIXTURE.SW_UNIT_02_FIX_1_4_ENABLED )
   END_RUNG wire#w2
   RUNG wire#w2
      Contact( "DB3600_UNIT_02_FIXTURE_2".CLAMPED_WITHOUT_PART_ANALOG )
   END_RUNG wire#w3
   RUNG wire#w3
      Contact( "DB3700_UNIT_02_FIXTURE_3".CLAMPED_WITHOUT_PART_ANALOG )
   END_RUNG wire#w4
   RUNG wire#w2
      I_Contact( "DB7240_HARDWARE_SOFTWARE_ENABLE_DISABLE".DISABLE_FIXTURE.SW_UNIT_02_FIX_2_3_ENABLED )
   END_RUNG wire#w4
   // the same network as SCL:
   "DB2440_GLOBAL_DATA".GLOBAL_DATA.ALL_UNCLAMPED_UNIT_02_ANALOG := ((("DB3500_UNIT_02_FIXTURE_1".UNCLAMPED_ANALOG OR "DB3500_UNIT_02_FIXTURE_1".CLAMPED_WITHOUT_PART_ANALOG) AND ("DB3800_UNIT_02_FIXTURE_4".UNCLAMPED_ANALOG OR "DB3800_UNIT_02_FIXTURE_4".CLAMPED_WITHOUT_PART_ANALOG)) OR NOT "DB7240_HARDWARE_SOFTWARE_ENABLE_DISABLE".DISABLE_FIXTURE.SW_UNIT_02_FIX_1_4_ENABLED) AND ((("DB3600_UNIT_02_FIXTURE_2".UNCLAMPED_ANALOG OR "DB3600_UNIT_02_FIXTURE_2".CLAMPED_WITHOUT_PART_ANALOG) AND ("DB3700_UNIT_02_FIXTURE_3".UNCLAMPED_ANALOG OR "DB3700_UNIT_02_FIXTURE_3".CLAMPED_WITHOUT_PART_ANALOG)) OR NOT "DB7240_HARDWARE_SOFTWARE_ENABLE_DISABLE".DISABLE_FIXTURE.SW_UNIT_02_FIX_2_3_ENABLED) AND "DB7215_PART_TYPE".PART_TYPE_U02_FIXTURES;
END_REGION

REGION Network 59: CLAMPED OR UNCLAMPED UNIT 02 ANALOG
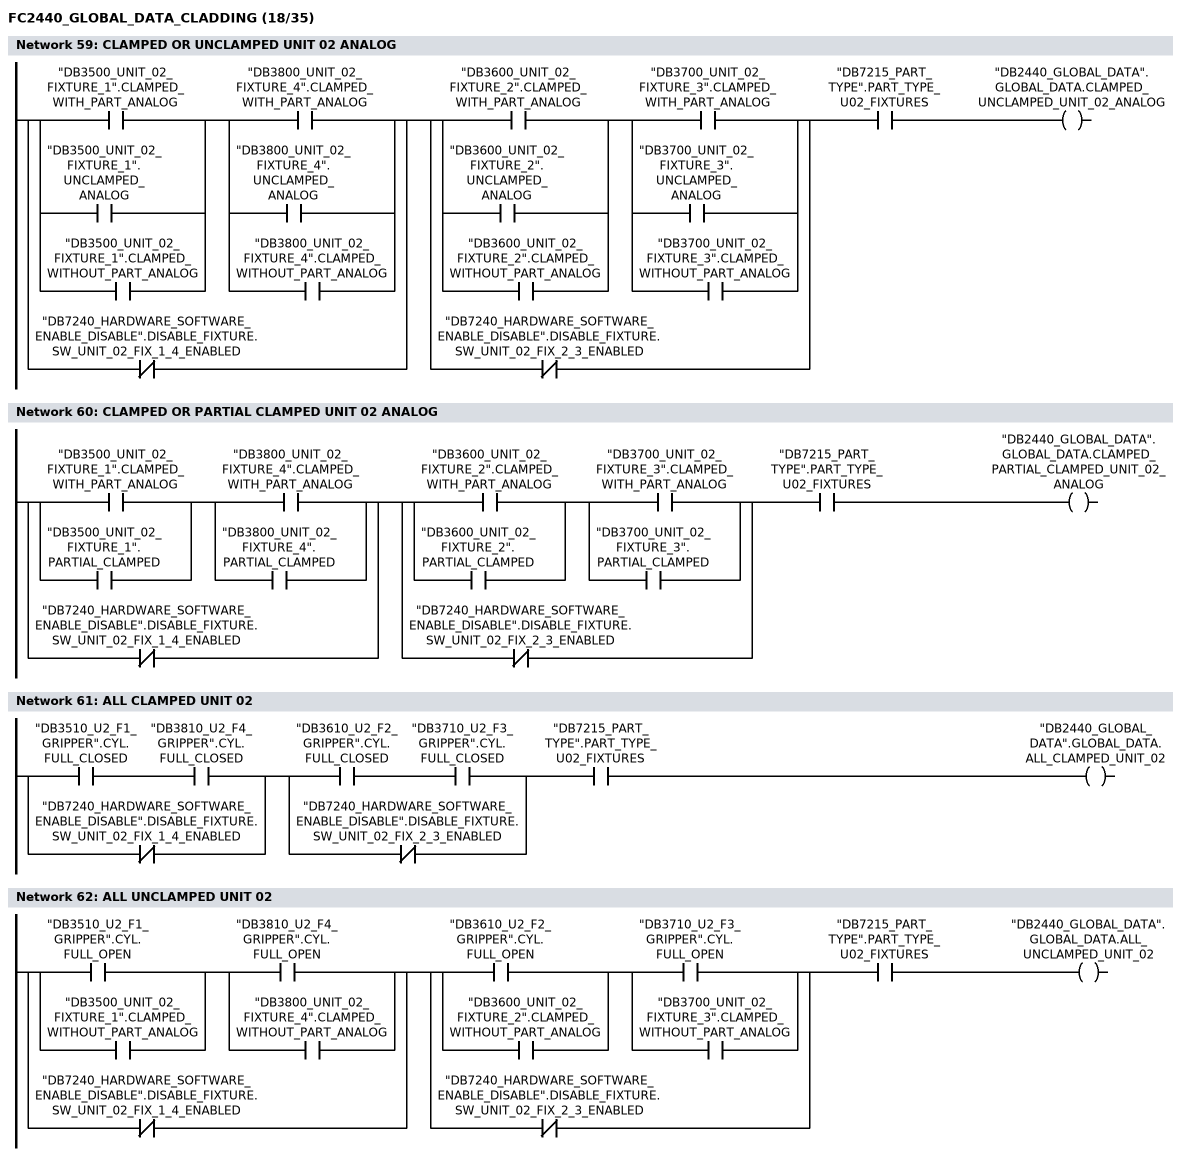
   RUNG wire#powerrail
      Contact( "DB3500_UNIT_02_FIXTURE_1".CLAMPED_WITH_PART_ANALOG )
      wire#w1
      Contact( "DB3800_UNIT_02_FIXTURE_4".CLAMPED_WITH_PART_ANALOG )
      wire#w2
      Contact( "DB3600_UNIT_02_FIXTURE_2".CLAMPED_WITH_PART_ANALOG )
      wire#w3
      Contact( "DB3700_UNIT_02_FIXTURE_3".CLAMPED_WITH_PART_ANALOG )
      wire#w4
      Contact( "DB7215_PART_TYPE".PART_TYPE_U02_FIXTURES )
      Coil( "DB2440_GLOBAL_DATA".GLOBAL_DATA.CLAMPED_UNCLAMPED_UNIT_02_ANALOG )
   END_RUNG
   RUNG wire#powerrail
      Contact( "DB3500_UNIT_02_FIXTURE_1".UNCLAMPED_ANALOG )
   END_RUNG wire#w1
   RUNG wire#powerrail
      Contact( "DB3500_UNIT_02_FIXTURE_1".CLAMPED_WITHOUT_PART_ANALOG )
   END_RUNG wire#w1
   RUNG wire#w1
      Contact( "DB3800_UNIT_02_FIXTURE_4".UNCLAMPED_ANALOG )
   END_RUNG wire#w2
   RUNG wire#w1
      Contact( "DB3800_UNIT_02_FIXTURE_4".CLAMPED_WITHOUT_PART_ANALOG )
   END_RUNG wire#w2
   RUNG wire#powerrail
      I_Contact( "DB7240_HARDWARE_SOFTWARE_ENABLE_DISABLE".DISABLE_FIXTURE.SW_UNIT_02_FIX_1_4_ENABLED )
   END_RUNG wire#w2
   RUNG wire#w2
      Contact( "DB3600_UNIT_02_FIXTURE_2".UNCLAMPED_ANALOG )
   END_RUNG wire#w3
   RUNG wire#w2
      Contact( "DB3600_UNIT_02_FIXTURE_2".CLAMPED_WITHOUT_PART_ANALOG )
   END_RUNG wire#w3
   RUNG wire#w3
      Contact( "DB3700_UNIT_02_FIXTURE_3".UNCLAMPED_ANALOG )
   END_RUNG wire#w4
   RUNG wire#w3
      Contact( "DB3700_UNIT_02_FIXTURE_3".CLAMPED_WITHOUT_PART_ANALOG )
   END_RUNG wire#w4
   RUNG wire#w2
      I_Contact( "DB7240_HARDWARE_SOFTWARE_ENABLE_DISABLE".DISABLE_FIXTURE.SW_UNIT_02_FIX_2_3_ENABLED )
   END_RUNG wire#w4
   // the same network as SCL:
   "DB2440_GLOBAL_DATA".GLOBAL_DATA.CLAMPED_UNCLAMPED_UNIT_02_ANALOG := ((("DB3500_UNIT_02_FIXTURE_1".CLAMPED_WITH_PART_ANALOG OR "DB3500_UNIT_02_FIXTURE_1".UNCLAMPED_ANALOG OR "DB3500_UNIT_02_FIXTURE_1".CLAMPED_WITHOUT_PART_ANALOG) AND ("DB3800_UNIT_02_FIXTURE_4".CLAMPED_WITH_PART_ANALOG OR "DB3800_UNIT_02_FIXTURE_4".UNCLAMPED_ANALOG OR "DB3800_UNIT_02_FIXTURE_4".CLAMPED_WITHOUT_PART_ANALOG)) OR NOT "DB7240_HARDWARE_SOFTWARE_ENABLE_DISABLE".DISABLE_FIXTURE.SW_UNIT_02_FIX_1_4_ENABLED) AND ((("DB3600_UNIT_02_FIXTURE_2".CLAMPED_WITH_PART_ANALOG OR "DB3600_UNIT_02_FIXTURE_2".UNCLAMPED_ANALOG OR "DB3600_UNIT_02_FIXTURE_2".CLAMPED_WITHOUT_PART_ANALOG) AND ("DB3700_UNIT_02_FIXTURE_3".CLAMPED_WITH_PART_ANALOG OR "DB3700_UNIT_02_FIXTURE_3".UNCLAMPED_ANALOG OR "DB3700_UNIT_02_FIXTURE_3".CLAMPED_WITHOUT_PART_ANALOG)) OR NOT "DB7240_HARDWARE_SOFTWARE_ENABLE_DISABLE".DISABLE_FIXTURE.SW_UNIT_02_FIX_2_3_ENABLED) AND "DB7215_PART_TYPE".PART_TYPE_U02_FIXTURES;
END_REGION

REGION Network 60: CLAMPED OR PARTIAL CLAMPED UNIT 02 ANALOG
   RUNG wire#powerrail
      Contact( "DB3500_UNIT_02_FIXTURE_1".CLAMPED_WITH_PART_ANALOG )
      wire#w1
      Contact( "DB3800_UNIT_02_FIXTURE_4".CLAMPED_WITH_PART_ANALOG )
      wire#w2
      Contact( "DB3600_UNIT_02_FIXTURE_2".CLAMPED_WITH_PART_ANALOG )
      wire#w3
      Contact( "DB3700_UNIT_02_FIXTURE_3".CLAMPED_WITH_PART_ANALOG )
      wire#w4
      Contact( "DB7215_PART_TYPE".PART_TYPE_U02_FIXTURES )
      Coil( "DB2440_GLOBAL_DATA".GLOBAL_DATA.CLAMPED_PARTIAL_CLAMPED_UNIT_02_ANALOG )
   END_RUNG
   RUNG wire#powerrail
      Contact( "DB3500_UNIT_02_FIXTURE_1".PARTIAL_CLAMPED )
   END_RUNG wire#w1
   RUNG wire#w1
      Contact( "DB3800_UNIT_02_FIXTURE_4".PARTIAL_CLAMPED )
   END_RUNG wire#w2
   RUNG wire#powerrail
      I_Contact( "DB7240_HARDWARE_SOFTWARE_ENABLE_DISABLE".DISABLE_FIXTURE.SW_UNIT_02_FIX_1_4_ENABLED )
   END_RUNG wire#w2
   RUNG wire#w2
      Contact( "DB3600_UNIT_02_FIXTURE_2".PARTIAL_CLAMPED )
   END_RUNG wire#w3
   RUNG wire#w3
      Contact( "DB3700_UNIT_02_FIXTURE_3".PARTIAL_CLAMPED )
   END_RUNG wire#w4
   RUNG wire#w2
      I_Contact( "DB7240_HARDWARE_SOFTWARE_ENABLE_DISABLE".DISABLE_FIXTURE.SW_UNIT_02_FIX_2_3_ENABLED )
   END_RUNG wire#w4
   // the same network as SCL:
   "DB2440_GLOBAL_DATA".GLOBAL_DATA.CLAMPED_PARTIAL_CLAMPED_UNIT_02_ANALOG := ((("DB3500_UNIT_02_FIXTURE_1".CLAMPED_WITH_PART_ANALOG OR "DB3500_UNIT_02_FIXTURE_1".PARTIAL_CLAMPED) AND ("DB3800_UNIT_02_FIXTURE_4".CLAMPED_WITH_PART_ANALOG OR "DB3800_UNIT_02_FIXTURE_4".PARTIAL_CLAMPED)) OR NOT "DB7240_HARDWARE_SOFTWARE_ENABLE_DISABLE".DISABLE_FIXTURE.SW_UNIT_02_FIX_1_4_ENABLED) AND ((("DB3600_UNIT_02_FIXTURE_2".CLAMPED_WITH_PART_ANALOG OR "DB3600_UNIT_02_FIXTURE_2".PARTIAL_CLAMPED) AND ("DB3700_UNIT_02_FIXTURE_3".CLAMPED_WITH_PART_ANALOG OR "DB3700_UNIT_02_FIXTURE_3".PARTIAL_CLAMPED)) OR NOT "DB7240_HARDWARE_SOFTWARE_ENABLE_DISABLE".DISABLE_FIXTURE.SW_UNIT_02_FIX_2_3_ENABLED) AND "DB7215_PART_TYPE".PART_TYPE_U02_FIXTURES;
END_REGION

REGION Network 61: ALL CLAMPED UNIT 02
   RUNG wire#powerrail
      Contact( "DB3510_U2_F1_GRIPPER".CYL.FULL_CLOSED )
      Contact( "DB3810_U2_F4_GRIPPER".CYL.FULL_CLOSED )
      wire#w1
      Contact( "DB3610_U2_F2_GRIPPER".CYL.FULL_CLOSED )
      Contact( "DB3710_U2_F3_GRIPPER".CYL.FULL_CLOSED )
      wire#w2
      Contact( "DB7215_PART_TYPE".PART_TYPE_U02_FIXTURES )
      Coil( "DB2440_GLOBAL_DATA".GLOBAL_DATA.ALL_CLAMPED_UNIT_02 )
   END_RUNG
   RUNG wire#powerrail
      I_Contact( "DB7240_HARDWARE_SOFTWARE_ENABLE_DISABLE".DISABLE_FIXTURE.SW_UNIT_02_FIX_1_4_ENABLED )
   END_RUNG wire#w1
   RUNG wire#w1
      I_Contact( "DB7240_HARDWARE_SOFTWARE_ENABLE_DISABLE".DISABLE_FIXTURE.SW_UNIT_02_FIX_2_3_ENABLED )
   END_RUNG wire#w2
   // the same network as SCL:
   "DB2440_GLOBAL_DATA".GLOBAL_DATA.ALL_CLAMPED_UNIT_02 := (("DB3510_U2_F1_GRIPPER".CYL.FULL_CLOSED AND "DB3810_U2_F4_GRIPPER".CYL.FULL_CLOSED) OR NOT "DB7240_HARDWARE_SOFTWARE_ENABLE_DISABLE".DISABLE_FIXTURE.SW_UNIT_02_FIX_1_4_ENABLED) AND (("DB3610_U2_F2_GRIPPER".CYL.FULL_CLOSED AND "DB3710_U2_F3_GRIPPER".CYL.FULL_CLOSED) OR NOT "DB7240_HARDWARE_SOFTWARE_ENABLE_DISABLE".DISABLE_FIXTURE.SW_UNIT_02_FIX_2_3_ENABLED) AND "DB7215_PART_TYPE".PART_TYPE_U02_FIXTURES;
END_REGION

